(* CODESYS project Rack.project

Project tree, tasks and I/O mapping:
  Device : AM401-CPU1608TP/TN, Shenzhen Inovance Control Technology, version 3.5.11.11
      settings: PersistentStartAdddr = 120000; PersistentStartEndAddr = 491519; Mode = 1
    application Application
      libraries: Standard, * (System); CmpLog, 3.5.5.0 (System); SysMem, 3.5.5.0 (System); CmpEventMgr, 3.5.8.0 (System); CmpApp, 3.5.11.0 (System)
      task MainTask (cyclic, interval 20 ms, priority 1) calls PLC_PRG
      task ETHERCAT (cyclic, interval 4000 µs, priority 0) calls ETHERCAT.EtherCAT_Task, Axis_Ctrl
      02_功能块/
        气缸/
          function block FB_Cylinder [LD]
        初始化/
          function block FB_LineCylinderInit [LD]
          function block FB_MainlineInit [LD]
          function block FB_MaterialInit [LD]
          function block FB_CylinderInit [LD]
      01_变量/
        global variables PersistentVars
        global variables GVL_FB
        global variables GVL_X
        global variables GVL_G
        global variables GVL_H
        global variables GVL_T
        global variables GVL_Q
        global variables GVL_O
        global variables GVT_INT
        global variables GVL_Axis
      03_程序/
        自动/
          program Auto_A [LD]
          program Auto_C [LD]
        输出/
          program Other [LD]
          program Cylinder_AZone [ST]
          program Cylinder_CZone [ST]
        系统/
          program Mode [LD]
          program Rst [LD]
        异常/
          program Error [LD]
        伺服控制/
          program Axis_Teaching [LD]
          program Axis_Ctrl [LD]
        OB/
          program PLC_PRG [ST]
      DifferentialMonitor
    ConfigStorage
    Device Diagnosis
    Network Configuration
      LocalBus Config
      EtherCAT Config
    HardWare Configuration
    资源使用表
    SoftMotion General Axis Pool
    HIGH_SPEED_IO : High Speed IO Module, Inovance, version 00.00.00.20
        unmapped channels: %IW0 InputData, %QB0 OutputData
      HSIO
    HwConfiguratioinDevice : SystemConfig, Inovance, version 00.00.00.10
        settings: NetworkConfigArray.NetworkConfigArray.BusType = 10; NetworkConfigArray.NetworkConfigArray.RackSum = 1; NetworkConfigArray.NetworkConfigArray.HardwareConfigArray.HardwareConfigArray.RackNo = 1
    ETHERCAT : EtherCAT Master, 3S - Smart Software Solutions GmbH, version 3.5.11.10
        settings:  = 0; NetworkName = 'eth1'; SelectNetworkByName = TRUE; DisableTaskGeneration = True
      Z1 : SV660_1Axis_V0.08, Inovance, order no. InoSV660N, version Revision=16#00010000
          settings: WriteValueList = H03-03_8195_4_1_UINT_RW;H03-05_8195_6_1_UINT_RW;H03-06_8195_7_31_UINT_RW;H03-07_8195_8_0_UINT_RW;; Number of Outputs = 2; Number of Inputs = 4; Number of Infos about Outputs = 2; Number of Infos about Inputs = 4; Sync.Length = 6; Sync.Length = 12; FMMU.Length = 6; FMMU.Length = 12; AutoUpdate = False; DC sync0 cycletime = 4000; DC sync1 cycletime = 4000; Number of SDO = 9; Homing method.Index = 16#6098; Homing method.Subindex = 16#00; Homing method.Value = 29; Homing method.Size = 8; Homing method.AbortIfError = FALSE; Homing method.JumpToLine = FALSE; Homing method.Line = 0; Homing method.CompleteAccess = FALSE; Speed during search for switch.Index = 16#6099; Speed during search for switch.Subindex = 16#01; Speed during search for switch.Value = 8388608; Speed during search for switch.Size = 32; Speed during search for switch.AbortIfError = FALSE; Speed during search for switch.JumpToLine = FALSE; Speed during search for switch.Line = 0; Speed during search for switch.CompleteAccess = FALSE; Homing acceleration.Index = 16#609A; Homing acceleration.Subindex = 16#00; Homing acceleration.Value = 167772160; Homing acceleration.Size = 32; Homing acceleration.AbortIfError = FALSE; Homing acceleration.JumpToLine = FALSE; Homing acceleration.Line = 0; Homing acceleration.CompleteAccess = FALSE; Speed during search for zero.Index = 16#6099; Speed during search for zero.Subindex = 16#02; Speed during search for zero.Value = 3355443;
            Speed during search for zero.Size = 32; Speed during search for zero.AbortIfError = FALSE; Speed during search for zero.JumpToLine = FALSE; Speed during search for zero.Line = 0; Speed during search for zero.CompleteAccess = FALSE; Time of home searching.Index = 16#2005; Time of home searching.Subindex = 16#24; Time of home searching.Value = 50000; Time of home searching.Size = 16; Time of home searching.AbortIfError = FALSE; Time of home searching.JumpToLine = FALSE; Time of home searching.Line = 0; Time of home searching.CompleteAccess = FALSE; Positive torque limit value.Index = 16#60E0; Positive torque limit value.Subindex = 16#00; Positive torque limit value.Value = 5000; Positive torque limit value.Size = 16; Positive torque limit value.AbortIfError = FALSE; Positive torque limit value.JumpToLine = FALSE; Positive torque limit value.Line = 0; Positive torque limit value.CompleteAccess = FALSE; Negative torque limit value.Index = 16#60E1; Negative torque limit value.Subindex = 16#00; Negative torque limit value.Value = 5000; Negative torque limit value.Size = 16; Negative torque limit value.AbortIfError = FALSE; Negative torque limit value.JumpToLine = FALSE; Negative torque limit value.Line = 0; Negative torque limit value.CompleteAccess = FALSE; Max profile velocity.Index = 16#607F; Max profile velocity.Subindex = 16#00; Max profile velocity.Value = 167772160; Max profile velocity.Size = 32; Max profile velocity.AbortIfError = FALSE; Max profile velocity.JumpToLine = FALSE; Max profile velocity.Line = 0; Max profile velocity.CompleteAccess = FALSE; RxTxPdo.NumberofEntries = 2; RxTxPdo.Sm = 2; RxTxPdo.DependOnSlot = False;
            RxTxPdo.DependOnSlotGroup = False; RxTxPdo.OverwrittenByModule = False; Exclude = [16#1701,16#1702,16#1703,16#1704,16#1705]; Controlword.Index = 16#6040; Controlword.SubIndex = 0; Controlword.Size = 16; Controlword.Offset = 0; Controlword.DependOnSlot = False; Controlword.DependOnSlotGroup = False; Target position.Index = 16#607A; Target position.SubIndex = 0; Target position.Size = 32; Target position.Offset = 0; Target position.DependOnSlot = False; Target position.DependOnSlotGroup = False; RxTxPdo.Sm = -1; RxTxPdo.NumberofEntries = 4; RxTxPdo.Index = 16#1A00; RxTxPdo.Sm = 3; RxTxPdo.DependOnSlot = False; RxTxPdo.DependOnSlotGroup = False; RxTxPdo.OverwrittenByModule = False; Exclude = [16#1B01,16#1B02,16#1B03,16#1B04]; Error code.Index = 16#603F; Error code.SubIndex = 0; Error code.Size = 16; Error code.Offset = 0; Error code.DependOnSlot = False; Error code.DependOnSlotGroup = False; Statusword.Index = 16#6041; Statusword.SubIndex = 0; Statusword.Size = 16; Statusword.Offset = 0; Statusword.DependOnSlot = False; Statusword.DependOnSlotGroup = False; Position actual value.Index = 16#6064; Position actual value.SubIndex = 0; Position actual value.Size = 32; Position actual value.Offset = 0; Position actual value.DependOnSlot = False;
            Position actual value.DependOnSlotGroup = False; Digital inputs.Index = 16#60FD; Digital inputs.SubIndex = 0; Digital inputs.Size = 32; Digital inputs.Offset = 0; Digital inputs.DependOnSlot = False; Digital inputs.DependOnSlotGroup = False; RxTxPdo.Sm = -1; Controlword.Name = 'Controlword'; Controlword.DataType = 'UINT'; Controlword.Default = ''; Controlword.Comment = ''; Target position.Name = 'Target position'; Target position.DataType = 'DINT'; Target position.Default = ''; Target position.Comment = ''; Error code.Name = 'Error code'; Error code.DataType = 'UINT'; Error code.Default = ''; Error code.Comment = ''; Statusword.Name = 'Statusword'; Statusword.DataType = 'UINT'; Statusword.Default = ''; Statusword.Comment = ''; Position actual value.Name = 'Position actual value'; Position actual value.DataType = 'DINT'; Position actual value.Default = ''; Position actual value.Comment = ''; Digital inputs.Name = 'Digital inputs'; Digital inputs.DataType = 'UDINT'; Digital inputs.Default = ''; Digital inputs.Comment = ''
          unmapped channels: %QW100 Controlword, %QD102 Target position, %IW100 Error code, %IW102 Statusword, %ID104 Position actual value, %ID106 Digital inputs
        Axis_1 : Axis, 3S - Smart Software Solutions GmbH, order no. 0, version 4.0.0.0
            settings: wDriveID = 0; dwRatioTechUnitsDenom = 8388608; iRatioTechUnitsNum = 5; 4000 = 1; 4001 = 0; 4003 = true; 4004 = 26; 4005 = 0; 4006 = 5; 4007 = 100; 4008 = 2; 4009 = 50000; 4010 = 5000; 4011 = 5000; 4012 = 100; ScalingIncs = 16#800000; 6005 = 5; AdrOffset_8010 = 200; BitOffset_8010 = 0; BitLength_8010 = 16; Address_8010 = '%QW100'; Type_8010 = 'UINT'; AddressPointer_8010 = ADR(%QW100); AdrOffset_8020 = 408; BitOffset_8020 = 0; BitLength_8020 = 32; Address_8020 = '%QD102'; Type_8020 = 'DINT'; AddressPointer_8020 = ADR(%QD102); AdrOffset_8030 = 4294967295; BitOffset_8030 = 0; BitLength_8030 = 0; Address_8030 = ''; Type_8030 = ''; AddressPointer_8030 = 0; AdrOffset_8040 = 4294967295; BitOffset_8040 = 0; BitLength_8040 = 0; Address_8040 = ''; Type_8040 = '';
              AddressPointer_8040 = 0; AdrOffset_8050 = 4294967295; BitOffset_8050 = 0; BitLength_8050 = 0; Address_8050 = ''; Type_8050 = ''; AddressPointer_8050 = 0; AdrOffset_8060 = 4294967295; BitOffset_8060 = 0; BitLength_8060 = 0; Address_8060 = ''; Type_8060 = ''; AddressPointer_8060 = 0; AdrOffset_8070 = 4294967295; BitOffset_8070 = 0; BitLength_8070 = 0; Address_8070 = ''; Type_8070 = ''; AddressPointer_8070 = 0; AdrOffset_8080 = 4294967295; BitOffset_8080 = 0; BitLength_8080 = 0; Address_8080 = ''; Type_8080 = ''; AddressPointer_8080 = 0; AdrOffset_8090 = 4294967295; BitOffset_8090 = 0; BitLength_8090 = 0; Address_8090 = ''; Type_8090 = ''; AddressPointer_8090 = 0; AdrOffset_8510 = 204; BitOffset_8510 = 0; BitLength_8510 = 16; Address_8510 = '%IW102'; Type_8510 = 'UINT'; AddressPointer_8510 = ADR(%IW102); AdrOffset_8520 = 416; BitOffset_8520 = 0; BitLength_8520 = 32;
              Address_8520 = '%ID104'; Type_8520 = 'DINT'; AddressPointer_8520 = ADR(%ID104); AdrOffset_8530 = 4294967295; BitOffset_8530 = 0; BitLength_8530 = 0; Address_8530 = ''; Type_8530 = ''; AddressPointer_8530 = 0; AdrOffset_8540 = 4294967295; BitOffset_8540 = 0; BitLength_8540 = 0; Address_8540 = ''; Type_8540 = ''; AddressPointer_8540 = 0; AdrOffset_8550 = 4294967295; BitOffset_8550 = 0; BitLength_8550 = 0; Address_8550 = ''; Type_8550 = ''; AddressPointer_8550 = 0; AdrOffset_8560 = 424; BitOffset_8560 = 0; BitLength_8560 = 32; Address_8560 = '%ID106'; Type_8560 = 'UDINT'; AddressPointer_8560 = ADR(%ID106); AdrOffset_8570 = 4294967295; BitOffset_8570 = 0; BitLength_8570 = 0; Address_8570 = ''; Type_8570 = ''; AddressPointer_8570 = 0; AdrOffset_8580 = 4294967295; BitOffset_8580 = 0; BitLength_8580 = 0; Address_8580 = ''; Type_8580 = ''; AddressPointer_8580 = 0; AdrOffset_8590 = 4294967295;
              BitOffset_8590 = 0; BitLength_8590 = 0; Address_8590 = ''; Type_8590 = ''; AddressPointer_8590 = 0; AdrOffset_8600 = 4294967295; BitOffset_8600 = 0; BitLength_8600 = 0; Address_8600 = ''; Type_8600 = ''; AddressPointer_8600 = 0; AdrOffset_8600 = 4294967295; BitOffset_8600 = 0; BitLength_8600 = 0; Address_8610 = ''; Type_8610 = ''; AddressPointer_8610 = 0; AdrOffset_8620 = 4294967295; BitOffset_8620 = 0; BitLength_8620 = 0; Address_8620 = ''; Type_8620 = ''; AddressPointer_8620 = 0
      C2_EC_12_B12 : C2-EC-12-B12, Sico Robot Automatic Technology (Nanjing) Co., Ltd., order no. C2-EC-12-B12, version Revision=16#00000001
          settings: AutoUpdate = False; DC sync0 cycletime = 4000; DC sync1 cycletime = 4000
          unmapped channels: %QX14.0 a[0..7], %QX14.1 a[0..7], %QX14.2 a[0..7], %QX14.3 a[0..7], %QX14.4 a[0..7], %QX14.5 a[0..7], %QX14.6 a[0..7], %QX14.7 a[0..7], %QX15.0 a[8..15], %QX15.1 a[8..15], %QX15.2 a[8..15], %QX15.3 a[8..15], %QX15.4 a[8..15], %QX15.5 a[8..15], %QX15.6 a[8..15], %QX15.7 a[8..15], %QX16.0 b[0..7], %QX16.1 b[0..7], %QX16.2 b[0..7], %QX16.3 b[0..7], %QX16.4 b[0..7], %QX16.5 b[0..7], %QX16.6 b[0..7], %QX16.7 b[0..7], %QX17.0 b[8..15], %QX17.1 b[8..15], %QX17.2 b[8..15], %QX17.3 b[8..15], %QX17.4 b[8..15], %QX17.5 b[8..15], %QX17.6 b[8..15], %QX17.7 b[8..15]
      C2_EC_12_B12_1 : C2-EC-12-B12, Sico Robot Automatic Technology (Nanjing) Co., Ltd., order no. C2-EC-12-B12, version Revision=16#00000001
          settings: AutoUpdate = False; DC sync0 cycletime = 4000; DC sync1 cycletime = 4000
          unmapped channels: %QX10.0 a[0..7], %QX10.1 a[0..7], %QX10.2 a[0..7], %QX10.3 a[0..7], %QX10.4 a[0..7], %QX10.5 a[0..7], %QX10.6 a[0..7], %QX10.7 a[0..7], %QX11.0 a[8..15], %QX11.1 a[8..15], %QX11.2 a[8..15], %QX11.3 a[8..15], %QX11.4 a[8..15], %QX11.5 a[8..15], %QX11.6 a[8..15], %QX11.7 a[8..15], %QX12.0 b[0..7], %QX12.1 b[0..7], %QX12.2 b[0..7], %QX12.3 b[0..7], %QX12.4 b[0..7], %QX12.5 b[0..7], %QX12.6 b[0..7], %QX12.7 b[0..7], %QX13.0 b[8..15], %QX13.1 b[8..15], %QX13.2 b[8..15], %QX13.3 b[8..15], %QX13.4 b[8..15], %QX13.5 b[8..15], %QX13.6 b[8..15], %QX13.7 b[8..15]
      GL10_RTU_ECTA : GL10-RTU-ECTA_2.0.6.0, Inovance, order no. GL10-RTU-ECTA, version Revision=16#01006000
          settings: Number of Outputs = 2; Number of Inputs = 9; IOModuleSize = 3; IOModuleName = GL10_3200END_2,GL10_3200END_3,GL10_0016ETN_1; IOModuleGuid = f377121e-49ca-4d15-9928-081e798ca8d1,1747bdd4-14e3-4bcd-ac98-21177ad82d1b,2504b1f7-36b1-4a3c-950b-33998ed58a91; Number of Infos about Outputs = 2; Number of Infos about Inputs = 9; Sync.Length = 2; Sync.Length = 10; FMMU.Length = 2; FMMU.Length = 10; Number of RxPDOs of the Slave = 4; Number of TxPDOs of the Slave = 5; AutoUpdate = False; DC sync0 cycletime = 4000; DC sync1 cycletime = 4000; Number of SDO = 11; DO module output mode after EtherCAT lost link.Index = 16#8202; DO module output mode after EtherCAT lost link.Subindex = 16#01; DO module output mode after EtherCAT lost link.Value = 65535; DO module output mode after EtherCAT lost link.Size = 16; DO module output mode after EtherCAT lost link.AbortIfError = FALSE; DO module output mode after EtherCAT lost link.JumpToLine = FALSE; DO module output mode after EtherCAT lost link.Line = 0; DO module output mode after EtherCAT lost link.CompleteAccess = False; DO module output value after EtherCAT lost link.Index = 16#8202; DO module output value after EtherCAT lost link.Subindex = 16#02; DO module output value after EtherCAT lost link.Value = 0; DO module output value after EtherCAT lost link.Size = 16; DO module output value after EtherCAT lost link.AbortIfError = FALSE; DO module output value after EtherCAT lost link.JumpToLine = FALSE; DO module output value after EtherCAT lost link.Line = 0; DO module output value after EtherCAT lost link.CompleteAccess = False; clear slot cfg 0xf030 entries.Index = 16#F030; clear slot cfg 0xf030 entries.Subindex = 16#00; clear slot cfg 0xf030 entries.Value = 0; clear slot cfg 0xf030 entries.Size = 8; clear slot cfg 0xf030 entries.AbortIfError = FALSE; clear slot cfg 0xf030 entries.JumpToLine = FALSE; clear slot cfg 0xf030 entries.Line = 0;
            clear slot cfg 0xf030 entries.CompleteAccess = False; download slot cfg 0xf030 entry.Index = 16#F030; download slot cfg 0xf030 entry.Subindex = 16#01; download slot cfg 0xf030 entry.Value = 284426769; download slot cfg 0xf030 entry.Size = 32; download slot cfg 0xf030 entry.AbortIfError = FALSE; download slot cfg 0xf030 entry.JumpToLine = FALSE; download slot cfg 0xf030 entry.Line = 0; download slot cfg 0xf030 entry.CompleteAccess = False; download slot cfg 0xf030 entry.Index = 16#F030; download slot cfg 0xf030 entry.Subindex = 16#02; download slot cfg 0xf030 entry.Value = 284426769; download slot cfg 0xf030 entry.Size = 32; download slot cfg 0xf030 entry.AbortIfError = FALSE; download slot cfg 0xf030 entry.JumpToLine = FALSE; download slot cfg 0xf030 entry.Line = 0; download slot cfg 0xf030 entry.CompleteAccess = False; download slot cfg 0xf030 entry.Index = 16#F030; download slot cfg 0xf030 entry.Subindex = 16#03; download slot cfg 0xf030 entry.Value = 284426784; download slot cfg 0xf030 entry.Size = 32; download slot cfg 0xf030 entry.AbortIfError = FALSE; download slot cfg 0xf030 entry.JumpToLine = FALSE; download slot cfg 0xf030 entry.Line = 0; download slot cfg 0xf030 entry.CompleteAccess = False; download slot cfg 0xf030 entry count.Index = 16#F030; download slot cfg 0xf030 entry count.Subindex = 16#00; download slot cfg 0xf030 entry count.Value = 3; download slot cfg 0xf030 entry count.Size = 8; download slot cfg 0xf030 entry count.AbortIfError = FALSE; download slot cfg 0xf030 entry count.JumpToLine = FALSE; download slot cfg 0xf030 entry count.Line = 0; download slot cfg 0xf030 entry count.CompleteAccess = False; RxTxPdo.NumberofExcludes = 0; RxTxPdo.NumberofEntries = 1; RxTxPdo.Index = 16#17A0; RxTxPdo.Fixed = True; RxTxPdo.Mandatory = False; RxTxPdo.Virtual = False; RxTxPdo.Sm = -1;
            RxTxPdo.Su = -1; RxTxPdo.Name = 'Device RPDO Mapping parameter'; RxTxPdo.DependOnSlot = False; RxTxPdo.DependOnSlotGroup = False; RxTxPdo.OverwrittenByModule = False; Device control.Index = 16#FB00; Device control.SubIndex = 0; Device control.Size = 16; Device control.Offset = 0; Device control.DependOnSlot = False; Device control.DependOnSlotGroup = False; RxTxPdo.NumberofExcludes = 1; RxTxPdo.NumberofEntries = 2; RxTxPdo.Index = 16#1620; RxTxPdo.Fixed = True; RxTxPdo.Mandatory = False; RxTxPdo.Virtual = False; RxTxPdo.Sm = 2; RxTxPdo.Su = 0; RxTxPdo.Name = '0016XXX Output maping'; RxTxPdo.DependOnSlot = True; RxTxPdo.DependOnSlotGroup = False; RxTxPdo.OverwrittenByModule = True; Exclude = 16#1624; GL10_0016ETN_1 Digital output CH1-8bit.Index = 16#7202; GL10_0016ETN_1 Digital output CH1-8bit.SubIndex = 1; GL10_0016ETN_1 Digital output CH1-8bit.Size = 8; GL10_0016ETN_1 Digital output CH1-8bit.Offset = 0; GL10_0016ETN_1 Digital output CH1-8bit.DependOnSlot = True; GL10_0016ETN_1 Digital output CH1-8bit.DependOnSlotGroup = True; GL10_0016ETN_1 Digital output CH2-8bit.Index = 16#7202; GL10_0016ETN_1 Digital output CH2-8bit.SubIndex = 2; GL10_0016ETN_1 Digital output CH2-8bit.Size = 8; GL10_0016ETN_1 Digital output CH2-8bit.Offset = 0; GL10_0016ETN_1 Digital output CH2-8bit.DependOnSlot = True; GL10_0016ETN_1 Digital output CH2-8bit.DependOnSlotGroup = True; RxTxPdo.NumberofExcludes = 1; RxTxPdo.NumberofEntries = 16; RxTxPdo.Index = 16#1624; RxTxPdo.Fixed = True;
            RxTxPdo.Mandatory = False; RxTxPdo.Virtual = False; RxTxPdo.Sm = -1; RxTxPdo.Su = 0; RxTxPdo.Name = '0016XXX Output maping'; RxTxPdo.DependOnSlot = True; RxTxPdo.DependOnSlotGroup = False; RxTxPdo.OverwrittenByModule = True; Exclude = 16#1620; GL10_0016ETN_1 Digital output CH1-bit0.Index = 16#7203; GL10_0016ETN_1 Digital output CH1-bit0.SubIndex = 1; GL10_0016ETN_1 Digital output CH1-bit0.Size = 1; GL10_0016ETN_1 Digital output CH1-bit0.Offset = 0; GL10_0016ETN_1 Digital output CH1-bit0.DependOnSlot = True; GL10_0016ETN_1 Digital output CH1-bit0.DependOnSlotGroup = True; GL10_0016ETN_1 Digital output CH1-bit1.Index = 16#7203; GL10_0016ETN_1 Digital output CH1-bit1.SubIndex = 2; GL10_0016ETN_1 Digital output CH1-bit1.Size = 1; GL10_0016ETN_1 Digital output CH1-bit1.Offset = 0; GL10_0016ETN_1 Digital output CH1-bit1.DependOnSlot = True; GL10_0016ETN_1 Digital output CH1-bit1.DependOnSlotGroup = True; GL10_0016ETN_1 Digital output CH1-bit2.Index = 16#7203; GL10_0016ETN_1 Digital output CH1-bit2.SubIndex = 3; GL10_0016ETN_1 Digital output CH1-bit2.Size = 1; GL10_0016ETN_1 Digital output CH1-bit2.Offset = 0; GL10_0016ETN_1 Digital output CH1-bit2.DependOnSlot = True; GL10_0016ETN_1 Digital output CH1-bit2.DependOnSlotGroup = True; GL10_0016ETN_1 Digital output CH1-bit3.Index = 16#7203; GL10_0016ETN_1 Digital output CH1-bit3.SubIndex = 4; GL10_0016ETN_1 Digital output CH1-bit3.Size = 1; GL10_0016ETN_1 Digital output CH1-bit3.Offset = 0; GL10_0016ETN_1 Digital output CH1-bit3.DependOnSlot = True; GL10_0016ETN_1 Digital output CH1-bit3.DependOnSlotGroup = True; GL10_0016ETN_1 Digital output CH1-bit4.Index = 16#7203; GL10_0016ETN_1 Digital output CH1-bit4.SubIndex = 5; GL10_0016ETN_1 Digital output CH1-bit4.Size = 1; GL10_0016ETN_1 Digital output CH1-bit4.Offset = 0; GL10_0016ETN_1 Digital output CH1-bit4.DependOnSlot = True; GL10_0016ETN_1 Digital output CH1-bit4.DependOnSlotGroup = True; GL10_0016ETN_1 Digital output CH1-bit5.Index = 16#7203;
            GL10_0016ETN_1 Digital output CH1-bit5.SubIndex = 6; GL10_0016ETN_1 Digital output CH1-bit5.Size = 1; GL10_0016ETN_1 Digital output CH1-bit5.Offset = 0; GL10_0016ETN_1 Digital output CH1-bit5.DependOnSlot = True; GL10_0016ETN_1 Digital output CH1-bit5.DependOnSlotGroup = True; GL10_0016ETN_1 Digital output CH1-bit6.Index = 16#7203; GL10_0016ETN_1 Digital output CH1-bit6.SubIndex = 7; GL10_0016ETN_1 Digital output CH1-bit6.Size = 1; GL10_0016ETN_1 Digital output CH1-bit6.Offset = 0; GL10_0016ETN_1 Digital output CH1-bit6.DependOnSlot = True; GL10_0016ETN_1 Digital output CH1-bit6.DependOnSlotGroup = True; GL10_0016ETN_1 Digital output CH1-bit7.Index = 16#7203; GL10_0016ETN_1 Digital output CH1-bit7.SubIndex = 8; GL10_0016ETN_1 Digital output CH1-bit7.Size = 1; GL10_0016ETN_1 Digital output CH1-bit7.Offset = 0; GL10_0016ETN_1 Digital output CH1-bit7.DependOnSlot = True; GL10_0016ETN_1 Digital output CH1-bit7.DependOnSlotGroup = True; GL10_0016ETN_1 Digital output CH2-bit0.Index = 16#7203; GL10_0016ETN_1 Digital output CH2-bit0.SubIndex = 9; GL10_0016ETN_1 Digital output CH2-bit0.Size = 1; GL10_0016ETN_1 Digital output CH2-bit0.Offset = 0; GL10_0016ETN_1 Digital output CH2-bit0.DependOnSlot = True; GL10_0016ETN_1 Digital output CH2-bit0.DependOnSlotGroup = True; GL10_0016ETN_1 Digital output CH2-bit1.Index = 16#7203; GL10_0016ETN_1 Digital output CH2-bit1.SubIndex = 10; GL10_0016ETN_1 Digital output CH2-bit1.Size = 1; GL10_0016ETN_1 Digital output CH2-bit1.Offset = 0; GL10_0016ETN_1 Digital output CH2-bit1.DependOnSlot = True; GL10_0016ETN_1 Digital output CH2-bit1.DependOnSlotGroup = True; GL10_0016ETN_1 Digital output CH2-bit2.Index = 16#7203; GL10_0016ETN_1 Digital output CH2-bit2.SubIndex = 11; GL10_0016ETN_1 Digital output CH2-bit2.Size = 1; GL10_0016ETN_1 Digital output CH2-bit2.Offset = 0; GL10_0016ETN_1 Digital output CH2-bit2.DependOnSlot = True; GL10_0016ETN_1 Digital output CH2-bit2.DependOnSlotGroup = True; GL10_0016ETN_1 Digital output CH2-bit3.Index = 16#7203; GL10_0016ETN_1 Digital output CH2-bit3.SubIndex = 12; GL10_0016ETN_1 Digital output CH2-bit3.Size = 1; GL10_0016ETN_1 Digital output CH2-bit3.Offset = 0; GL10_0016ETN_1 Digital output CH2-bit3.DependOnSlot = True;
            GL10_0016ETN_1 Digital output CH2-bit3.DependOnSlotGroup = True; GL10_0016ETN_1 Digital output CH2-bit4.Index = 16#7203; GL10_0016ETN_1 Digital output CH2-bit4.SubIndex = 13; GL10_0016ETN_1 Digital output CH2-bit4.Size = 1; GL10_0016ETN_1 Digital output CH2-bit4.Offset = 0; GL10_0016ETN_1 Digital output CH2-bit4.DependOnSlot = True; GL10_0016ETN_1 Digital output CH2-bit4.DependOnSlotGroup = True; GL10_0016ETN_1 Digital output CH2-bit5.Index = 16#7203; GL10_0016ETN_1 Digital output CH2-bit5.SubIndex = 14; GL10_0016ETN_1 Digital output CH2-bit5.Size = 1; GL10_0016ETN_1 Digital output CH2-bit5.Offset = 0; GL10_0016ETN_1 Digital output CH2-bit5.DependOnSlot = True; GL10_0016ETN_1 Digital output CH2-bit5.DependOnSlotGroup = True; GL10_0016ETN_1 Digital output CH2-bit6.Index = 16#7203; GL10_0016ETN_1 Digital output CH2-bit6.SubIndex = 15; GL10_0016ETN_1 Digital output CH2-bit6.Size = 1; GL10_0016ETN_1 Digital output CH2-bit6.Offset = 0; GL10_0016ETN_1 Digital output CH2-bit6.DependOnSlot = True; GL10_0016ETN_1 Digital output CH2-bit6.DependOnSlotGroup = True; GL10_0016ETN_1 Digital output CH2-bit7.Index = 16#7203; GL10_0016ETN_1 Digital output CH2-bit7.SubIndex = 16; GL10_0016ETN_1 Digital output CH2-bit7.Size = 1; GL10_0016ETN_1 Digital output CH2-bit7.Offset = 0; GL10_0016ETN_1 Digital output CH2-bit7.DependOnSlot = True; GL10_0016ETN_1 Digital output CH2-bit7.DependOnSlotGroup = True; RxTxPdo.NumberofExcludes = 0; RxTxPdo.NumberofEntries = 2; RxTxPdo.Index = 16#1622; RxTxPdo.Fixed = True; RxTxPdo.Mandatory = False; RxTxPdo.Virtual = False; RxTxPdo.Sm = -1; RxTxPdo.Su = 0; RxTxPdo.Name = '0016XXX Control maping'; RxTxPdo.DependOnSlot = True; RxTxPdo.DependOnSlotGroup = False; RxTxPdo.OverwrittenByModule = True; GL10_0016ETN_1 DO module output mode after EtherCAT lost link.Index = 16#8202; GL10_0016ETN_1 DO module output mode after EtherCAT lost link.SubIndex = 1; GL10_0016ETN_1 DO module output mode after EtherCAT lost link.Size = 16;
            GL10_0016ETN_1 DO module output mode after EtherCAT lost link.Offset = 0; GL10_0016ETN_1 DO module output mode after EtherCAT lost link.DependOnSlot = True; GL10_0016ETN_1 DO module output mode after EtherCAT lost link.DependOnSlotGroup = True; GL10_0016ETN_1 DO module output value after EtherCAT lost link.Index = 16#8202; GL10_0016ETN_1 DO module output value after EtherCAT lost link.SubIndex = 2; GL10_0016ETN_1 DO module output value after EtherCAT lost link.Size = 16; GL10_0016ETN_1 DO module output value after EtherCAT lost link.Offset = 0; GL10_0016ETN_1 DO module output value after EtherCAT lost link.DependOnSlot = True; GL10_0016ETN_1 DO module output value after EtherCAT lost link.DependOnSlotGroup = True; RxTxPdo.NumberofExcludes = 0; RxTxPdo.NumberofEntries = 1; RxTxPdo.Index = 16#1BA0; RxTxPdo.Fixed = True; RxTxPdo.Mandatory = False; RxTxPdo.Virtual = False; RxTxPdo.Sm = 3; RxTxPdo.Su = 3; RxTxPdo.Name = 'Device TPDO Mapping parameter'; RxTxPdo.DependOnSlot = False; RxTxPdo.DependOnSlotGroup = False; RxTxPdo.OverwrittenByModule = False; Device status.Index = 16#F100; Device status.SubIndex = 0; Device status.Size = 16; Device status.Offset = 0; Device status.DependOnSlot = False; Device status.DependOnSlotGroup = False; RxTxPdo.NumberofExcludes = 1; RxTxPdo.NumberofEntries = 4; RxTxPdo.Index = 16#1A00; RxTxPdo.Fixed = True; RxTxPdo.Mandatory = False; RxTxPdo.Virtual = False; RxTxPdo.Sm = 3; RxTxPdo.Su = 0; RxTxPdo.Name = '3200END Input maping'; RxTxPdo.DependOnSlot = True; RxTxPdo.DependOnSlotGroup = False; RxTxPdo.OverwrittenByModule = True; Exclude = 16#1A04;
            GL10_3200END_2 Digital input CH1-8bit.Index = 16#6001; GL10_3200END_2 Digital input CH1-8bit.SubIndex = 1; GL10_3200END_2 Digital input CH1-8bit.Size = 8; GL10_3200END_2 Digital input CH1-8bit.Offset = 0; GL10_3200END_2 Digital input CH1-8bit.DependOnSlot = True; GL10_3200END_2 Digital input CH1-8bit.DependOnSlotGroup = True; GL10_3200END_2 Digital input CH2-8bit.Index = 16#6001; GL10_3200END_2 Digital input CH2-8bit.SubIndex = 2; GL10_3200END_2 Digital input CH2-8bit.Size = 8; GL10_3200END_2 Digital input CH2-8bit.Offset = 0; GL10_3200END_2 Digital input CH2-8bit.DependOnSlot = True; GL10_3200END_2 Digital input CH2-8bit.DependOnSlotGroup = True; GL10_3200END_2 Digital input CH3-8bit.Index = 16#6001; GL10_3200END_2 Digital input CH3-8bit.SubIndex = 3; GL10_3200END_2 Digital input CH3-8bit.Size = 8; GL10_3200END_2 Digital input CH3-8bit.Offset = 0; GL10_3200END_2 Digital input CH3-8bit.DependOnSlot = True; GL10_3200END_2 Digital input CH3-8bit.DependOnSlotGroup = True; GL10_3200END_2 Digital input CH4-8bit.Index = 16#6001; GL10_3200END_2 Digital input CH4-8bit.SubIndex = 4; GL10_3200END_2 Digital input CH4-8bit.Size = 8; GL10_3200END_2 Digital input CH4-8bit.Offset = 0; GL10_3200END_2 Digital input CH4-8bit.DependOnSlot = True; GL10_3200END_2 Digital input CH4-8bit.DependOnSlotGroup = True; RxTxPdo.NumberofExcludes = 1; RxTxPdo.NumberofEntries = 32; RxTxPdo.Index = 16#1A04; RxTxPdo.Fixed = True; RxTxPdo.Mandatory = False; RxTxPdo.Virtual = False; RxTxPdo.Sm = -1; RxTxPdo.Su = 0; RxTxPdo.Name = '3200END Input maping'; RxTxPdo.DependOnSlot = True; RxTxPdo.DependOnSlotGroup = False; RxTxPdo.OverwrittenByModule = True; Exclude = 16#1A00; GL10_3200END_2 Digital input CH1-bit0.Index = 16#6002; GL10_3200END_2 Digital input CH1-bit0.SubIndex = 1; GL10_3200END_2 Digital input CH1-bit0.Size = 1;
            GL10_3200END_2 Digital input CH1-bit0.Offset = 0; GL10_3200END_2 Digital input CH1-bit0.DependOnSlot = True; GL10_3200END_2 Digital input CH1-bit0.DependOnSlotGroup = True; GL10_3200END_2 Digital input CH1-bit1.Index = 16#6002; GL10_3200END_2 Digital input CH1-bit1.SubIndex = 2; GL10_3200END_2 Digital input CH1-bit1.Size = 1; GL10_3200END_2 Digital input CH1-bit1.Offset = 0; GL10_3200END_2 Digital input CH1-bit1.DependOnSlot = True; GL10_3200END_2 Digital input CH1-bit1.DependOnSlotGroup = True; GL10_3200END_2 Digital input CH1-bit2.Index = 16#6002; GL10_3200END_2 Digital input CH1-bit2.SubIndex = 3; GL10_3200END_2 Digital input CH1-bit2.Size = 1; GL10_3200END_2 Digital input CH1-bit2.Offset = 0; GL10_3200END_2 Digital input CH1-bit2.DependOnSlot = True; GL10_3200END_2 Digital input CH1-bit2.DependOnSlotGroup = True; GL10_3200END_2 Digital input CH1-bit3.Index = 16#6002; GL10_3200END_2 Digital input CH1-bit3.SubIndex = 4; GL10_3200END_2 Digital input CH1-bit3.Size = 1; GL10_3200END_2 Digital input CH1-bit3.Offset = 0; GL10_3200END_2 Digital input CH1-bit3.DependOnSlot = True; GL10_3200END_2 Digital input CH1-bit3.DependOnSlotGroup = True; GL10_3200END_2 Digital input CH1-bit4.Index = 16#6002; GL10_3200END_2 Digital input CH1-bit4.SubIndex = 5; GL10_3200END_2 Digital input CH1-bit4.Size = 1; GL10_3200END_2 Digital input CH1-bit4.Offset = 0; GL10_3200END_2 Digital input CH1-bit4.DependOnSlot = True; GL10_3200END_2 Digital input CH1-bit4.DependOnSlotGroup = True; GL10_3200END_2 Digital input CH1-bit5.Index = 16#6002; GL10_3200END_2 Digital input CH1-bit5.SubIndex = 6; GL10_3200END_2 Digital input CH1-bit5.Size = 1; GL10_3200END_2 Digital input CH1-bit5.Offset = 0; GL10_3200END_2 Digital input CH1-bit5.DependOnSlot = True; GL10_3200END_2 Digital input CH1-bit5.DependOnSlotGroup = True; GL10_3200END_2 Digital input CH1-bit6.Index = 16#6002; GL10_3200END_2 Digital input CH1-bit6.SubIndex = 7; GL10_3200END_2 Digital input CH1-bit6.Size = 1; GL10_3200END_2 Digital input CH1-bit6.Offset = 0; GL10_3200END_2 Digital input CH1-bit6.DependOnSlot = True; GL10_3200END_2 Digital input CH1-bit6.DependOnSlotGroup = True; GL10_3200END_2 Digital input CH1-bit7.Index = 16#6002;
            GL10_3200END_2 Digital input CH1-bit7.SubIndex = 8; GL10_3200END_2 Digital input CH1-bit7.Size = 1; GL10_3200END_2 Digital input CH1-bit7.Offset = 0; GL10_3200END_2 Digital input CH1-bit7.DependOnSlot = True; GL10_3200END_2 Digital input CH1-bit7.DependOnSlotGroup = True; GL10_3200END_2 Digital input CH2-bit0.Index = 16#6002; GL10_3200END_2 Digital input CH2-bit0.SubIndex = 9; GL10_3200END_2 Digital input CH2-bit0.Size = 1; GL10_3200END_2 Digital input CH2-bit0.Offset = 0; GL10_3200END_2 Digital input CH2-bit0.DependOnSlot = True; GL10_3200END_2 Digital input CH2-bit0.DependOnSlotGroup = True; GL10_3200END_2 Digital input CH2-bit1.Index = 16#6002; GL10_3200END_2 Digital input CH2-bit1.SubIndex = 10; GL10_3200END_2 Digital input CH2-bit1.Size = 1; GL10_3200END_2 Digital input CH2-bit1.Offset = 0; GL10_3200END_2 Digital input CH2-bit1.DependOnSlot = True; GL10_3200END_2 Digital input CH2-bit1.DependOnSlotGroup = True; GL10_3200END_2 Digital input CH2-bit2.Index = 16#6002; GL10_3200END_2 Digital input CH2-bit2.SubIndex = 11; GL10_3200END_2 Digital input CH2-bit2.Size = 1; GL10_3200END_2 Digital input CH2-bit2.Offset = 0; GL10_3200END_2 Digital input CH2-bit2.DependOnSlot = True; GL10_3200END_2 Digital input CH2-bit2.DependOnSlotGroup = True; GL10_3200END_2 Digital input CH2-bit3.Index = 16#6002; GL10_3200END_2 Digital input CH2-bit3.SubIndex = 12; GL10_3200END_2 Digital input CH2-bit3.Size = 1; GL10_3200END_2 Digital input CH2-bit3.Offset = 0; GL10_3200END_2 Digital input CH2-bit3.DependOnSlot = True; GL10_3200END_2 Digital input CH2-bit3.DependOnSlotGroup = True; GL10_3200END_2 Digital input CH2-bit4.Index = 16#6002; GL10_3200END_2 Digital input CH2-bit4.SubIndex = 13; GL10_3200END_2 Digital input CH2-bit4.Size = 1; GL10_3200END_2 Digital input CH2-bit4.Offset = 0; GL10_3200END_2 Digital input CH2-bit4.DependOnSlot = True; GL10_3200END_2 Digital input CH2-bit4.DependOnSlotGroup = True; GL10_3200END_2 Digital input CH2-bit5.Index = 16#6002; GL10_3200END_2 Digital input CH2-bit5.SubIndex = 14; GL10_3200END_2 Digital input CH2-bit5.Size = 1; GL10_3200END_2 Digital input CH2-bit5.Offset = 0; GL10_3200END_2 Digital input CH2-bit5.DependOnSlot = True;
            GL10_3200END_2 Digital input CH2-bit5.DependOnSlotGroup = True; GL10_3200END_2 Digital input CH2-bit6.Index = 16#6002; GL10_3200END_2 Digital input CH2-bit6.SubIndex = 15; GL10_3200END_2 Digital input CH2-bit6.Size = 1; GL10_3200END_2 Digital input CH2-bit6.Offset = 0; GL10_3200END_2 Digital input CH2-bit6.DependOnSlot = True; GL10_3200END_2 Digital input CH2-bit6.DependOnSlotGroup = True; GL10_3200END_2 Digital input CH2-bit7.Index = 16#6002; GL10_3200END_2 Digital input CH2-bit7.SubIndex = 16; GL10_3200END_2 Digital input CH2-bit7.Size = 1; GL10_3200END_2 Digital input CH2-bit7.Offset = 0; GL10_3200END_2 Digital input CH2-bit7.DependOnSlot = True; GL10_3200END_2 Digital input CH2-bit7.DependOnSlotGroup = True; GL10_3200END_2 Digital input CH3-bit0.Index = 16#6002; GL10_3200END_2 Digital input CH3-bit0.SubIndex = 17; GL10_3200END_2 Digital input CH3-bit0.Size = 1; GL10_3200END_2 Digital input CH3-bit0.Offset = 0; GL10_3200END_2 Digital input CH3-bit0.DependOnSlot = True; GL10_3200END_2 Digital input CH3-bit0.DependOnSlotGroup = True; GL10_3200END_2 Digital input CH3-bit1.Index = 16#6002; GL10_3200END_2 Digital input CH3-bit1.SubIndex = 18; GL10_3200END_2 Digital input CH3-bit1.Size = 1; GL10_3200END_2 Digital input CH3-bit1.Offset = 0; GL10_3200END_2 Digital input CH3-bit1.DependOnSlot = True; GL10_3200END_2 Digital input CH3-bit1.DependOnSlotGroup = True; GL10_3200END_2 Digital input CH3-bit2.Index = 16#6002; GL10_3200END_2 Digital input CH3-bit2.SubIndex = 19; GL10_3200END_2 Digital input CH3-bit2.Size = 1; GL10_3200END_2 Digital input CH3-bit2.Offset = 0; GL10_3200END_2 Digital input CH3-bit2.DependOnSlot = True; GL10_3200END_2 Digital input CH3-bit2.DependOnSlotGroup = True; GL10_3200END_2 Digital input CH3-bit3.Index = 16#6002; GL10_3200END_2 Digital input CH3-bit3.SubIndex = 20; GL10_3200END_2 Digital input CH3-bit3.Size = 1; GL10_3200END_2 Digital input CH3-bit3.Offset = 0; GL10_3200END_2 Digital input CH3-bit3.DependOnSlot = True; GL10_3200END_2 Digital input CH3-bit3.DependOnSlotGroup = True; GL10_3200END_2 Digital input CH3-bit4.Index = 16#6002; GL10_3200END_2 Digital input CH3-bit4.SubIndex = 21; GL10_3200END_2 Digital input CH3-bit4.Size = 1;
            GL10_3200END_2 Digital input CH3-bit4.Offset = 0; GL10_3200END_2 Digital input CH3-bit4.DependOnSlot = True; GL10_3200END_2 Digital input CH3-bit4.DependOnSlotGroup = True; GL10_3200END_2 Digital input CH3-bit5.Index = 16#6002; GL10_3200END_2 Digital input CH3-bit5.SubIndex = 22; GL10_3200END_2 Digital input CH3-bit5.Size = 1; GL10_3200END_2 Digital input CH3-bit5.Offset = 0; GL10_3200END_2 Digital input CH3-bit5.DependOnSlot = True; GL10_3200END_2 Digital input CH3-bit5.DependOnSlotGroup = True; GL10_3200END_2 Digital input CH3-bit6.Index = 16#6002; GL10_3200END_2 Digital input CH3-bit6.SubIndex = 23; GL10_3200END_2 Digital input CH3-bit6.Size = 1; GL10_3200END_2 Digital input CH3-bit6.Offset = 0; GL10_3200END_2 Digital input CH3-bit6.DependOnSlot = True; GL10_3200END_2 Digital input CH3-bit6.DependOnSlotGroup = True; GL10_3200END_2 Digital input CH3-bit7.Index = 16#6002; GL10_3200END_2 Digital input CH3-bit7.SubIndex = 24; GL10_3200END_2 Digital input CH3-bit7.Size = 1; GL10_3200END_2 Digital input CH3-bit7.Offset = 0; GL10_3200END_2 Digital input CH3-bit7.DependOnSlot = True; GL10_3200END_2 Digital input CH3-bit7.DependOnSlotGroup = True; GL10_3200END_2 Digital input CH4-bit0.Index = 16#6002; GL10_3200END_2 Digital input CH4-bit0.SubIndex = 25; GL10_3200END_2 Digital input CH4-bit0.Size = 1; GL10_3200END_2 Digital input CH4-bit0.Offset = 0; GL10_3200END_2 Digital input CH4-bit0.DependOnSlot = True; GL10_3200END_2 Digital input CH4-bit0.DependOnSlotGroup = True; GL10_3200END_2 Digital input CH4-bit1.Index = 16#6002; GL10_3200END_2 Digital input CH4-bit1.SubIndex = 26; GL10_3200END_2 Digital input CH4-bit1.Size = 1; GL10_3200END_2 Digital input CH4-bit1.Offset = 0; GL10_3200END_2 Digital input CH4-bit1.DependOnSlot = True; GL10_3200END_2 Digital input CH4-bit1.DependOnSlotGroup = True; GL10_3200END_2 Digital input CH4-bit2.Index = 16#6002; GL10_3200END_2 Digital input CH4-bit2.SubIndex = 27; GL10_3200END_2 Digital input CH4-bit2.Size = 1; GL10_3200END_2 Digital input CH4-bit2.Offset = 0; GL10_3200END_2 Digital input CH4-bit2.DependOnSlot = True; GL10_3200END_2 Digital input CH4-bit2.DependOnSlotGroup = True; GL10_3200END_2 Digital input CH4-bit3.Index = 16#6002;
            GL10_3200END_2 Digital input CH4-bit3.SubIndex = 28; GL10_3200END_2 Digital input CH4-bit3.Size = 1; GL10_3200END_2 Digital input CH4-bit3.Offset = 0; GL10_3200END_2 Digital input CH4-bit3.DependOnSlot = True; GL10_3200END_2 Digital input CH4-bit3.DependOnSlotGroup = True; GL10_3200END_2 Digital input CH4-bit4.Index = 16#6002; GL10_3200END_2 Digital input CH4-bit4.SubIndex = 29; GL10_3200END_2 Digital input CH4-bit4.Size = 1; GL10_3200END_2 Digital input CH4-bit4.Offset = 0; GL10_3200END_2 Digital input CH4-bit4.DependOnSlot = True; GL10_3200END_2 Digital input CH4-bit4.DependOnSlotGroup = True; GL10_3200END_2 Digital input CH4-bit5.Index = 16#6002; GL10_3200END_2 Digital input CH4-bit5.SubIndex = 30; GL10_3200END_2 Digital input CH4-bit5.Size = 1; GL10_3200END_2 Digital input CH4-bit5.Offset = 0; GL10_3200END_2 Digital input CH4-bit5.DependOnSlot = True; GL10_3200END_2 Digital input CH4-bit5.DependOnSlotGroup = True; GL10_3200END_2 Digital input CH4-bit6.Index = 16#6002; GL10_3200END_2 Digital input CH4-bit6.SubIndex = 31; GL10_3200END_2 Digital input CH4-bit6.Size = 1; GL10_3200END_2 Digital input CH4-bit6.Offset = 0; GL10_3200END_2 Digital input CH4-bit6.DependOnSlot = True; GL10_3200END_2 Digital input CH4-bit6.DependOnSlotGroup = True; GL10_3200END_2 Digital input CH4-bit7.Index = 16#6002; GL10_3200END_2 Digital input CH4-bit7.SubIndex = 32; GL10_3200END_2 Digital input CH4-bit7.Size = 1; GL10_3200END_2 Digital input CH4-bit7.Offset = 0; GL10_3200END_2 Digital input CH4-bit7.DependOnSlot = True; GL10_3200END_2 Digital input CH4-bit7.DependOnSlotGroup = True; RxTxPdo.NumberofExcludes = 1; RxTxPdo.NumberofEntries = 4; RxTxPdo.Index = 16#1A10; RxTxPdo.Fixed = True; RxTxPdo.Mandatory = False; RxTxPdo.Virtual = False; RxTxPdo.Sm = 3; RxTxPdo.Su = 0; RxTxPdo.Name = '3200END Input maping'; RxTxPdo.DependOnSlot = True; RxTxPdo.DependOnSlotGroup = False;
            RxTxPdo.OverwrittenByModule = True; Exclude = 16#1A14; GL10_3200END_3 Digital input CH1-8bit.Index = 16#6101; GL10_3200END_3 Digital input CH1-8bit.SubIndex = 1; GL10_3200END_3 Digital input CH1-8bit.Size = 8; GL10_3200END_3 Digital input CH1-8bit.Offset = 0; GL10_3200END_3 Digital input CH1-8bit.DependOnSlot = True; GL10_3200END_3 Digital input CH1-8bit.DependOnSlotGroup = True; GL10_3200END_3 Digital input CH2-8bit.Index = 16#6101; GL10_3200END_3 Digital input CH2-8bit.SubIndex = 2; GL10_3200END_3 Digital input CH2-8bit.Size = 8; GL10_3200END_3 Digital input CH2-8bit.Offset = 0; GL10_3200END_3 Digital input CH2-8bit.DependOnSlot = True; GL10_3200END_3 Digital input CH2-8bit.DependOnSlotGroup = True; GL10_3200END_3 Digital input CH3-8bit.Index = 16#6101; GL10_3200END_3 Digital input CH3-8bit.SubIndex = 3; GL10_3200END_3 Digital input CH3-8bit.Size = 8; GL10_3200END_3 Digital input CH3-8bit.Offset = 0; GL10_3200END_3 Digital input CH3-8bit.DependOnSlot = True; GL10_3200END_3 Digital input CH3-8bit.DependOnSlotGroup = True; GL10_3200END_3 Digital input CH4-8bit.Index = 16#6101; GL10_3200END_3 Digital input CH4-8bit.SubIndex = 4; GL10_3200END_3 Digital input CH4-8bit.Size = 8; GL10_3200END_3 Digital input CH4-8bit.Offset = 0; GL10_3200END_3 Digital input CH4-8bit.DependOnSlot = True; GL10_3200END_3 Digital input CH4-8bit.DependOnSlotGroup = True; RxTxPdo.NumberofExcludes = 1; RxTxPdo.NumberofEntries = 32; RxTxPdo.Index = 16#1A14; RxTxPdo.Fixed = True; RxTxPdo.Mandatory = False; RxTxPdo.Virtual = False; RxTxPdo.Sm = -1; RxTxPdo.Su = 0; RxTxPdo.Name = '3200END Input maping'; RxTxPdo.DependOnSlot = True; RxTxPdo.DependOnSlotGroup = False; RxTxPdo.OverwrittenByModule = True; Exclude = 16#1A10; GL10_3200END_3 Digital input CH1-bit0.Index = 16#6102;
            GL10_3200END_3 Digital input CH1-bit0.SubIndex = 1; GL10_3200END_3 Digital input CH1-bit0.Size = 1; GL10_3200END_3 Digital input CH1-bit0.Offset = 0; GL10_3200END_3 Digital input CH1-bit0.DependOnSlot = True; GL10_3200END_3 Digital input CH1-bit0.DependOnSlotGroup = True; GL10_3200END_3 Digital input CH1-bit1.Index = 16#6102; GL10_3200END_3 Digital input CH1-bit1.SubIndex = 2; GL10_3200END_3 Digital input CH1-bit1.Size = 1; GL10_3200END_3 Digital input CH1-bit1.Offset = 0; GL10_3200END_3 Digital input CH1-bit1.DependOnSlot = True; GL10_3200END_3 Digital input CH1-bit1.DependOnSlotGroup = True; GL10_3200END_3 Digital input CH1-bit2.Index = 16#6102; GL10_3200END_3 Digital input CH1-bit2.SubIndex = 3; GL10_3200END_3 Digital input CH1-bit2.Size = 1; GL10_3200END_3 Digital input CH1-bit2.Offset = 0; GL10_3200END_3 Digital input CH1-bit2.DependOnSlot = True; GL10_3200END_3 Digital input CH1-bit2.DependOnSlotGroup = True; GL10_3200END_3 Digital input CH1-bit3.Index = 16#6102; GL10_3200END_3 Digital input CH1-bit3.SubIndex = 4; GL10_3200END_3 Digital input CH1-bit3.Size = 1; GL10_3200END_3 Digital input CH1-bit3.Offset = 0; GL10_3200END_3 Digital input CH1-bit3.DependOnSlot = True; GL10_3200END_3 Digital input CH1-bit3.DependOnSlotGroup = True; GL10_3200END_3 Digital input CH1-bit4.Index = 16#6102; GL10_3200END_3 Digital input CH1-bit4.SubIndex = 5; GL10_3200END_3 Digital input CH1-bit4.Size = 1; GL10_3200END_3 Digital input CH1-bit4.Offset = 0; GL10_3200END_3 Digital input CH1-bit4.DependOnSlot = True; GL10_3200END_3 Digital input CH1-bit4.DependOnSlotGroup = True; GL10_3200END_3 Digital input CH1-bit5.Index = 16#6102; GL10_3200END_3 Digital input CH1-bit5.SubIndex = 6; GL10_3200END_3 Digital input CH1-bit5.Size = 1; GL10_3200END_3 Digital input CH1-bit5.Offset = 0; GL10_3200END_3 Digital input CH1-bit5.DependOnSlot = True; GL10_3200END_3 Digital input CH1-bit5.DependOnSlotGroup = True; GL10_3200END_3 Digital input CH1-bit6.Index = 16#6102; GL10_3200END_3 Digital input CH1-bit6.SubIndex = 7; GL10_3200END_3 Digital input CH1-bit6.Size = 1; GL10_3200END_3 Digital input CH1-bit6.Offset = 0; GL10_3200END_3 Digital input CH1-bit6.DependOnSlot = True;
            GL10_3200END_3 Digital input CH1-bit6.DependOnSlotGroup = True; GL10_3200END_3 Digital input CH1-bit7.Index = 16#6102; GL10_3200END_3 Digital input CH1-bit7.SubIndex = 8; GL10_3200END_3 Digital input CH1-bit7.Size = 1; GL10_3200END_3 Digital input CH1-bit7.Offset = 0; GL10_3200END_3 Digital input CH1-bit7.DependOnSlot = True; GL10_3200END_3 Digital input CH1-bit7.DependOnSlotGroup = True; GL10_3200END_3 Digital input CH2-bit0.Index = 16#6102; GL10_3200END_3 Digital input CH2-bit0.SubIndex = 9; GL10_3200END_3 Digital input CH2-bit0.Size = 1; GL10_3200END_3 Digital input CH2-bit0.Offset = 0; GL10_3200END_3 Digital input CH2-bit0.DependOnSlot = True; GL10_3200END_3 Digital input CH2-bit0.DependOnSlotGroup = True; GL10_3200END_3 Digital input CH2-bit1.Index = 16#6102; GL10_3200END_3 Digital input CH2-bit1.SubIndex = 10; GL10_3200END_3 Digital input CH2-bit1.Size = 1; GL10_3200END_3 Digital input CH2-bit1.Offset = 0; GL10_3200END_3 Digital input CH2-bit1.DependOnSlot = True; GL10_3200END_3 Digital input CH2-bit1.DependOnSlotGroup = True; GL10_3200END_3 Digital input CH2-bit2.Index = 16#6102; GL10_3200END_3 Digital input CH2-bit2.SubIndex = 11; GL10_3200END_3 Digital input CH2-bit2.Size = 1; GL10_3200END_3 Digital input CH2-bit2.Offset = 0; GL10_3200END_3 Digital input CH2-bit2.DependOnSlot = True; GL10_3200END_3 Digital input CH2-bit2.DependOnSlotGroup = True; GL10_3200END_3 Digital input CH2-bit3.Index = 16#6102; GL10_3200END_3 Digital input CH2-bit3.SubIndex = 12; GL10_3200END_3 Digital input CH2-bit3.Size = 1; GL10_3200END_3 Digital input CH2-bit3.Offset = 0; GL10_3200END_3 Digital input CH2-bit3.DependOnSlot = True; GL10_3200END_3 Digital input CH2-bit3.DependOnSlotGroup = True; GL10_3200END_3 Digital input CH2-bit4.Index = 16#6102; GL10_3200END_3 Digital input CH2-bit4.SubIndex = 13; GL10_3200END_3 Digital input CH2-bit4.Size = 1; GL10_3200END_3 Digital input CH2-bit4.Offset = 0; GL10_3200END_3 Digital input CH2-bit4.DependOnSlot = True; GL10_3200END_3 Digital input CH2-bit4.DependOnSlotGroup = True; GL10_3200END_3 Digital input CH2-bit5.Index = 16#6102; GL10_3200END_3 Digital input CH2-bit5.SubIndex = 14; GL10_3200END_3 Digital input CH2-bit5.Size = 1;
            GL10_3200END_3 Digital input CH2-bit5.Offset = 0; GL10_3200END_3 Digital input CH2-bit5.DependOnSlot = True; GL10_3200END_3 Digital input CH2-bit5.DependOnSlotGroup = True; GL10_3200END_3 Digital input CH2-bit6.Index = 16#6102; GL10_3200END_3 Digital input CH2-bit6.SubIndex = 15; GL10_3200END_3 Digital input CH2-bit6.Size = 1; GL10_3200END_3 Digital input CH2-bit6.Offset = 0; GL10_3200END_3 Digital input CH2-bit6.DependOnSlot = True; GL10_3200END_3 Digital input CH2-bit6.DependOnSlotGroup = True; GL10_3200END_3 Digital input CH2-bit7.Index = 16#6102; GL10_3200END_3 Digital input CH2-bit7.SubIndex = 16; GL10_3200END_3 Digital input CH2-bit7.Size = 1; GL10_3200END_3 Digital input CH2-bit7.Offset = 0; GL10_3200END_3 Digital input CH2-bit7.DependOnSlot = True; GL10_3200END_3 Digital input CH2-bit7.DependOnSlotGroup = True; GL10_3200END_3 Digital input CH3-bit0.Index = 16#6102; GL10_3200END_3 Digital input CH3-bit0.SubIndex = 17; GL10_3200END_3 Digital input CH3-bit0.Size = 1; GL10_3200END_3 Digital input CH3-bit0.Offset = 0; GL10_3200END_3 Digital input CH3-bit0.DependOnSlot = True; GL10_3200END_3 Digital input CH3-bit0.DependOnSlotGroup = True; GL10_3200END_3 Digital input CH3-bit1.Index = 16#6102; GL10_3200END_3 Digital input CH3-bit1.SubIndex = 18; GL10_3200END_3 Digital input CH3-bit1.Size = 1; GL10_3200END_3 Digital input CH3-bit1.Offset = 0; GL10_3200END_3 Digital input CH3-bit1.DependOnSlot = True; GL10_3200END_3 Digital input CH3-bit1.DependOnSlotGroup = True; GL10_3200END_3 Digital input CH3-bit2.Index = 16#6102; GL10_3200END_3 Digital input CH3-bit2.SubIndex = 19; GL10_3200END_3 Digital input CH3-bit2.Size = 1; GL10_3200END_3 Digital input CH3-bit2.Offset = 0; GL10_3200END_3 Digital input CH3-bit2.DependOnSlot = True; GL10_3200END_3 Digital input CH3-bit2.DependOnSlotGroup = True; GL10_3200END_3 Digital input CH3-bit3.Index = 16#6102; GL10_3200END_3 Digital input CH3-bit3.SubIndex = 20; GL10_3200END_3 Digital input CH3-bit3.Size = 1; GL10_3200END_3 Digital input CH3-bit3.Offset = 0; GL10_3200END_3 Digital input CH3-bit3.DependOnSlot = True; GL10_3200END_3 Digital input CH3-bit3.DependOnSlotGroup = True; GL10_3200END_3 Digital input CH3-bit4.Index = 16#6102;
            GL10_3200END_3 Digital input CH3-bit4.SubIndex = 21; GL10_3200END_3 Digital input CH3-bit4.Size = 1; GL10_3200END_3 Digital input CH3-bit4.Offset = 0; GL10_3200END_3 Digital input CH3-bit4.DependOnSlot = True; GL10_3200END_3 Digital input CH3-bit4.DependOnSlotGroup = True; GL10_3200END_3 Digital input CH3-bit5.Index = 16#6102; GL10_3200END_3 Digital input CH3-bit5.SubIndex = 22; GL10_3200END_3 Digital input CH3-bit5.Size = 1; GL10_3200END_3 Digital input CH3-bit5.Offset = 0; GL10_3200END_3 Digital input CH3-bit5.DependOnSlot = True; GL10_3200END_3 Digital input CH3-bit5.DependOnSlotGroup = True; GL10_3200END_3 Digital input CH3-bit6.Index = 16#6102; GL10_3200END_3 Digital input CH3-bit6.SubIndex = 23; GL10_3200END_3 Digital input CH3-bit6.Size = 1; GL10_3200END_3 Digital input CH3-bit6.Offset = 0; GL10_3200END_3 Digital input CH3-bit6.DependOnSlot = True; GL10_3200END_3 Digital input CH3-bit6.DependOnSlotGroup = True; GL10_3200END_3 Digital input CH3-bit7.Index = 16#6102; GL10_3200END_3 Digital input CH3-bit7.SubIndex = 24; GL10_3200END_3 Digital input CH3-bit7.Size = 1; GL10_3200END_3 Digital input CH3-bit7.Offset = 0; GL10_3200END_3 Digital input CH3-bit7.DependOnSlot = True; GL10_3200END_3 Digital input CH3-bit7.DependOnSlotGroup = True; GL10_3200END_3 Digital input CH4-bit0.Index = 16#6102; GL10_3200END_3 Digital input CH4-bit0.SubIndex = 25; GL10_3200END_3 Digital input CH4-bit0.Size = 1; GL10_3200END_3 Digital input CH4-bit0.Offset = 0; GL10_3200END_3 Digital input CH4-bit0.DependOnSlot = True; GL10_3200END_3 Digital input CH4-bit0.DependOnSlotGroup = True; GL10_3200END_3 Digital input CH4-bit1.Index = 16#6102; GL10_3200END_3 Digital input CH4-bit1.SubIndex = 26; GL10_3200END_3 Digital input CH4-bit1.Size = 1; GL10_3200END_3 Digital input CH4-bit1.Offset = 0; GL10_3200END_3 Digital input CH4-bit1.DependOnSlot = True; GL10_3200END_3 Digital input CH4-bit1.DependOnSlotGroup = True; GL10_3200END_3 Digital input CH4-bit2.Index = 16#6102; GL10_3200END_3 Digital input CH4-bit2.SubIndex = 27; GL10_3200END_3 Digital input CH4-bit2.Size = 1; GL10_3200END_3 Digital input CH4-bit2.Offset = 0; GL10_3200END_3 Digital input CH4-bit2.DependOnSlot = True;
            GL10_3200END_3 Digital input CH4-bit2.DependOnSlotGroup = True; GL10_3200END_3 Digital input CH4-bit3.Index = 16#6102; GL10_3200END_3 Digital input CH4-bit3.SubIndex = 28; GL10_3200END_3 Digital input CH4-bit3.Size = 1; GL10_3200END_3 Digital input CH4-bit3.Offset = 0; GL10_3200END_3 Digital input CH4-bit3.DependOnSlot = True; GL10_3200END_3 Digital input CH4-bit3.DependOnSlotGroup = True; GL10_3200END_3 Digital input CH4-bit4.Index = 16#6102; GL10_3200END_3 Digital input CH4-bit4.SubIndex = 29; GL10_3200END_3 Digital input CH4-bit4.Size = 1; GL10_3200END_3 Digital input CH4-bit4.Offset = 0; GL10_3200END_3 Digital input CH4-bit4.DependOnSlot = True; GL10_3200END_3 Digital input CH4-bit4.DependOnSlotGroup = True; GL10_3200END_3 Digital input CH4-bit5.Index = 16#6102; GL10_3200END_3 Digital input CH4-bit5.SubIndex = 30; GL10_3200END_3 Digital input CH4-bit5.Size = 1; GL10_3200END_3 Digital input CH4-bit5.Offset = 0; GL10_3200END_3 Digital input CH4-bit5.DependOnSlot = True; GL10_3200END_3 Digital input CH4-bit5.DependOnSlotGroup = True; GL10_3200END_3 Digital input CH4-bit6.Index = 16#6102; GL10_3200END_3 Digital input CH4-bit6.SubIndex = 31; GL10_3200END_3 Digital input CH4-bit6.Size = 1; GL10_3200END_3 Digital input CH4-bit6.Offset = 0; GL10_3200END_3 Digital input CH4-bit6.DependOnSlot = True; GL10_3200END_3 Digital input CH4-bit6.DependOnSlotGroup = True; GL10_3200END_3 Digital input CH4-bit7.Index = 16#6102; GL10_3200END_3 Digital input CH4-bit7.SubIndex = 32; GL10_3200END_3 Digital input CH4-bit7.Size = 1; GL10_3200END_3 Digital input CH4-bit7.Offset = 0; GL10_3200END_3 Digital input CH4-bit7.DependOnSlot = True; GL10_3200END_3 Digital input CH4-bit7.DependOnSlotGroup = True; Device control.Name = 'Device control'; Device control.DataType = 'UINT'; Device control.Default = ''; Device control.Comment = ''; GL10_0016ETN_1 Digital output CH1-8bit.Name = 'GL10_0016ETN_1 Digital output CH1-8bit'; GL10_0016ETN_1 Digital output CH1-8bit.DataType = 'USINT'; GL10_0016ETN_1 Digital output CH1-8bit.Default = ''; GL10_0016ETN_1 Digital output CH1-8bit.Comment = ''; GL10_0016ETN_1 Digital output CH2-8bit.Name = 'GL10_0016ETN_1 Digital output CH2-8bit';
            GL10_0016ETN_1 Digital output CH2-8bit.DataType = 'USINT'; GL10_0016ETN_1 Digital output CH2-8bit.Default = ''; GL10_0016ETN_1 Digital output CH2-8bit.Comment = ''; GL10_0016ETN_1 Digital output CH1-bit0.Name = 'GL10_0016ETN_1 Digital output CH1-bit0'; GL10_0016ETN_1 Digital output CH1-bit0.DataType = 'BOOL'; GL10_0016ETN_1 Digital output CH1-bit0.Default = ''; GL10_0016ETN_1 Digital output CH1-bit0.Comment = ''; GL10_0016ETN_1 Digital output CH1-bit1.Name = 'GL10_0016ETN_1 Digital output CH1-bit1'; GL10_0016ETN_1 Digital output CH1-bit1.DataType = 'BOOL'; GL10_0016ETN_1 Digital output CH1-bit1.Default = ''; GL10_0016ETN_1 Digital output CH1-bit1.Comment = ''; GL10_0016ETN_1 Digital output CH1-bit2.Name = 'GL10_0016ETN_1 Digital output CH1-bit2'; GL10_0016ETN_1 Digital output CH1-bit2.DataType = 'BOOL'; GL10_0016ETN_1 Digital output CH1-bit2.Default = ''; GL10_0016ETN_1 Digital output CH1-bit2.Comment = ''; GL10_0016ETN_1 Digital output CH1-bit3.Name = 'GL10_0016ETN_1 Digital output CH1-bit3'; GL10_0016ETN_1 Digital output CH1-bit3.DataType = 'BOOL'; GL10_0016ETN_1 Digital output CH1-bit3.Default = ''; GL10_0016ETN_1 Digital output CH1-bit3.Comment = ''; GL10_0016ETN_1 Digital output CH1-bit4.Name = 'GL10_0016ETN_1 Digital output CH1-bit4'; GL10_0016ETN_1 Digital output CH1-bit4.DataType = 'BOOL'; GL10_0016ETN_1 Digital output CH1-bit4.Default = ''; GL10_0016ETN_1 Digital output CH1-bit4.Comment = ''; GL10_0016ETN_1 Digital output CH1-bit5.Name = 'GL10_0016ETN_1 Digital output CH1-bit5'; GL10_0016ETN_1 Digital output CH1-bit5.DataType = 'BOOL'; GL10_0016ETN_1 Digital output CH1-bit5.Default = ''; GL10_0016ETN_1 Digital output CH1-bit5.Comment = ''; GL10_0016ETN_1 Digital output CH1-bit6.Name = 'GL10_0016ETN_1 Digital output CH1-bit6'; GL10_0016ETN_1 Digital output CH1-bit6.DataType = 'BOOL'; GL10_0016ETN_1 Digital output CH1-bit6.Default = ''; GL10_0016ETN_1 Digital output CH1-bit6.Comment = ''; GL10_0016ETN_1 Digital output CH1-bit7.Name = 'GL10_0016ETN_1 Digital output CH1-bit7'; GL10_0016ETN_1 Digital output CH1-bit7.DataType = 'BOOL'; GL10_0016ETN_1 Digital output CH1-bit7.Default = ''; GL10_0016ETN_1 Digital output CH1-bit7.Comment = ''; GL10_0016ETN_1 Digital output CH2-bit0.Name = 'GL10_0016ETN_1 Digital output CH2-bit0'; GL10_0016ETN_1 Digital output CH2-bit0.DataType = 'BOOL'; GL10_0016ETN_1 Digital output CH2-bit0.Default = ''; GL10_0016ETN_1 Digital output CH2-bit0.Comment = ''; GL10_0016ETN_1 Digital output CH2-bit1.Name = 'GL10_0016ETN_1 Digital output CH2-bit1';
            GL10_0016ETN_1 Digital output CH2-bit1.DataType = 'BOOL'; GL10_0016ETN_1 Digital output CH2-bit1.Default = ''; GL10_0016ETN_1 Digital output CH2-bit1.Comment = ''; GL10_0016ETN_1 Digital output CH2-bit2.Name = 'GL10_0016ETN_1 Digital output CH2-bit2'; GL10_0016ETN_1 Digital output CH2-bit2.DataType = 'BOOL'; GL10_0016ETN_1 Digital output CH2-bit2.Default = ''; GL10_0016ETN_1 Digital output CH2-bit2.Comment = ''; GL10_0016ETN_1 Digital output CH2-bit3.Name = 'GL10_0016ETN_1 Digital output CH2-bit3'; GL10_0016ETN_1 Digital output CH2-bit3.DataType = 'BOOL'; GL10_0016ETN_1 Digital output CH2-bit3.Default = ''; GL10_0016ETN_1 Digital output CH2-bit3.Comment = ''; GL10_0016ETN_1 Digital output CH2-bit4.Name = 'GL10_0016ETN_1 Digital output CH2-bit4'; GL10_0016ETN_1 Digital output CH2-bit4.DataType = 'BOOL'; GL10_0016ETN_1 Digital output CH2-bit4.Default = ''; GL10_0016ETN_1 Digital output CH2-bit4.Comment = ''; GL10_0016ETN_1 Digital output CH2-bit5.Name = 'GL10_0016ETN_1 Digital output CH2-bit5'; GL10_0016ETN_1 Digital output CH2-bit5.DataType = 'BOOL'; GL10_0016ETN_1 Digital output CH2-bit5.Default = ''; GL10_0016ETN_1 Digital output CH2-bit5.Comment = ''; GL10_0016ETN_1 Digital output CH2-bit6.Name = 'GL10_0016ETN_1 Digital output CH2-bit6'; GL10_0016ETN_1 Digital output CH2-bit6.DataType = 'BOOL'; GL10_0016ETN_1 Digital output CH2-bit6.Default = ''; GL10_0016ETN_1 Digital output CH2-bit6.Comment = ''; GL10_0016ETN_1 Digital output CH2-bit7.Name = 'GL10_0016ETN_1 Digital output CH2-bit7'; GL10_0016ETN_1 Digital output CH2-bit7.DataType = 'BOOL'; GL10_0016ETN_1 Digital output CH2-bit7.Default = ''; GL10_0016ETN_1 Digital output CH2-bit7.Comment = ''; GL10_0016ETN_1 DO module output mode after EtherCAT lost link.Name = 'GL10_0016ETN_1 DO module output mode after EtherCAT lost link'; GL10_0016ETN_1 DO module output mode after EtherCAT lost link.DataType = 'UINT'; GL10_0016ETN_1 DO module output mode after EtherCAT lost link.Default = ''; GL10_0016ETN_1 DO module output mode after EtherCAT lost link.Comment = ''; GL10_0016ETN_1 DO module output value after EtherCAT lost link.Name = 'GL10_0016ETN_1 DO module output value after EtherCAT lost link'; GL10_0016ETN_1 DO module output value after EtherCAT lost link.DataType = 'UINT'; GL10_0016ETN_1 DO module output value after EtherCAT lost link.Default = ''; GL10_0016ETN_1 DO module output value after EtherCAT lost link.Comment = ''; Device status.Name = 'Device status'; Device status.DataType = 'UINT'; Device status.Default = ''; Device status.Comment = ''; GL10_3200END_2 Digital input CH1-8bit.Name = 'GL10_3200END_2 Digital input CH1-8bit';
            GL10_3200END_2 Digital input CH1-8bit.DataType = 'USINT'; GL10_3200END_2 Digital input CH1-8bit.Default = ''; GL10_3200END_2 Digital input CH1-8bit.Comment = ''; GL10_3200END_2 Digital input CH2-8bit.Name = 'GL10_3200END_2 Digital input CH2-8bit'; GL10_3200END_2 Digital input CH2-8bit.DataType = 'USINT'; GL10_3200END_2 Digital input CH2-8bit.Default = ''; GL10_3200END_2 Digital input CH2-8bit.Comment = ''; GL10_3200END_2 Digital input CH3-8bit.Name = 'GL10_3200END_2 Digital input CH3-8bit'; GL10_3200END_2 Digital input CH3-8bit.DataType = 'USINT'; GL10_3200END_2 Digital input CH3-8bit.Default = ''; GL10_3200END_2 Digital input CH3-8bit.Comment = ''; GL10_3200END_2 Digital input CH4-8bit.Name = 'GL10_3200END_2 Digital input CH4-8bit'; GL10_3200END_2 Digital input CH4-8bit.DataType = 'USINT'; GL10_3200END_2 Digital input CH4-8bit.Default = ''; GL10_3200END_2 Digital input CH4-8bit.Comment = ''; GL10_3200END_2 Digital input CH1-bit0.Name = 'GL10_3200END_2 Digital input CH1-bit0'; GL10_3200END_2 Digital input CH1-bit0.DataType = 'BOOL'; GL10_3200END_2 Digital input CH1-bit0.Default = ''; GL10_3200END_2 Digital input CH1-bit0.Comment = ''; GL10_3200END_2 Digital input CH1-bit1.Name = 'GL10_3200END_2 Digital input CH1-bit1'; GL10_3200END_2 Digital input CH1-bit1.DataType = 'BOOL'; GL10_3200END_2 Digital input CH1-bit1.Default = ''; GL10_3200END_2 Digital input CH1-bit1.Comment = ''; GL10_3200END_2 Digital input CH1-bit2.Name = 'GL10_3200END_2 Digital input CH1-bit2'; GL10_3200END_2 Digital input CH1-bit2.DataType = 'BOOL'; GL10_3200END_2 Digital input CH1-bit2.Default = ''; GL10_3200END_2 Digital input CH1-bit2.Comment = ''; GL10_3200END_2 Digital input CH1-bit3.Name = 'GL10_3200END_2 Digital input CH1-bit3'; GL10_3200END_2 Digital input CH1-bit3.DataType = 'BOOL'; GL10_3200END_2 Digital input CH1-bit3.Default = ''; GL10_3200END_2 Digital input CH1-bit3.Comment = ''; GL10_3200END_2 Digital input CH1-bit4.Name = 'GL10_3200END_2 Digital input CH1-bit4'; GL10_3200END_2 Digital input CH1-bit4.DataType = 'BOOL'; GL10_3200END_2 Digital input CH1-bit4.Default = ''; GL10_3200END_2 Digital input CH1-bit4.Comment = ''; GL10_3200END_2 Digital input CH1-bit5.Name = 'GL10_3200END_2 Digital input CH1-bit5'; GL10_3200END_2 Digital input CH1-bit5.DataType = 'BOOL'; GL10_3200END_2 Digital input CH1-bit5.Default = ''; GL10_3200END_2 Digital input CH1-bit5.Comment = ''; GL10_3200END_2 Digital input CH1-bit6.Name = 'GL10_3200END_2 Digital input CH1-bit6';
            GL10_3200END_2 Digital input CH1-bit6.DataType = 'BOOL'; GL10_3200END_2 Digital input CH1-bit6.Default = ''; GL10_3200END_2 Digital input CH1-bit6.Comment = ''; GL10_3200END_2 Digital input CH1-bit7.Name = 'GL10_3200END_2 Digital input CH1-bit7'; GL10_3200END_2 Digital input CH1-bit7.DataType = 'BOOL'; GL10_3200END_2 Digital input CH1-bit7.Default = ''; GL10_3200END_2 Digital input CH1-bit7.Comment = ''; GL10_3200END_2 Digital input CH2-bit0.Name = 'GL10_3200END_2 Digital input CH2-bit0'; GL10_3200END_2 Digital input CH2-bit0.DataType = 'BOOL'; GL10_3200END_2 Digital input CH2-bit0.Default = ''; GL10_3200END_2 Digital input CH2-bit0.Comment = ''; GL10_3200END_2 Digital input CH2-bit1.Name = 'GL10_3200END_2 Digital input CH2-bit1'; GL10_3200END_2 Digital input CH2-bit1.DataType = 'BOOL'; GL10_3200END_2 Digital input CH2-bit1.Default = ''; GL10_3200END_2 Digital input CH2-bit1.Comment = ''; GL10_3200END_2 Digital input CH2-bit2.Name = 'GL10_3200END_2 Digital input CH2-bit2'; GL10_3200END_2 Digital input CH2-bit2.DataType = 'BOOL'; GL10_3200END_2 Digital input CH2-bit2.Default = ''; GL10_3200END_2 Digital input CH2-bit2.Comment = ''; GL10_3200END_2 Digital input CH2-bit3.Name = 'GL10_3200END_2 Digital input CH2-bit3'; GL10_3200END_2 Digital input CH2-bit3.DataType = 'BOOL'; GL10_3200END_2 Digital input CH2-bit3.Default = ''; GL10_3200END_2 Digital input CH2-bit3.Comment = ''; GL10_3200END_2 Digital input CH2-bit4.Name = 'GL10_3200END_2 Digital input CH2-bit4'; GL10_3200END_2 Digital input CH2-bit4.DataType = 'BOOL'; GL10_3200END_2 Digital input CH2-bit4.Default = ''; GL10_3200END_2 Digital input CH2-bit4.Comment = ''; GL10_3200END_2 Digital input CH2-bit5.Name = 'GL10_3200END_2 Digital input CH2-bit5'; GL10_3200END_2 Digital input CH2-bit5.DataType = 'BOOL'; GL10_3200END_2 Digital input CH2-bit5.Default = ''; GL10_3200END_2 Digital input CH2-bit5.Comment = ''; GL10_3200END_2 Digital input CH2-bit6.Name = 'GL10_3200END_2 Digital input CH2-bit6'; GL10_3200END_2 Digital input CH2-bit6.DataType = 'BOOL'; GL10_3200END_2 Digital input CH2-bit6.Default = ''; GL10_3200END_2 Digital input CH2-bit6.Comment = ''; GL10_3200END_2 Digital input CH2-bit7.Name = 'GL10_3200END_2 Digital input CH2-bit7'; GL10_3200END_2 Digital input CH2-bit7.DataType = 'BOOL'; GL10_3200END_2 Digital input CH2-bit7.Default = ''; GL10_3200END_2 Digital input CH2-bit7.Comment = ''; GL10_3200END_2 Digital input CH3-bit0.Name = 'GL10_3200END_2 Digital input CH3-bit0';
            GL10_3200END_2 Digital input CH3-bit0.DataType = 'BOOL'; GL10_3200END_2 Digital input CH3-bit0.Default = ''; GL10_3200END_2 Digital input CH3-bit0.Comment = ''; GL10_3200END_2 Digital input CH3-bit1.Name = 'GL10_3200END_2 Digital input CH3-bit1'; GL10_3200END_2 Digital input CH3-bit1.DataType = 'BOOL'; GL10_3200END_2 Digital input CH3-bit1.Default = ''; GL10_3200END_2 Digital input CH3-bit1.Comment = ''; GL10_3200END_2 Digital input CH3-bit2.Name = 'GL10_3200END_2 Digital input CH3-bit2'; GL10_3200END_2 Digital input CH3-bit2.DataType = 'BOOL'; GL10_3200END_2 Digital input CH3-bit2.Default = ''; GL10_3200END_2 Digital input CH3-bit2.Comment = ''; GL10_3200END_2 Digital input CH3-bit3.Name = 'GL10_3200END_2 Digital input CH3-bit3'; GL10_3200END_2 Digital input CH3-bit3.DataType = 'BOOL'; GL10_3200END_2 Digital input CH3-bit3.Default = ''; GL10_3200END_2 Digital input CH3-bit3.Comment = ''; GL10_3200END_2 Digital input CH3-bit4.Name = 'GL10_3200END_2 Digital input CH3-bit4'; GL10_3200END_2 Digital input CH3-bit4.DataType = 'BOOL'; GL10_3200END_2 Digital input CH3-bit4.Default = ''; GL10_3200END_2 Digital input CH3-bit4.Comment = ''; GL10_3200END_2 Digital input CH3-bit5.Name = 'GL10_3200END_2 Digital input CH3-bit5'; GL10_3200END_2 Digital input CH3-bit5.DataType = 'BOOL'; GL10_3200END_2 Digital input CH3-bit5.Default = ''; GL10_3200END_2 Digital input CH3-bit5.Comment = ''; GL10_3200END_2 Digital input CH3-bit6.Name = 'GL10_3200END_2 Digital input CH3-bit6'; GL10_3200END_2 Digital input CH3-bit6.DataType = 'BOOL'; GL10_3200END_2 Digital input CH3-bit6.Default = ''; GL10_3200END_2 Digital input CH3-bit6.Comment = ''; GL10_3200END_2 Digital input CH3-bit7.Name = 'GL10_3200END_2 Digital input CH3-bit7'; GL10_3200END_2 Digital input CH3-bit7.DataType = 'BOOL'; GL10_3200END_2 Digital input CH3-bit7.Default = ''; GL10_3200END_2 Digital input CH3-bit7.Comment = ''; GL10_3200END_2 Digital input CH4-bit0.Name = 'GL10_3200END_2 Digital input CH4-bit0'; GL10_3200END_2 Digital input CH4-bit0.DataType = 'BOOL'; GL10_3200END_2 Digital input CH4-bit0.Default = ''; GL10_3200END_2 Digital input CH4-bit0.Comment = ''; GL10_3200END_2 Digital input CH4-bit1.Name = 'GL10_3200END_2 Digital input CH4-bit1'; GL10_3200END_2 Digital input CH4-bit1.DataType = 'BOOL'; GL10_3200END_2 Digital input CH4-bit1.Default = ''; GL10_3200END_2 Digital input CH4-bit1.Comment = ''; GL10_3200END_2 Digital input CH4-bit2.Name = 'GL10_3200END_2 Digital input CH4-bit2';
            GL10_3200END_2 Digital input CH4-bit2.DataType = 'BOOL'; GL10_3200END_2 Digital input CH4-bit2.Default = ''; GL10_3200END_2 Digital input CH4-bit2.Comment = ''; GL10_3200END_2 Digital input CH4-bit3.Name = 'GL10_3200END_2 Digital input CH4-bit3'; GL10_3200END_2 Digital input CH4-bit3.DataType = 'BOOL'; GL10_3200END_2 Digital input CH4-bit3.Default = ''; GL10_3200END_2 Digital input CH4-bit3.Comment = ''; GL10_3200END_2 Digital input CH4-bit4.Name = 'GL10_3200END_2 Digital input CH4-bit4'; GL10_3200END_2 Digital input CH4-bit4.DataType = 'BOOL'; GL10_3200END_2 Digital input CH4-bit4.Default = ''; GL10_3200END_2 Digital input CH4-bit4.Comment = ''; GL10_3200END_2 Digital input CH4-bit5.Name = 'GL10_3200END_2 Digital input CH4-bit5'; GL10_3200END_2 Digital input CH4-bit5.DataType = 'BOOL'; GL10_3200END_2 Digital input CH4-bit5.Default = ''; GL10_3200END_2 Digital input CH4-bit5.Comment = ''; GL10_3200END_2 Digital input CH4-bit6.Name = 'GL10_3200END_2 Digital input CH4-bit6'; GL10_3200END_2 Digital input CH4-bit6.DataType = 'BOOL'; GL10_3200END_2 Digital input CH4-bit6.Default = ''; GL10_3200END_2 Digital input CH4-bit6.Comment = ''; GL10_3200END_2 Digital input CH4-bit7.Name = 'GL10_3200END_2 Digital input CH4-bit7'; GL10_3200END_2 Digital input CH4-bit7.DataType = 'BOOL'; GL10_3200END_2 Digital input CH4-bit7.Default = ''; GL10_3200END_2 Digital input CH4-bit7.Comment = ''; GL10_3200END_3 Digital input CH1-8bit.Name = 'GL10_3200END_3 Digital input CH1-8bit'; GL10_3200END_3 Digital input CH1-8bit.DataType = 'USINT'; GL10_3200END_3 Digital input CH1-8bit.Default = ''; GL10_3200END_3 Digital input CH1-8bit.Comment = ''; GL10_3200END_3 Digital input CH2-8bit.Name = 'GL10_3200END_3 Digital input CH2-8bit'; GL10_3200END_3 Digital input CH2-8bit.DataType = 'USINT'; GL10_3200END_3 Digital input CH2-8bit.Default = ''; GL10_3200END_3 Digital input CH2-8bit.Comment = ''; GL10_3200END_3 Digital input CH3-8bit.Name = 'GL10_3200END_3 Digital input CH3-8bit'; GL10_3200END_3 Digital input CH3-8bit.DataType = 'USINT'; GL10_3200END_3 Digital input CH3-8bit.Default = ''; GL10_3200END_3 Digital input CH3-8bit.Comment = ''; GL10_3200END_3 Digital input CH4-8bit.Name = 'GL10_3200END_3 Digital input CH4-8bit'; GL10_3200END_3 Digital input CH4-8bit.DataType = 'USINT'; GL10_3200END_3 Digital input CH4-8bit.Default = ''; GL10_3200END_3 Digital input CH4-8bit.Comment = ''; GL10_3200END_3 Digital input CH1-bit0.Name = 'GL10_3200END_3 Digital input CH1-bit0';
            GL10_3200END_3 Digital input CH1-bit0.DataType = 'BOOL'; GL10_3200END_3 Digital input CH1-bit0.Default = ''; GL10_3200END_3 Digital input CH1-bit0.Comment = ''; GL10_3200END_3 Digital input CH1-bit1.Name = 'GL10_3200END_3 Digital input CH1-bit1'; GL10_3200END_3 Digital input CH1-bit1.DataType = 'BOOL'; GL10_3200END_3 Digital input CH1-bit1.Default = ''; GL10_3200END_3 Digital input CH1-bit1.Comment = ''; GL10_3200END_3 Digital input CH1-bit2.Name = 'GL10_3200END_3 Digital input CH1-bit2'; GL10_3200END_3 Digital input CH1-bit2.DataType = 'BOOL'; GL10_3200END_3 Digital input CH1-bit2.Default = ''; GL10_3200END_3 Digital input CH1-bit2.Comment = ''; GL10_3200END_3 Digital input CH1-bit3.Name = 'GL10_3200END_3 Digital input CH1-bit3'; GL10_3200END_3 Digital input CH1-bit3.DataType = 'BOOL'; GL10_3200END_3 Digital input CH1-bit3.Default = ''; GL10_3200END_3 Digital input CH1-bit3.Comment = ''; GL10_3200END_3 Digital input CH1-bit4.Name = 'GL10_3200END_3 Digital input CH1-bit4'; GL10_3200END_3 Digital input CH1-bit4.DataType = 'BOOL'; GL10_3200END_3 Digital input CH1-bit4.Default = ''; GL10_3200END_3 Digital input CH1-bit4.Comment = ''; GL10_3200END_3 Digital input CH1-bit5.Name = 'GL10_3200END_3 Digital input CH1-bit5'; GL10_3200END_3 Digital input CH1-bit5.DataType = 'BOOL'; GL10_3200END_3 Digital input CH1-bit5.Default = ''; GL10_3200END_3 Digital input CH1-bit5.Comment = ''; GL10_3200END_3 Digital input CH1-bit6.Name = 'GL10_3200END_3 Digital input CH1-bit6'; GL10_3200END_3 Digital input CH1-bit6.DataType = 'BOOL'; GL10_3200END_3 Digital input CH1-bit6.Default = ''; GL10_3200END_3 Digital input CH1-bit6.Comment = ''; GL10_3200END_3 Digital input CH1-bit7.Name = 'GL10_3200END_3 Digital input CH1-bit7'; GL10_3200END_3 Digital input CH1-bit7.DataType = 'BOOL'; GL10_3200END_3 Digital input CH1-bit7.Default = ''; GL10_3200END_3 Digital input CH1-bit7.Comment = ''; GL10_3200END_3 Digital input CH2-bit0.Name = 'GL10_3200END_3 Digital input CH2-bit0'; GL10_3200END_3 Digital input CH2-bit0.DataType = 'BOOL'; GL10_3200END_3 Digital input CH2-bit0.Default = ''; GL10_3200END_3 Digital input CH2-bit0.Comment = ''; GL10_3200END_3 Digital input CH2-bit1.Name = 'GL10_3200END_3 Digital input CH2-bit1'; GL10_3200END_3 Digital input CH2-bit1.DataType = 'BOOL'; GL10_3200END_3 Digital input CH2-bit1.Default = ''; GL10_3200END_3 Digital input CH2-bit1.Comment = ''; GL10_3200END_3 Digital input CH2-bit2.Name = 'GL10_3200END_3 Digital input CH2-bit2';
            GL10_3200END_3 Digital input CH2-bit2.DataType = 'BOOL'; GL10_3200END_3 Digital input CH2-bit2.Default = ''; GL10_3200END_3 Digital input CH2-bit2.Comment = ''; GL10_3200END_3 Digital input CH2-bit3.Name = 'GL10_3200END_3 Digital input CH2-bit3'; GL10_3200END_3 Digital input CH2-bit3.DataType = 'BOOL'; GL10_3200END_3 Digital input CH2-bit3.Default = ''; GL10_3200END_3 Digital input CH2-bit3.Comment = ''; GL10_3200END_3 Digital input CH2-bit4.Name = 'GL10_3200END_3 Digital input CH2-bit4'; GL10_3200END_3 Digital input CH2-bit4.DataType = 'BOOL'; GL10_3200END_3 Digital input CH2-bit4.Default = ''; GL10_3200END_3 Digital input CH2-bit4.Comment = ''; GL10_3200END_3 Digital input CH2-bit5.Name = 'GL10_3200END_3 Digital input CH2-bit5'; GL10_3200END_3 Digital input CH2-bit5.DataType = 'BOOL'; GL10_3200END_3 Digital input CH2-bit5.Default = ''; GL10_3200END_3 Digital input CH2-bit5.Comment = ''; GL10_3200END_3 Digital input CH2-bit6.Name = 'GL10_3200END_3 Digital input CH2-bit6'; GL10_3200END_3 Digital input CH2-bit6.DataType = 'BOOL'; GL10_3200END_3 Digital input CH2-bit6.Default = ''; GL10_3200END_3 Digital input CH2-bit6.Comment = ''; GL10_3200END_3 Digital input CH2-bit7.Name = 'GL10_3200END_3 Digital input CH2-bit7'; GL10_3200END_3 Digital input CH2-bit7.DataType = 'BOOL'; GL10_3200END_3 Digital input CH2-bit7.Default = ''; GL10_3200END_3 Digital input CH2-bit7.Comment = ''; GL10_3200END_3 Digital input CH3-bit0.Name = 'GL10_3200END_3 Digital input CH3-bit0'; GL10_3200END_3 Digital input CH3-bit0.DataType = 'BOOL'; GL10_3200END_3 Digital input CH3-bit0.Default = ''; GL10_3200END_3 Digital input CH3-bit0.Comment = ''; GL10_3200END_3 Digital input CH3-bit1.Name = 'GL10_3200END_3 Digital input CH3-bit1'; GL10_3200END_3 Digital input CH3-bit1.DataType = 'BOOL'; GL10_3200END_3 Digital input CH3-bit1.Default = ''; GL10_3200END_3 Digital input CH3-bit1.Comment = ''; GL10_3200END_3 Digital input CH3-bit2.Name = 'GL10_3200END_3 Digital input CH3-bit2'; GL10_3200END_3 Digital input CH3-bit2.DataType = 'BOOL'; GL10_3200END_3 Digital input CH3-bit2.Default = ''; GL10_3200END_3 Digital input CH3-bit2.Comment = ''; GL10_3200END_3 Digital input CH3-bit3.Name = 'GL10_3200END_3 Digital input CH3-bit3'; GL10_3200END_3 Digital input CH3-bit3.DataType = 'BOOL'; GL10_3200END_3 Digital input CH3-bit3.Default = ''; GL10_3200END_3 Digital input CH3-bit3.Comment = ''; GL10_3200END_3 Digital input CH3-bit4.Name = 'GL10_3200END_3 Digital input CH3-bit4';
            GL10_3200END_3 Digital input CH3-bit4.DataType = 'BOOL'; GL10_3200END_3 Digital input CH3-bit4.Default = ''; GL10_3200END_3 Digital input CH3-bit4.Comment = ''; GL10_3200END_3 Digital input CH3-bit5.Name = 'GL10_3200END_3 Digital input CH3-bit5'; GL10_3200END_3 Digital input CH3-bit5.DataType = 'BOOL'; GL10_3200END_3 Digital input CH3-bit5.Default = ''; GL10_3200END_3 Digital input CH3-bit5.Comment = ''; GL10_3200END_3 Digital input CH3-bit6.Name = 'GL10_3200END_3 Digital input CH3-bit6'; GL10_3200END_3 Digital input CH3-bit6.DataType = 'BOOL'; GL10_3200END_3 Digital input CH3-bit6.Default = ''; GL10_3200END_3 Digital input CH3-bit6.Comment = ''; GL10_3200END_3 Digital input CH3-bit7.Name = 'GL10_3200END_3 Digital input CH3-bit7'; GL10_3200END_3 Digital input CH3-bit7.DataType = 'BOOL'; GL10_3200END_3 Digital input CH3-bit7.Default = ''; GL10_3200END_3 Digital input CH3-bit7.Comment = ''; GL10_3200END_3 Digital input CH4-bit0.Name = 'GL10_3200END_3 Digital input CH4-bit0'; GL10_3200END_3 Digital input CH4-bit0.DataType = 'BOOL'; GL10_3200END_3 Digital input CH4-bit0.Default = ''; GL10_3200END_3 Digital input CH4-bit0.Comment = ''; GL10_3200END_3 Digital input CH4-bit1.Name = 'GL10_3200END_3 Digital input CH4-bit1'; GL10_3200END_3 Digital input CH4-bit1.DataType = 'BOOL'; GL10_3200END_3 Digital input CH4-bit1.Default = ''; GL10_3200END_3 Digital input CH4-bit1.Comment = ''; GL10_3200END_3 Digital input CH4-bit2.Name = 'GL10_3200END_3 Digital input CH4-bit2'; GL10_3200END_3 Digital input CH4-bit2.DataType = 'BOOL'; GL10_3200END_3 Digital input CH4-bit2.Default = ''; GL10_3200END_3 Digital input CH4-bit2.Comment = ''; GL10_3200END_3 Digital input CH4-bit3.Name = 'GL10_3200END_3 Digital input CH4-bit3'; GL10_3200END_3 Digital input CH4-bit3.DataType = 'BOOL'; GL10_3200END_3 Digital input CH4-bit3.Default = ''; GL10_3200END_3 Digital input CH4-bit3.Comment = ''; GL10_3200END_3 Digital input CH4-bit4.Name = 'GL10_3200END_3 Digital input CH4-bit4'; GL10_3200END_3 Digital input CH4-bit4.DataType = 'BOOL'; GL10_3200END_3 Digital input CH4-bit4.Default = ''; GL10_3200END_3 Digital input CH4-bit4.Comment = ''; GL10_3200END_3 Digital input CH4-bit5.Name = 'GL10_3200END_3 Digital input CH4-bit5'; GL10_3200END_3 Digital input CH4-bit5.DataType = 'BOOL'; GL10_3200END_3 Digital input CH4-bit5.Default = ''; GL10_3200END_3 Digital input CH4-bit5.Comment = ''; GL10_3200END_3 Digital input CH4-bit6.Name = 'GL10_3200END_3 Digital input CH4-bit6';
            GL10_3200END_3 Digital input CH4-bit6.DataType = 'BOOL'; GL10_3200END_3 Digital input CH4-bit6.Default = ''; GL10_3200END_3 Digital input CH4-bit6.Comment = ''; GL10_3200END_3 Digital input CH4-bit7.Name = 'GL10_3200END_3 Digital input CH4-bit7'; GL10_3200END_3 Digital input CH4-bit7.DataType = 'BOOL'; GL10_3200END_3 Digital input CH4-bit7.Default = ''; GL10_3200END_3 Digital input CH4-bit7.Comment = ''
          unmapped channels: %QB2 GL10_0016ETN_1 Digital output CH1-8bit, %QB3 GL10_0016ETN_1 Digital output CH2-8bit, %IW214 Device status, %IB2 GL10_3200END_2 Digital input CH1-8bit, %IB3 GL10_3200END_2 Digital input CH2-8bit, %IB4 GL10_3200END_2 Digital input CH3-8bit, %IB5 GL10_3200END_2 Digital input CH4-8bit, %IB6 GL10_3200END_3 Digital input CH1-8bit, %IB7 GL10_3200END_3 Digital input CH2-8bit, %IB8 GL10_3200END_3 Digital input CH3-8bit, %IB9 GL10_3200END_3 Digital input CH4-8bit
        GL10_3200END_2 : AM600-3200END(32 channels DI Module), Inovance, order no. GL10-3200END, version 0
        GL10_3200END_3 : AM600-3200END(32 channels DI Module), Inovance, order no. GL10-3200END, version 0
        GL10_0016ETN_1 : AM600-0016XXX(16 channels DO module), Inovance, order no. GL10-0016XXX, version 0
    MODBUS_TCP : ModbusTCP Device, Inovance, version 00.00.00.10
        settings:  = 0
  SMElement/
    SM0_SM511
    SM512_SM1023
    SM1024_SM1535
    SM1536_SM2047
    SM2048_SM2559
    SM2560_SM3071
    SM3072_SM3583
    SM3584_SM4095
    SM4096_SM4607
    SM4608_SM5119
    SM5120_SM5631
    SM5632_SM6143
    SM6144_SM6655
    SM6656_SM7167
    SM7168_SM7679
    SM7680_SM8191
    SM8192_SM8703
    SM8704_SM9215
    SM9216_SM9727
    SM9728_SM9999
  SDElement/
    SD0_SD511
    SD512_SD1023
    SD1024_SD1535
    SD1536_SD2047
    SD2048_SD2559
    SD2560_SD3071
    SD3072_SD3583
    SD3584_SD4095
    SD4096_SD4607
    SD4608_SD5119
    SD5120_SD5631
    SD5632_SD6143
    SD6144_SD6655
    SD6656_SD7167
    SD7168_SD7679
    SD7680_SD8191
    SD8192_SD8703
    SD8704_SD9215
    SD9216_SD9727
    SD9728_SD9999
*)

// Device/Application/01_变量/PersistentVars
{attribute 'qualified_only'}
VAR_GLOBAL PERSISTENT RETAIN
END_VAR

// Device/Application/01_变量/GVL_FB
VAR_GLOBAL
	LnCylInit_A: FB_LineCylinderInit;
	LnCylInit_B: FB_LineCylinderInit;
	DockCylInitC: FB_CylinderInit;
	PickModInitA: FB_MaterialInit;
	PickModInitB: FB_MaterialInit;
	MainModInitC: FB_MainlineInit;
END_VAR

// Device/Application/01_变量/GVL_X
VAR_GLOBAL
X_MainEStopPB AT %IX9.7 :BOOL;
X_MatReqSig AT %IX9.2 :BOOL;
X_StartPB AT %IX9.4 :BOOL;
X_StopPB AT %IX9.5 :BOOL;
X_ResetPB AT %IX9.6 :BOOL;

X_ManAutoSw AT %IX9.3 :BOOL;	
X_MFrSafeDr AT %IX8.5 :BOOL;
X_MRrSafeDr AT %IX8.6 :BOOL;
X_MLftSafeDr AT %IX8.7 :BOOL;
X_MRgtSafeDr AT %IX9.0 :BOOL;

X_StpCyl_R_A1 AT %IX4.5 :BOOL;
X_StpCyl_W_A1 AT %IX4.4 :BOOL;
X_StpCyl_R_A2 AT %IX4.6 :BOOL;
X_StpCyl_W_A2 AT %IX4.7:BOOL;
X_StpCyl_R_A3 AT %IX5.3 :BOOL;
X_StpCyl_W_A3 AT %IX5.2 :BOOL;
X_StpCyl_R_A4 AT %IX6.2 :BOOL;
X_StpCyl_W_A4 AT %IX6.3 :BOOL;
X_StpCyl_R_A5 AT %IX6.5 :BOOL;
X_StpCyl_W_A5 AT %IX6.4 :BOOL;
X_LftCyl_R_A1 AT %IX5.0 :BOOL;
X_LftCyl_W_A1 AT %IX5.1 :BOOL;
X_LftCyl_R_A2 AT %IX5.6 :BOOL;
X_LftCyl_W_A2 AT %IX5.7 :BOOL;
X_LftCyl_R_A3 AT %IX6.1 :BOOL;
X_LftCyl_W_A3 AT %IX6.0 :BOOL;
X_LftCyl_R_A4 AT %IX6.6 :BOOL;
X_LftCyl_W_A4 AT %IX6.7 :BOOL;
X_TrnCyl_R_A1 AT %IX5.5 :BOOL;
X_TrnCyl_W_A1 AT %IX5.4 :BOOL;
X_ModASftC_R AT %IX2.0 :BOOL;
X_ModASftC_W AT %IX2.1 :BOOL;
X_ModAGrpC_R AT %IX2.5 :BOOL;
X_ModAGrpC_W AT %IX2.4 :BOOL;
X_ModARotC_R AT %IX2.3 :BOOL;
X_ModARotC_W AT %IX2.2 :BOOL;



X_StpCyl_R_C1 AT %IX7.3 :BOOL;
X_StpCyl_W_C1 AT %IX7.2 :BOOL;
X_LftCyl_R_C1 AT %IX7.1 :BOOL;
X_LftCyl_W_C1 AT %IX7.0 :BOOL;
X_ModCSftC_R AT %IX2.6 :BOOL;
X_ModCSftC_W AT %IX2.7 :BOOL;
X_MdCLftLC_R AT %IX3.0 :BOOL;
X_MdCLftLC_W AT %IX3.1 :BOOL;
X_MdCGrpLC_R AT %IX3.4 :BOOL;
X_MdCGrpLC_W AT %IX3.5 :BOOL;
X_MdCRotLC_R AT %IX3.2 :BOOL;
X_MdCRotLC_W AT %IX3.3 :BOOL;

X_FwdDet_A AT %IX7.4 :BOOL;
X_RevDet_A AT %IX7.5 :BOOL;
X_LftRotPosA AT %IX7.6 :BOOL;
X_PickPosDetA AT %IX7.7 :BOOL;
X_PlacePos_A AT %IX8.0 :BOOL;
X_PlaceFull_A AT %IX8.1 :BOOL;
X_BufPos_A AT %IX8.2 :BOOL;
X_BufFull_A AT %IX8.3 :BOOL;
X_WaitPos_A AT %IX8.4 :BOOL;



X_DockPosDetC  :BOOL;
X_NextStnRdyC  :BOOL;
END_VAR

// Device/Application/01_变量/GVL_G
VAR_GLOBAL
Clock_05HZ      AT %MX0.2: BOOL;
Clock_10HZ      AT %MX0.3: BOOL;
Clock_20HZ      AT %MX0.4: BOOL;
Clock_50HZ      AT %MX0.5: BOOL;
Clock_100HZ     AT %MX0.6: BOOL;
	
G_SysRunOk AT %MX2.0:BOOL;
G_SysFault AT %MX2.1:BOOL;
G_SysRstSt AT %MX2.2:BOOL;
G_SysRstAct AT %MX2.3:BOOL;
G_SysRstOk AT %MX2.4:BOOL;

G_SafeDrOk AT %MX2.7 :BOOL;

G_ManMode AT %MX3.0:BOOL;
G_AutoMode AT %MX3.1:BOOL;
G_DryRun AT %MX3.2:BOOL;
G_StepMode AT %MX3.3:BOOL;
G_ProdMode AT %MX3.4:BOOL;

G_PickAPart AT %MX4.0:BOOL;
G_MainLPart AT %MX4.2:BOOL;
G_MainRPart AT %MX4.3:BOOL;
PickAPart: BOOL;
MainLPart:BOOL;
ModAStep AT	%MW10 :INT;
ModCStep AT	%MW12 :INT;	
SysState AT	%MW13 :INT;			
END_VAR
VAR_GLOBAL PERSISTENT RETAIN
TotalProd AT %MB130772 : INT;
CT AT %MB130768 : DINT;
END_VAR

// Device/Application/01_变量/GVL_H
VAR_GLOBAL
H_BuzMaskSw AT %MX99.0 :BOOL;
H_MainLtSw AT %MX99.1 :BOOL;
H_SafeDrMask AT %MX99.3 :BOOL;
H_StnAMask AT %MX99.6 :BOOL;
H_DryRunPB AT %MX100.1 :BOOL;
H_StepPB AT %MX100.2 :BOOL;
H_ProdPB AT %MX100.3 :BOOL;
H_ModAStepPB AT %MX100.4 :BOOL;
H_ModCStepPB AT %MX100.6 :BOOL;
//气缸-主侧A
H_StpC_R_A1 AT %MX110.0 :BOOL;
H_StpC_W_A1 AT %MX110.1 :BOOL;
H_StpC_R_A2 AT %MX110.2 :BOOL;
H_StpC_W_A2 AT %MX110.3 :BOOL;
H_StpC_R_A3 AT %MX110.4 :BOOL;
H_StpC_W_A3 AT %MX110.5 :BOOL;
H_StpC_R_A4 AT %MX110.6 :BOOL;
H_StpC_W_A4 AT %MX110.7 :BOOL;
H_StpC_R_A5 AT %MX111.0 :BOOL;
H_StpC_W_A5 AT %MX111.1 :BOOL;
H_LftC_R_A1 AT %MX111.2 :BOOL;
H_LftC_W_A1 AT %MX111.3 :BOOL;
H_LftC_R_A2 AT %MX111.4 :BOOL;
H_LftC_W_A2 AT %MX111.5 :BOOL;
H_LftC_R_A3 AT %MX111.6 :BOOL;
H_LftC_W_A3 AT %MX111.7 :BOOL;
H_LftC_R_A4 AT %MX112.0 :BOOL;
H_LftC_W_A4 AT %MX112.1 :BOOL;
H_TrnC_R_A1 AT %MX112.2 :BOOL;
H_TrnC_W_A1 AT %MX112.3 :BOOL;
H_ModASftC_R AT %MX112.4 :BOOL;
H_ModASftC_W AT %MX112.5 :BOOL;
H_ModAGrpC_R AT %MX112.6 :BOOL;
H_ModAGrpC_W AT %MX112.7 :BOOL;
H_ModARotC_R AT %MX113.0 :BOOL;
H_ModARotC_W AT %MX113.1 :BOOL;

//气缸-C
H_StpC_R_C1 AT %MX130.0 :BOOL;
H_StpC_W_C1 AT %MX130.1:BOOL;
H_LftC_R_C1 AT %MX130.2 :BOOL;
H_LftC_W_C1 AT %MX130.3 :BOOL;
H_ModCSftC_R AT %MX130.4 :BOOL;
H_ModCSftC_W AT %MX130.5 :BOOL;
H_MdCLftLC_R AT %MX130.6 :BOOL;
H_MdCLftLC_W AT %MX130.7 :BOOL;
H_MdCLftRC_R AT %MX131.0 :BOOL;
H_MdCLftRC_W AT %MX131.1 :BOOL;
H_MdCGrpLC_R AT %MX131.2 :BOOL;
H_MdCGrpLC_W AT %MX131.3 :BOOL;
H_MdCGrpRC_R AT %MX131.4 :BOOL;
H_MdCGrpRC_W AT %MX131.5 :BOOL;
H_MdCRotLC_R AT %MX131.6 :BOOL;
H_MdCRotLC_W AT %MX131.7 :BOOL;
H_MdCRotRC_R AT %MX132.0 :BOOL;
H_MdCRotRC_W AT %MX132.1 :BOOL;
//流水线
H_ConvRunA1 AT %MX114.0 :BOOL;
H_ConvStopA1 AT %MX114.1 :BOOL;
H_ConvRunA2 AT %MX114.2 :BOOL;
H_ConvStopA2 AT %MX114.3 :BOOL;

//伺服-主侧A
H_Ax1ErrRst AT %MX115.0 :BOOL;
H_Ax1HomePB AT %MX115.1 :BOOL;
H_Ax1JogF_PB AT %MX115.2 :BOOL;
H_Ax1JogR_PB AT %MX115.3 :BOOL;
H_Ax1EnSw AT %MX115.4 :BOOL;

H_Ax1TchP1PB AT %MX116.0 :BOOL;
H_Ax1TchP2PB AT %MX116.1 :BOOL;
H_Ax1TchP3PB AT %MX116.2 :BOOL;

H_Ax1MovP1PB AT %MX117.0 :BOOL;
H_Ax1MovP2PB AT %MX117.1 :BOOL;
H_Ax1MovP3PB AT %MX117.2 :BOOL;

END_VAR
VAR_GLOBAL
//气缸-主侧A屏蔽
H_StpCR_A1_M AT %MX200.0 : BOOL;
H_ClrAccT_PB AT %MX204.6: BOOL;
H_StpCW_A1_M AT %MX200.1 : BOOL;
H_StpCR_A2_M AT %MX200.2 : BOOL;
H_StpCW_A2_M AT %MX200.3 : BOOL;
H_StpCR_A3_M AT %MX200.4 : BOOL;
H_StpCW_A3_M AT %MX200.5 : BOOL;
H_StpCR_A4_M AT %MX200.6 : BOOL;
H_StpCW_A4_M AT %MX200.7 : BOOL;
H_StpCR_A5_M AT %MX201.0 : BOOL;
H_StpCW_A5_M AT %MX201.1 : BOOL;
H_LftCR_A1_M AT %MX201.2 : BOOL;
H_LftCW_A1_M AT %MX201.3 : BOOL;
H_LftCR_A2_M AT %MX201.4 : BOOL;
H_LftCW_A2_M AT %MX201.5 : BOOL;
H_LftCR_A3_M AT %MX201.6 : BOOL;
H_LftCW_A3_M AT %MX201.7 : BOOL;
H_LftCR_A4_M AT %MX202.0 : BOOL;
H_LftCW_A4_M AT %MX202.1 : BOOL;
H_TrnCR_A1_M AT %MX202.2 : BOOL;
H_TrnCW_A1_M AT %MX202.3 : BOOL;
H_MdASftCR_M AT %MX202.4 : BOOL;
H_MdASftCW_M AT %MX202.5 : BOOL;
H_MdAGrpCR_M AT %MX202.6 : BOOL;
H_MdAGrpCW_M AT %MX202.7 : BOOL;
H_MdARotCR_M AT %MX203.0 : BOOL;
H_MdARotCW_M AT %MX203.1 : BOOL;
//气缸-C屏蔽
H_StpCR_C1_M AT %MX203.2 : BOOL;
H_StpCW_C1_M AT %MX203.3 : BOOL;
H_LftCR_C1_M AT %MX203.4 : BOOL;
H_LftCW_C1_M AT %MX203.5 : BOOL;
H_MdCSftCR_M AT %MX203.6 : BOOL;
H_MdCSftCW_M AT %MX203.7 : BOOL;
H_MdCLftLR_M AT %MX204.0 : BOOL;
H_MdCLftLW_M AT %MX204.1 : BOOL;
H_MdCRotLR_M AT %MX204.2 : BOOL;
H_MdCRotLW_M AT %MX204.3 : BOOL;
H_MdCGrpLR_M AT %MX204.4 : BOOL;
H_MdCGrpLW_M AT %MX204.5 : BOOL;
END_VAR

// Device/Application/01_变量/GVL_T
VAR_GLOBAL PERSISTENT RETAIN
StpCylPosT AT %MD32700 :TIME;
StpCylTO_T AT %MD32701 :TIME;
LftCylPosT AT %MD32702 :TIME;
LftCylTO_T AT %MD32703 :TIME;
SftCylPosT AT %MD32704 :TIME;
SftCylTO_T AT %MD32705 :TIME;
RotCylPosT AT %MD32706 :TIME;
RotCylTO_T AT %MD32707 :TIME;
GrpCylPosT AT %MD32708 :TIME;
GrpCylTO_T AT %MD32709 :TIME;
TotalTime AT %MB131360 : DINT;
Ax1ErrorID AT %MD32751 :UDINT;

//气缸-主侧A定位延时
H_StpCRPosDyA1 AT %MD32710 :TIME;
H_StpCWPosDyA1 AT %MD32711:TIME;
H_StpCRPosDyA2 AT %MD32712 :TIME;
H_StpCWPosDyA2 AT %MD32713 :TIME;
H_StpCRPosDyA3 AT %MD32714 :TIME;
H_StpCWPosDyA3 AT %MD32715 :TIME;
H_StpCRPosDyA4 AT %MD32716 :TIME;
H_StpCWPosDyA4 AT %MD32717 :TIME;
H_StpCRPosDyA5 AT %MD32718 :TIME;
H_StpCWPosDyA5 AT %MD32719 :TIME;
H_LftCRPosDyA1 AT %MD32720 :TIME;
H_LftCWPosDyA1 AT %MD32721 :TIME;
H_LftCRPosDyA2 AT %MD32722 :TIME;
H_LftCWPosDyA2 AT %MD32723 :TIME;
H_LftCRPosDyA3 AT %MD32724 :TIME;
H_LftCWPosDyA3 AT %MD32725 :TIME;
H_LftCRPosDyA4 AT %MD32726 :TIME;
H_LftCWPosDyA4 AT %MD32727 :TIME;
H_TrnCRPosDyA1 AT %MD32728 :TIME;
H_TrnCWPosDyA1 AT %MD32729 :TIME;
H_MASftCRPosDy AT %MD32730 :TIME;
H_MASftCWPosDy AT %MD32731 :TIME;
H_MAGrpCRPosDy AT %MD32732 :TIME;
H_MAGrpCWPosDy AT %MD32733 :TIME;
H_MARotCRPosDy AT %MD32734 :TIME;
H_MARotCWPosDy AT %MD32735 :TIME;
//气缸-C定位延时
H_StpCRPosDyC1 AT %MD32736 :TIME;
H_StpCWPosDyC1 AT %MD32737 :TIME;
H_LftCRPosDyC1 AT %MD32738 :TIME;
H_LftCWPosDyC1 AT %MD32739 :TIME;
H_MCSftCRPosDy AT %MD32740 :TIME;
H_MCSftCWPosDy AT %MD32741 :TIME;
H_MCLftLRPosDy AT %MD32742 :TIME;
H_MCLftLWPosDy AT %MD32743 :TIME;
H_MCRotLRPosDy AT %MD32744 :TIME;
H_MCRotLWPosDy AT %MD32745 :TIME;
H_MCGrpLRPosDy AT %MD32746 :TIME;
H_MCGrpLWPosDy AT %MD32747 :TIME;
//气缸-主侧A超时延时
H_StpCTO_DlyA1 AT %MD32600 :TIME;
H_StpCTO_DlyA2 AT %MD32601 :TIME;
H_StpCTO_DlyA3 AT %MD32602 :TIME;
H_StpCTO_DlyA4 AT %MD32603 :TIME;
H_StpCTO_DlyA5 AT %MD32604 :TIME;
H_LftCTO_DlyA1 AT %MD32605 :TIME;
H_LftCTO_DlyA2 AT %MD32606 :TIME;
H_LftCTO_DlyA3 AT %MD32607 :TIME;
H_LftCTO_DlyA4 AT %MD32608 :TIME;
H_TrnCTO_DlyA1 AT %MD32609 :TIME;
H_MASftCTO_Dly AT %MD32610 :TIME;
H_MAGrpCTO_Dly AT %MD32611 :TIME;
H_MARotCTO_Dly AT %MD32612 :TIME;
//气缸-C超时延时
H_StpCTO_DlyC1 AT %MD32613 :TIME;
H_LftCTO_DlyC1 AT %MD32614 :TIME;
H_MCSftCTO_Dly AT %MD32615 :TIME;
H_MCLftLTO_Dly AT %MD32616 :TIME;
H_MCRotLTO_Dly AT %MD32617 :TIME;
H_MCGrpLTO_Dly AT %MD32618 :TIME;
//气缸-主侧A屏蔽延时
H_StpCRMaskDyA1 AT %MD32630 :TIME;
H_StpCWMaskDyA1 AT %MD32631 :TIME;
H_StpCRMaskDyA2 AT %MD32632 :TIME;
H_StpCWMaskDyA2 AT %MD32633 :TIME;
H_StpCRMaskDyA3 AT %MD32634 :TIME;
H_StpCWMaskDyA3 AT %MD32635 :TIME;
H_StpCRMaskDyA4 AT %MD32636 :TIME;
H_StpCWMaskDyA4 AT %MD32637 :TIME;
H_StpCRMaskDyA5 AT %MD32638 :TIME;
H_StpCWMaskDyA5 AT %MD32639 :TIME;
H_LftCRMaskDyA1 AT %MD32640 :TIME;
H_LftCWMaskDyA1 AT %MD32641 :TIME;
H_LftCRMaskDyA2 AT %MD32642 :TIME;
H_LftCWMaskDyA2 AT %MD32643 :TIME;
H_LftCRMaskDyA3 AT %MD32644 :TIME;
H_LftCWMaskDyA3 AT %MD32645 :TIME;
H_LftCRMaskDyA4 AT %MD32646 :TIME;
H_LftCWMaskDyA4 AT %MD32647 :TIME;
H_TrnCRMaskDyA1 AT %MD32648 :TIME;
H_TrnCWMaskDyA1 AT %MD32649 :TIME;
H_MASftCRMaskDy AT %MD32650 :TIME;
H_MASftCWMaskDy AT %MD32651 :TIME;
H_MAGrpCRMaskDy AT %MD32652 :TIME;
H_MAGrpCWMaskDy AT %MD32653 :TIME;
H_MARotCRMaskDy AT %MD32654 :TIME;
H_MARotCWMaskDy AT %MD32655 :TIME;
//气缸-C屏蔽延时
H_StpCRMaskDyC1 AT %MD32656 :TIME;
H_StpCWMaskDyC1 AT %MD32657 :TIME;
H_LftCRMaskDyC1 AT %MD32658 :TIME;
H_LftCWMaskDyC1 AT %MD32659 :TIME;
H_MCSftCRMaskDy AT %MD32660 :TIME;
H_MCSftCWMaskDy AT %MD32661 :TIME;
H_MCLftLRMaskDy AT %MD32662 :TIME;
H_MCLftLWMaskDy AT %MD32663 :TIME;
H_MCRotLRMaskDy AT %MD32664 :TIME;
H_MCRotLWMaskDy AT %MD32665 :TIME;
H_MCGrpLRMaskDy AT %MD32666 :TIME;
H_MCGrpLWMaskDy AT %MD32667 :TIME;
END_VAR

// Device/Application/01_变量/GVL_Q
VAR_GLOBAL
//指示灯
Q_TowerLtRed AT %QX3.3 :BOOL;
Q_TowerLtYlw AT %QX3.1 :BOOL;
Q_TowerLtGrn AT %QX3.6 :BOOL;
Q_TowerLtBuz AT %QX3.5 :BOOL;

Q_MainLight AT %QX2.3 :BOOL;

Q_StartLt AT %QX3.0 :BOOL;
Q_StopLt AT %QX3.2 :BOOL;
Q_ResetLt AT %QX3.4 :BOOL;
//流水线
Q_ConvRunA1 AT %QX2.1 :BOOL;
Q_ConvRunA2 AT %QX2.0 :BOOL;
//气缸-A
Q_StpCyl_R_A1 AT %QX13.2 :BOOL;
Q_StpCyl_W_A1 AT %QX11.2:BOOL;
Q_StpCyl_R_A2 AT %QX13.3 :BOOL;
Q_StpCyl_W_A2 AT %QX11.3 :BOOL;
Q_StpCyl_R_A3 AT %QX14.1 :BOOL;
Q_StpCyl_W_A3 AT %QX16.1 :BOOL;
Q_StpCyl_R_A4 AT %QX14.5 :BOOL;
Q_StpCyl_W_A4 AT %QX16.5 :BOOL;
Q_StpCyl_R_A5 AT %QX14.6 :BOOL;
Q_StpCyl_W_A5 AT %QX16.6 :BOOL;
Q_LftCyl_R_A1 AT %QX14.0 :BOOL;
Q_LftCyl_W_A1 AT %QX16.0 :BOOL;
Q_LftCyl_R_A2 AT %QX14.3 :BOOL;
Q_LftCyl_W_A2 AT %QX16.3 :BOOL;
Q_LftCyl_R_A3 AT %QX14.4 :BOOL;
Q_LftCyl_W_A3 AT %QX16.4 :BOOL;
Q_LftCyl_R_A4 AT %QX14.7 :BOOL;
Q_LftCyl_W_A4 AT %QX16.7 :BOOL;
Q_TrnCyl_R_A1 AT %QX14.2 :BOOL;
Q_TrnCyl_W_A1 AT %QX16.2 :BOOL;
Q_ModASftC_R AT %QX12.0 :BOOL;
Q_ModASftC_W AT %QX10.0 :BOOL;
Q_ModAGrpC_R AT %QX12.2 :BOOL;
Q_ModAGrpC_W AT %QX10.2 :BOOL;
Q_ModARotC_R AT %QX12.1 :BOOL;
Q_ModARotC_W AT %QX10.1 :BOOL;
//气缸-C
Q_StpCyl_R_C1 AT %QX15.1 :BOOL;
Q_StpCyl_W_C1 AT %QX17.1 :BOOL;
Q_LftCyl_R_C1 AT %QX15.0 :BOOL;
Q_LftCyl_W_C1 AT %QX17.0 :BOOL;
Q_ModCSftC_R AT %QX12.3 :BOOL;
Q_ModCSftC_W AT %QX10.3 :BOOL;
Q_MdCLftLC_R AT %QX12.4 :BOOL;
Q_MdCLftLC_W AT %QX10.4 :BOOL;
Q_MdCGrpLC_R AT %QX12.6 :BOOL;
Q_MdCGrpLC_W AT %QX10.6 :BOOL;
Q_MdCRotLC_R AT %QX12.5 :BOOL;
Q_MdCRotLC_W AT %QX10.5 :BOOL;

END_VAR

// Device/Application/01_变量/GVL_O
VAR_GLOBAL
//气缸定位到达-A
O_StpC_R_A1 AT %MX140.0 :BOOL;
O_StpC_W_A1 AT %MX140.1 :BOOL;
O_StpC_R_A2 AT %MX140.2 :BOOL;
O_StpC_W_A2 AT %MX140.3 :BOOL;
O_StpC_R_A3 AT %MX140.4 :BOOL;
O_StpC_W_A3 AT %MX140.5 :BOOL;
O_StpC_R_A4 AT %MX140.6 :BOOL;
O_StpC_W_A4 AT %MX140.7 :BOOL;
O_StpC_R_A5 AT %MX141.0 :BOOL;
O_StpC_W_A5 AT %MX141.1 :BOOL;
O_LftC_R_A1 AT %MX141.2 :BOOL;
O_LftC_W_A1 AT %MX141.3 :BOOL;
O_LftC_R_A2 AT %MX141.4 :BOOL;
O_LftC_W_A2 AT %MX141.5 :BOOL;
O_LftC_R_A3 AT %MX141.6 :BOOL;
O_LftC_W_A3 AT %MX141.7 :BOOL;
O_LftC_R_A4 AT %MX142.0 :BOOL;
O_LftC_W_A4 AT %MX142.1 :BOOL;
O_TrnC_R_A1 AT %MX142.2 :BOOL;
O_TrnC_W_A1 AT %MX142.3 :BOOL;
O_ModASftC_R AT %MX142.4 :BOOL;
O_ModASftC_W AT %MX142.5 :BOOL;
O_ModAGrpC_R AT %MX142.6 :BOOL;
O_ModAGrpC_W AT %MX142.7 :BOOL;
O_ModARotC_R AT %MX143.0 :BOOL;
O_ModARotC_W AT %MX143.1 :BOOL;
//气缸定位到达-C
O_StpC_R_C1 AT %MX160.0 :BOOL;
O_StpC_W_C1 AT %MX160.1:BOOL;
O_LftC_R_C1 AT %MX160.2 :BOOL;
O_LftC_W_C1 AT %MX160.3 :BOOL;
O_ModCSftC_R AT %MX160.4 :BOOL;
O_ModCSftC_W AT %MX160.5 :BOOL;
O_MdCLftLC_R AT %MX160.6 :BOOL;
O_MdCLftLC_W AT %MX160.7 :BOOL;
O_MdCGrpLC_R AT %MX161.2 :BOOL;
O_MdCGrpLC_W AT %MX161.3 :BOOL;
O_MdCRotLC_R AT %MX161.6 :BOOL;
O_MdCRotLC_W AT %MX161.7 :BOOL;
//气缸定位异常-A
O_StpCRFltA1 AT %MX170.0 :BOOL;
O_StpCWFltA1 AT %MX170.1 :BOOL;
O_StpCRFltA2 AT %MX170.2 :BOOL;
O_StpCWFltA2 AT %MX170.3 :BOOL;
O_StpCRFltA3 AT %MX170.4 :BOOL;
O_StpCWFltA3 AT %MX170.5 :BOOL;
O_StpCRFltA4 AT %MX170.6 :BOOL;
O_StpCWFltA4 AT %MX170.7 :BOOL;
O_StpCRFltA5 AT %MX171.0 :BOOL;
O_StpCWFltA5 AT %MX171.1 :BOOL;
O_LftCRFltA1 AT %MX171.2 :BOOL;
O_LftCWFltA1 AT %MX171.3 :BOOL;
O_LftCRFltA2 AT %MX171.4 :BOOL;
O_LftCWFltA2 AT %MX171.5 :BOOL;
O_LftCRFltA3 AT %MX171.6 :BOOL;
O_LftCWFltA3 AT %MX171.7 :BOOL;
O_LftCRFltA4 AT %MX172.0 :BOOL;
O_LftCWFltA4 AT %MX172.1 :BOOL;
O_TrnCRFltA1 AT %MX172.2 :BOOL;
O_TrnCWFltA1 AT %MX172.3 :BOOL;
O_MASftCRFlt AT %MX172.4 :BOOL;
O_MASftCWFlt AT %MX172.5 :BOOL;
O_MAGrpCRFlt AT %MX172.6 :BOOL;
O_MAGrpCWFlt AT %MX172.7 :BOOL;
O_MARotCRFlt AT %MX173.0 :BOOL;
O_MARotCWFlt AT %MX173.1 :BOOL;
//气缸定位异常-C
O_StpCRFltC1 AT %MX190.0 :BOOL;
O_StpCWFltC1 AT %MX190.1:BOOL;
O_LftCRFltC1 AT %MX190.2 :BOOL;
O_LftCWFltC1 AT %MX190.3 :BOOL;
O_MCSftCRFlt AT %MX190.4 :BOOL;
O_MCSftCWFlt AT %MX190.5 :BOOL;
O_MCLftLRFlt AT %MX190.6 :BOOL;
O_MCLftLWFlt AT %MX190.7 :BOOL;
O_MCLftRRFlt AT %MX191.0 :BOOL;
O_MCLftRWFlt AT %MX191.1 :BOOL;
O_MCGrpLRFlt AT %MX191.2 :BOOL;
O_MCGrpLWFlt AT %MX191.3 :BOOL;
O_MCGrpRRFlt AT %MX191.4 :BOOL;
O_MCGrpRWFlt AT %MX191.5 :BOOL;
O_MCRotLRFlt AT %MX191.6 :BOOL;
O_MCRotLWFlt AT %MX191.7 :BOOL;
O_MCRotRRFlt AT %MX192.0 :BOOL;
O_MCRotRWFlt AT %MX192.1 :BOOL;
O_EmgStopFlt AT %MX193.0 :BOOL;
O_SafeDrFlt AT %MX193.1 :BOOL;
  
ModAFault:BOOL;
O_Stp2DirErr   AT %MX193.2 :BOOL;
O_Stp3CarrTO AT %MX193.3 :BOOL;
O_PickCarrTO  AT %MX193.4 :BOOL;
O_Stp5CarrTO AT %MX193.5 :BOOL;
O_WaitCarrTO  AT %MX193.6 :BOOL;
END_VAR

// Device/Application/01_变量/GVT_INT
VAR_GLOBAL
	//自动控制区域A
	St1Org_A: BOOL;
	St1Work_A: BOOL;
	DirDetDly_A: TON;
	WpDirDet_A: BOOL;
	DirChkStp_A: INT;
	DirChkRdy_A: BOOL;
	St2Org_A: BOOL;
	St2Work_A: BOOL;
	DetResSt2_A: INT;
	DetResSt3_A: INT;
	LftRotStOrgA: BOOL;
	LftRotNoRevA: BOOL;
	RevStep_A: INT;
	UD1Work_A: BOOL;
	RevWork_A: BOOL;
	St3Work_A: BOOL;
	UD1Org_A: BOOL;
	UD1Work1_A: BOOL;
	RevOrg_A: BOOL;
	UD1OrgPos1_A: BOOL;
	St3Work1_A: BOOL;
	St3Org_A: BOOL;
	R_TRIG_A: R_TRIG;
	UD2Work_A: BOOL;
	PickStnDly_A: TON;
	ReqAuxPick_A: BOOL;
	PickStnStp_A: INT;
	UD2Org_A: BOOL;
	PickModStp_A: INT;
	AlwAuxPlaceA: BOOL;
	ModReadyActA: BOOL;
	ModAllOrg_A: BOOL;
	ZAxMovPick_A: BOOL;
	GripCylWorkA: BOOL;
	ZAxMovInit_A: BOOL;
	SftCylWork_A: BOOL;
	ZAxMovPlaceA: BOOL;
	GripCylOrg_A: BOOL;
	ZAxMovInit1A: BOOL;
	SftCylOrg_A: BOOL;
	PlaceStp_A: INT;
	PlacePosDlyA: TON;
	ModRlsBusy_A: BOOL;
	ModPickBusyA: BOOL;
	St4Work_A: BOOL;
	UD3Work_A: BOOL;
	St4Org_A: BOOL;
	UD3Org_A: BOOL;
	BufStnStep_A: INT;
	WaitStnStpA: INT;
	St5Work_A: BOOL;
	St5Org_A: BOOL;
	WaitStnDly_A: TON;
	UD4Work_A: BOOL;
	ReqMainPickA: BOOL;
	UD4Org_A: BOOL;
	RotCylWork_A: BOOL;
	RotCylOrg_A: BOOL;
	PlaceStnMemA: BOOL;

//自动控区域C
	R_TRIG_C1: R_TRIG;
	R_TRIG_C: R_TRIG;
	MainModStepC: INT;
	DockStnStp_C: INT;
	AlwMainRls_C: BOOL;
	DockStnDly_C: TON;
	MainRlsBusyC: BOOL;
	StpCylWork_C: BOOL;
	LftCylWork_C: BOOL;
	LftCylOrg_C: BOOL;
	StpCylOrg_C: BOOL;
	MainModRdy_C: BOOL;
	MainAllOrg_C: BOOL;
	MainSftOrg_C: BOOL;
	MainLLftWrkC: BOOL;
	MainLGrpWrkC: BOOL;
	MainLLftOrgC: BOOL;
	MainSftWrk_C: BOOL;
	MainLLftWrk1C: BOOL;
	MainLRotWrk_C: BOOL;
	MainLGrpOrg_C: BOOL;
	MainLLftOrg1C: BOOL;
	MainLRotOrgC: BOOL;
	MainSftWrk1_C: BOOL;
	MainSftOrg1C: BOOL;
	MainPickAct_A: BOOL;
END_VAR

// Device/Application/01_变量/GVL_Axis
VAR_GLOBAL
//轴写入
Ax1Enable AT %MX7000.0:BOOL;
Ax1EmgStop AT %MX7010.0:BOOL;
Ax1Home AT %MX7020.0:BOOL;
Ax1JogFwd AT %MX7030.0:BOOL;
Ax1JogRev AT %MX7040.0:BOOL;
Ax1AbsMove AT %MX7050.0:BOOL;
Ax1ErrRst AT %MX7060.0:BOOL;
END_VAR

VAR_GLOBAL PERSISTENT RETAIN
Ax1Accel AT %MD30000:REAL;
Ax1Decel AT %MD30100:REAL;
Ax1JogSpd AT %MD30200:REAL;
Ax1AbsSpd AT %MD30300:REAL;
Ax1AbsPos AT %MD30400:REAL;
END_VAR
VAR_GLOBAL
//轴读取
Ax1PosLim AT %MX7100.0:BOOL;
Ax1NegLim AT %MX7110.0:BOOL;
Ax1Origin AT %MX7120.0:BOOL;
Ax1Error AT %MX7130.0:BOOL;
Ax1Busy AT %MX7140.0:BOOL;
Ax1InPos AT %MX7150.0:BOOL;
Ax1HomeOK AT %MX7160.0:BOOL;
Ax1CurPos AT %MD20000:REAL;
END_VAR
VAR_GLOBAL RETAIN PERSISTENT
//校点数据存储
Ax1PosP1 AT %MD31000:REAL;
Ax1PosP2 AT %MD31002:REAL;
Ax1PosP3 AT %MD31004:REAL;
END_VAR
VAR_GLOBAL
//伺服定位
Ax1GoP1 AT %MX7200.0:BOOL;
Ax1GoP2 AT %MX7200.1:BOOL;
Ax1GoP3 AT %MX7200.2:BOOL;
END_VAR

// Device/Application/03_程序/OB/PLC_PRG
PROGRAM PLC_PRG
VAR
END_VAR

Mode();
Rst();
Error();
Auto_A();
Auto_C();
Cylinder_AZone();
Cylinder_CZone();
Other();
Axis_Teaching();

END_PROGRAM

// Device/Application/03_程序/系统/Mode
PROGRAM Mode
VAR
	PLS_0: R_TRIG;
	PLS_1: R_TRIG;
	PLS_2: R_TRIG;
	TON1      :TON;
	TON2      :TON;
	TON3      :TON;
	TON4      :TON;
	TON5      :TON;
	TON6      :TON;
	TON7      :TON;
	TON8      :TON;
	TON9      :TON;
	TON10      :TON;
	TON11      :TON;
	NOT1: BOOL;
	TON_0: TON;
	PLS_3: R_TRIG;
END_VAR
VAR // added by the converter: edge detectors and wires of the graphical bodies
    _w1, _w2, _w3, _w4, _w5, _w6, _w7, _w8, _w9, _w10, _w11, _w12, _w13, _w14, _w15, _w16, _w17, _w18, _w19, _w20, _w21 : BOOL;
END_VAR

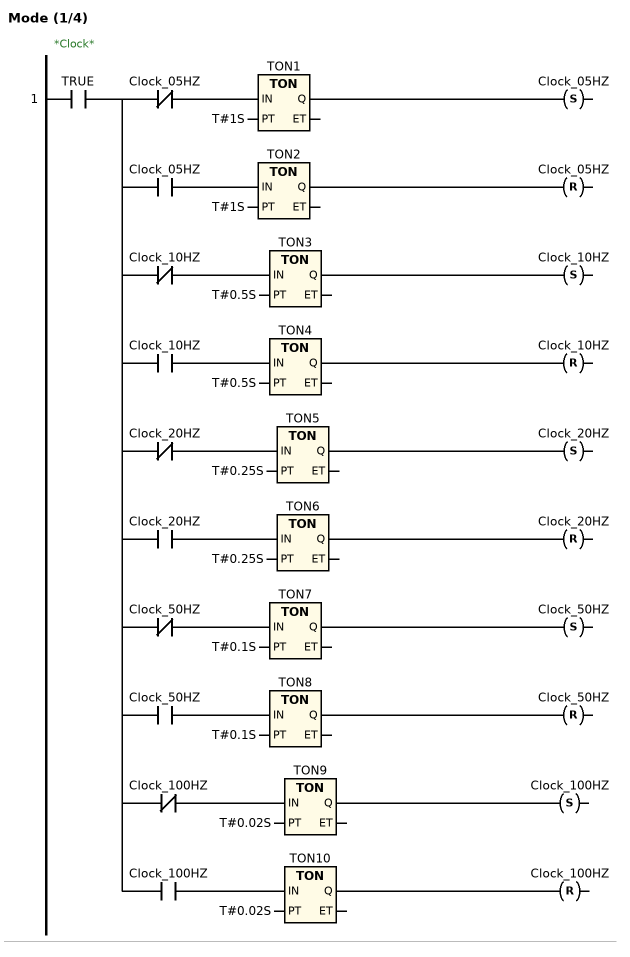
// NETWORK 1
// *Clock*
TON1(IN := TRUE AND NOT Clock_05HZ, PT := T#1S); // TON
Clock_05HZ S= TON1.Q;
TON2(IN := TRUE AND Clock_05HZ, PT := T#1S); // TON
Clock_05HZ R= TON2.Q;
TON3(IN := TRUE AND NOT Clock_10HZ, PT := T#0.5S); // TON
Clock_10HZ S= TON3.Q;
TON4(IN := TRUE AND Clock_10HZ, PT := T#0.5S); // TON
Clock_10HZ R= TON4.Q;
TON5(IN := TRUE AND NOT Clock_20HZ, PT := T#0.25S); // TON
Clock_20HZ S= TON5.Q;
TON6(IN := TRUE AND Clock_20HZ, PT := T#0.25S); // TON
Clock_20HZ R= TON6.Q;
TON7(IN := TRUE AND NOT Clock_50HZ, PT := T#0.1S); // TON
Clock_50HZ S= TON7.Q;
TON8(IN := TRUE AND Clock_50HZ, PT := T#0.1S); // TON
Clock_50HZ R= TON8.Q;
TON9(IN := TRUE AND NOT Clock_100HZ, PT := T#0.02S); // TON
Clock_100HZ S= TON9.Q;
TON10(IN := TRUE AND Clock_100HZ, PT := T#0.02S); // TON
Clock_100HZ R= TON10.Q;

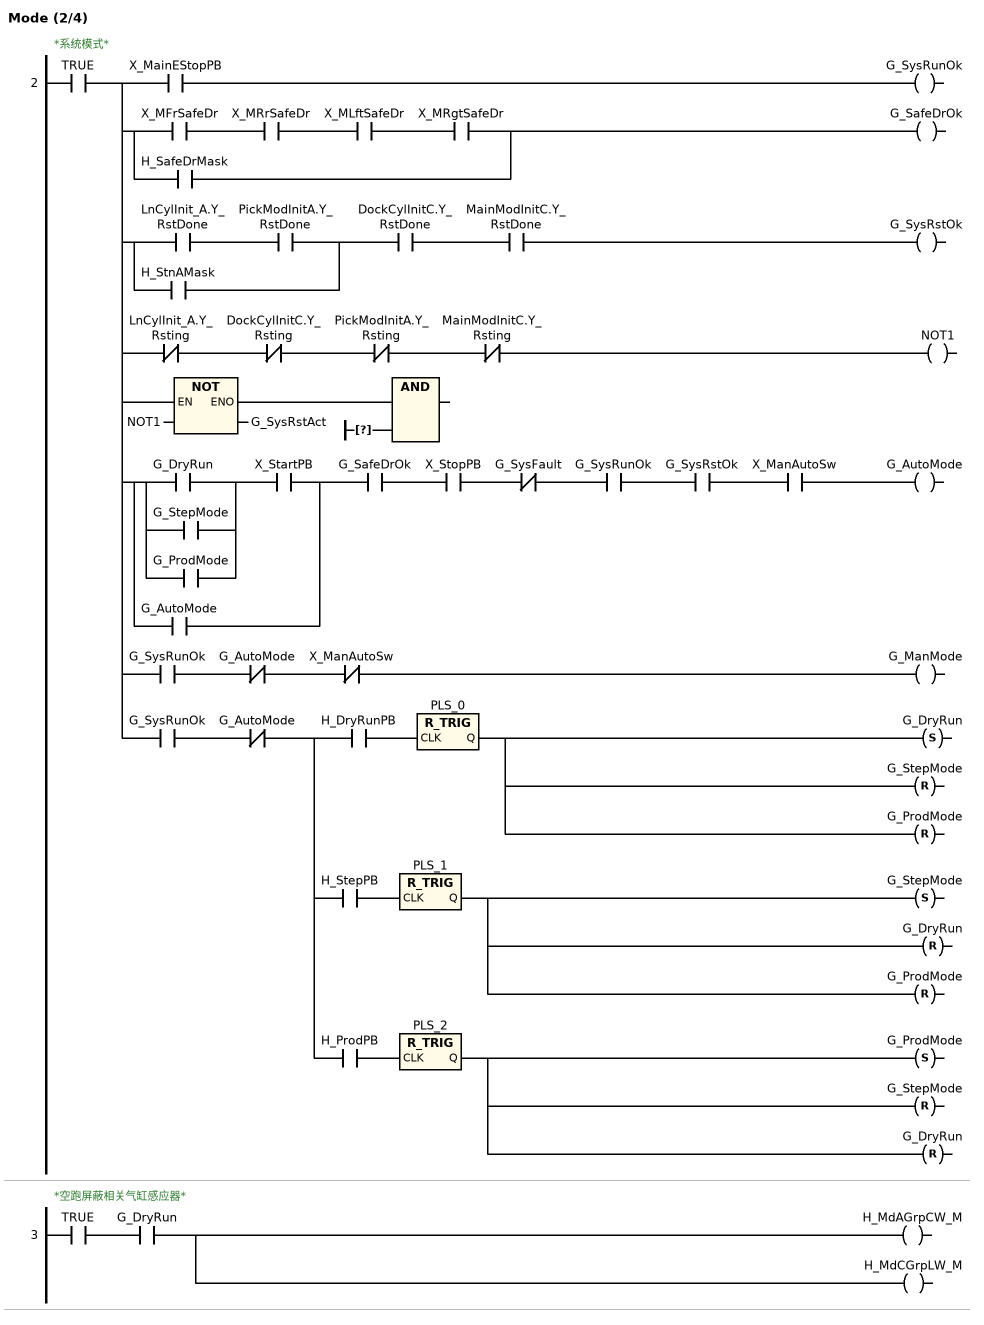
// NETWORK 2
// *系统模式*
_w1 := TRUE AND X_MainEStopPB;
G_SysRunOk := _w1;
_w2 := (TRUE AND X_MFrSafeDr) AND X_MRrSafeDr AND X_MLftSafeDr AND X_MRgtSafeDr OR TRUE AND H_SafeDrMask;
G_SafeDrOk := _w2;
_w3 := ((TRUE AND LnCylInit_A.Y_RstDone) AND PickModInitA.Y_RstDone OR TRUE AND H_StnAMask) AND DockCylInitC.Y_RstDone AND MainModInitC.Y_RstDone;
G_SysRstOk := _w3;
_w4 := (TRUE AND NOT LnCylInit_A.Y_Rsting) AND NOT DockCylInitC.Y_Rsting AND NOT PickModInitA.Y_Rsting AND NOT MainModInitC.Y_Rsting;
NOT1 := _w4;
G_SysRstAct := NOT NOT1;
_w5 := ((TRUE AND G_DryRun OR TRUE AND G_StepMode OR TRUE AND G_ProdMode) AND X_StartPB OR TRUE AND G_AutoMode) AND G_SafeDrOk AND X_StopPB AND NOT G_SysFault AND G_SysRunOk AND G_SysRstOk AND X_ManAutoSw;
G_AutoMode := _w5;
_w6 := (TRUE AND G_SysRunOk) AND NOT G_AutoMode AND NOT X_ManAutoSw;
G_ManMode := _w6;
_w7 := (TRUE AND G_SysRunOk) AND NOT G_AutoMode;
PLS_0(CLK := _w7 AND H_DryRunPB); // R_TRIG
G_DryRun S= PLS_0.Q;
G_StepMode R= PLS_0.Q;
G_ProdMode R= PLS_0.Q;
PLS_1(CLK := _w7 AND H_StepPB); // R_TRIG
G_StepMode S= PLS_1.Q;
G_DryRun R= PLS_1.Q;
G_ProdMode R= PLS_1.Q;
PLS_2(CLK := _w7 AND H_ProdPB); // R_TRIG
G_ProdMode S= PLS_2.Q;
G_StepMode R= PLS_2.Q;
G_DryRun R= PLS_2.Q;

// NETWORK 3
// *空跑屏蔽相关气缸感应器*
_w8 := TRUE AND G_DryRun;
H_MdAGrpCW_M := _w8;
H_MdCGrpLW_M := _w8;

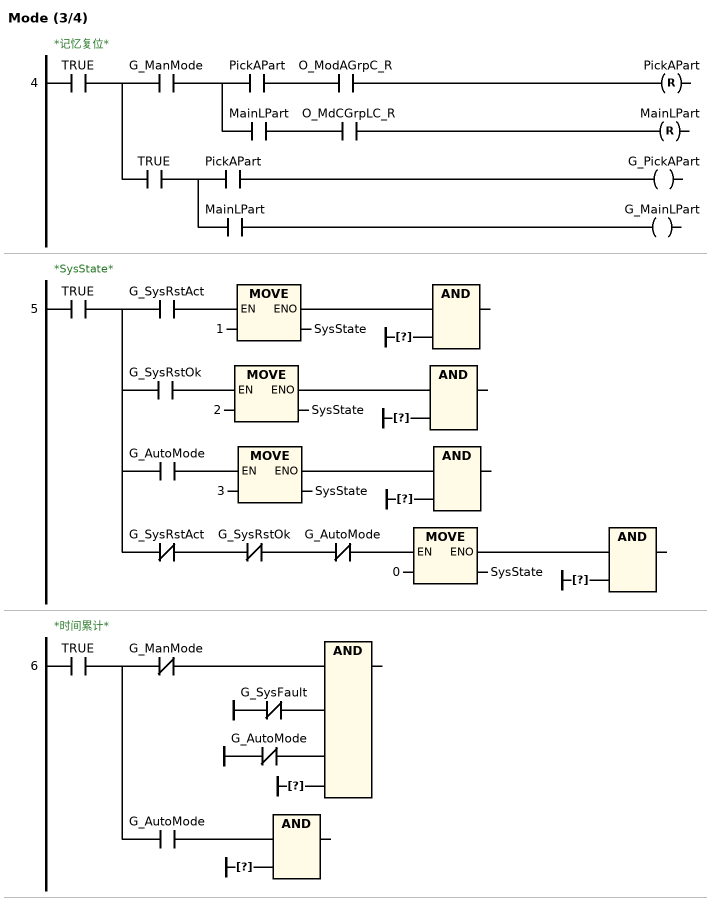
// NETWORK 4
// *记忆复位*
_w9 := TRUE AND G_ManMode;
_w10 := (_w9 AND PickAPart) AND O_ModAGrpC_R;
PickAPart R= _w10;
_w11 := (_w9 AND MainLPart) AND O_MdCGrpLC_R;
MainLPart R= _w11;
_w12 := TRUE AND TRUE;
_w13 := _w12 AND PickAPart;
G_PickAPart := _w13;
_w14 := _w12 AND MainLPart;
G_MainLPart := _w14;

// NETWORK 5
// *SysState*
_w15 := TRUE AND G_SysRstAct;
IF _w15 THEN SysState := 1; END_IF
_w16 := TRUE AND G_SysRstOk;
IF _w16 THEN SysState := 2; END_IF
_w17 := TRUE AND G_AutoMode;
IF _w17 THEN SysState := 3; END_IF
_w18 := (TRUE AND NOT G_SysRstAct) AND NOT G_SysRstOk AND NOT G_AutoMode;
IF _w18 THEN SysState := 0; END_IF

// NETWORK 6
// *时间累计*

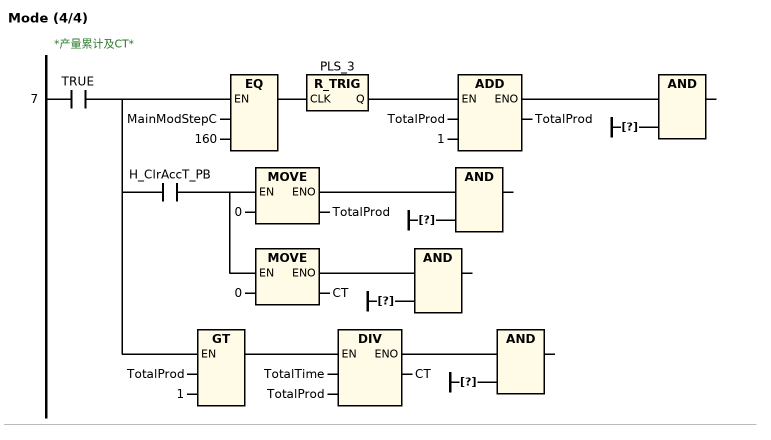
// NETWORK 7
// *产量累计及CT*
PLS_3(CLK := MainModStepC = 160); // R_TRIG
_w19 := PLS_3.Q;
IF _w19 THEN TotalProd := TotalProd + 1; END_IF
_w20 := TRUE AND H_ClrAccT_PB;
IF _w20 THEN TotalProd := 0; END_IF
IF _w20 THEN CT := 0; END_IF
_w21 := TotalProd > 1;
IF _w21 THEN CT := TotalTime / TotalProd; END_IF

END_PROGRAM

// Device/Application/03_程序/系统/Rst
PROGRAM Rst
VAR
	
	LnInitEnA: BOOL;
	LnInitStA: BOOL;
	DckInitEnC: BOOL;
	DckInitStC: BOOL;
	
	PModInitEnA: BOOL;
	PModInitStA: BOOL;
	MModInitEnC: BOOL;
	MModInitStC: BOOL;
	
	T1: TON;
	T2: TON;
	T3: TON;
	T4: TON;
	T5: TON;
	T6: TON;
END_VAR
VAR // added by the converter: edge detectors and wires of the graphical bodies
    _w1, _w2, _w3, _w4 : BOOL;
END_VAR

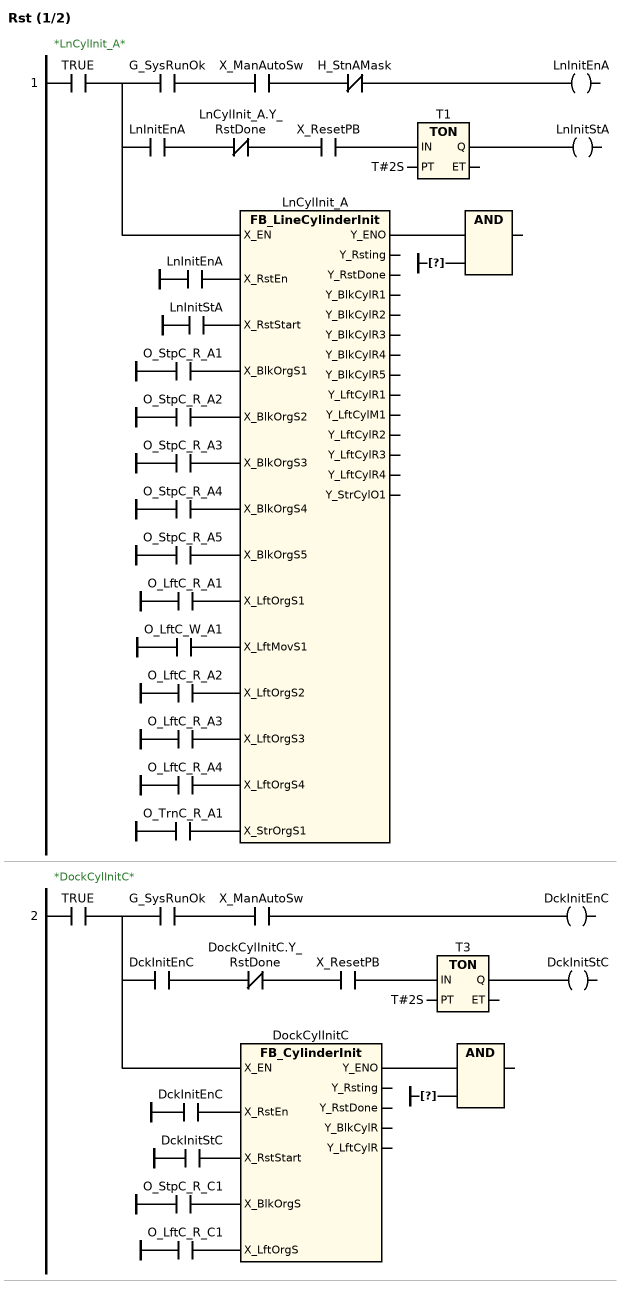
// NETWORK 1
// *LnCylInit_A*
_w1 := (TRUE AND G_SysRunOk) AND X_ManAutoSw AND NOT H_StnAMask;
LnInitEnA := _w1;
T1(IN := (TRUE AND LnInitEnA) AND NOT LnCylInit_A.Y_RstDone AND X_ResetPB, PT := T#2S); // TON
LnInitStA := T1.Q;
LnCylInit_A(
    X_EN := TRUE,
    X_RstEn := LnInitEnA,
    X_RstStart := LnInitStA,
    X_BlkOrgS1 := O_StpC_R_A1,
    X_BlkOrgS2 := O_StpC_R_A2,
    X_BlkOrgS3 := O_StpC_R_A3,
    X_BlkOrgS4 := O_StpC_R_A4,
    X_BlkOrgS5 := O_StpC_R_A5,
    X_LftOrgS1 := O_LftC_R_A1,
    X_LftMovS1 := O_LftC_W_A1,
    X_LftOrgS2 := O_LftC_R_A2,
    X_LftOrgS3 := O_LftC_R_A3,
    X_LftOrgS4 := O_LftC_R_A4,
    X_StrOrgS1 := O_TrnC_R_A1); // FB_LineCylinderInit

// NETWORK 2
// *DockCylInitC*
_w2 := (TRUE AND G_SysRunOk) AND X_ManAutoSw;
DckInitEnC := _w2;
T3(IN := (TRUE AND DckInitEnC) AND NOT DockCylInitC.Y_RstDone AND X_ResetPB, PT := T#2S); // TON
DckInitStC := T3.Q;
DockCylInitC(
    X_EN := TRUE,
    X_RstEn := DckInitEnC,
    X_RstStart := DckInitStC,
    X_BlkOrgS := O_StpC_R_C1,
    X_LftOrgS := O_LftC_R_C1); // FB_CylinderInit

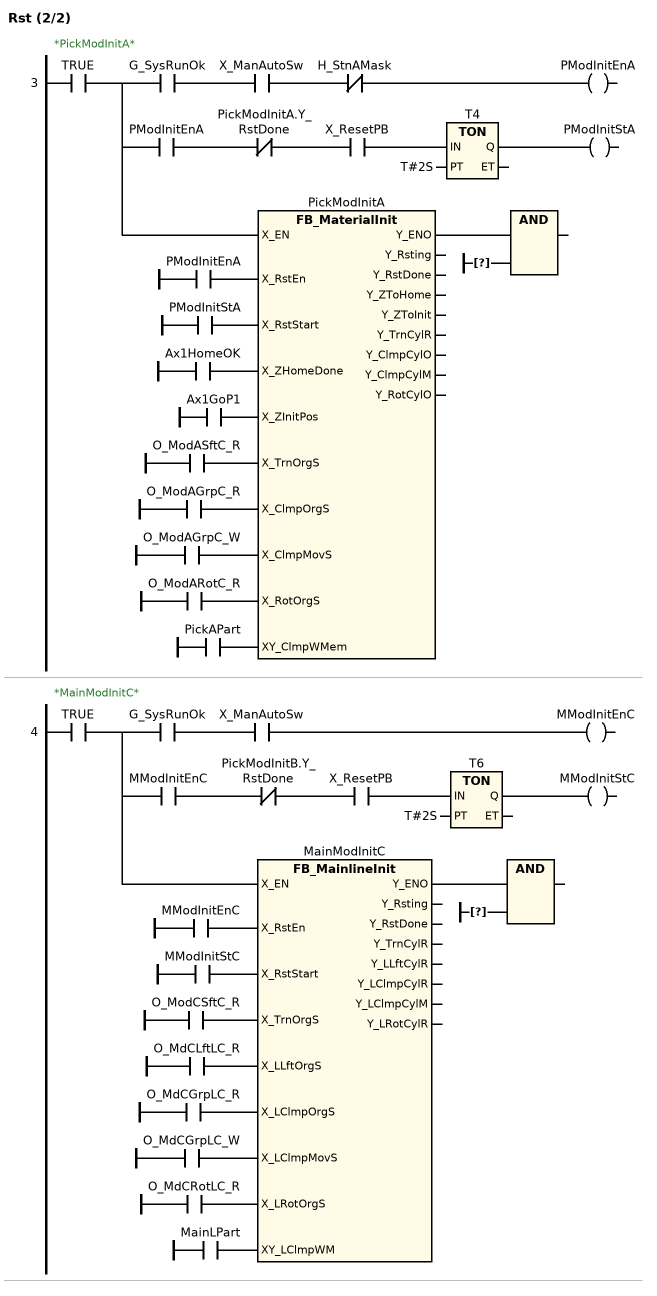
// NETWORK 3
// *PickModInitA*
_w3 := (TRUE AND G_SysRunOk) AND X_ManAutoSw AND NOT H_StnAMask;
PModInitEnA := _w3;
T4(IN := (TRUE AND PModInitEnA) AND NOT PickModInitA.Y_RstDone AND X_ResetPB, PT := T#2S); // TON
PModInitStA := T4.Q;
PickModInitA(
    X_EN := TRUE,
    X_RstEn := PModInitEnA,
    X_RstStart := PModInitStA,
    X_ZHomeDone := Ax1HomeOK,
    X_ZInitPos := Ax1GoP1,
    X_TrnOrgS := O_ModASftC_R,
    X_ClmpOrgS := O_ModAGrpC_R,
    X_ClmpMovS := O_ModAGrpC_W,
    X_RotOrgS := O_ModARotC_R,
    XY_ClmpWMem := PickAPart); // FB_MaterialInit

// NETWORK 4
// *MainModInitC*
_w4 := (TRUE AND G_SysRunOk) AND X_ManAutoSw;
MModInitEnC := _w4;
T6(IN := (TRUE AND MModInitEnC) AND NOT PickModInitB.Y_RstDone AND X_ResetPB, PT := T#2S); // TON
MModInitStC := T6.Q;
MainModInitC(
    X_EN := TRUE,
    X_RstEn := MModInitEnC,
    X_RstStart := MModInitStC,
    X_TrnOrgS := O_ModCSftC_R,
    X_LLftOrgS := O_MdCLftLC_R,
    X_LClmpOrgS := O_MdCGrpLC_R,
    X_LClmpMovS := O_MdCGrpLC_W,
    X_LRotOrgS := O_MdCRotLC_R,
    XY_LClmpWM := MainLPart); // FB_MainlineInit

END_PROGRAM

// Device/Application/02_功能块/初始化/FB_LineCylinderInit
FUNCTION_BLOCK FB_LineCylinderInit
VAR_INPUT
X_EN: BOOL;
X_RstEn : BOOL;
X_RstStart : BOOL;
X_BlkOrgS1: BOOL;
X_BlkOrgS2: BOOL;
X_BlkOrgS3: BOOL;
X_BlkOrgS4: BOOL;
X_BlkOrgS5: BOOL;	
X_LftOrgS1: BOOL;
X_LftMovS1: BOOL;
X_LftOrgS2: BOOL;
X_LftOrgS3: BOOL;
X_LftOrgS4: BOOL;
X_StrOrgS1: BOOL;
END_VAR
VAR_OUTPUT
Y_ENO: BOOL;
Y_Rsting : BOOL;
Y_RstDone : BOOL;
Y_BlkCylR1: BOOL;
Y_BlkCylR2: BOOL;
Y_BlkCylR3: BOOL;
Y_BlkCylR4: BOOL;
Y_BlkCylR5: BOOL; 
Y_LftCylR1: BOOL;
Y_LftCylM1: BOOL;
Y_LftCylR2: BOOL;
Y_LftCylR3: BOOL;
Y_LftCylR4: BOOL;
Y_StrCylO1: BOOL;
END_VAR

VAR

	PLS_0: R_TRIG;
	RstStep: INT;
	TON_0: TON;
	TON_1: TON;
	OrgPos1: BOOL;
	OrgPos2: BOOL;
	Delay1: BOOL;
	Delay2: BOOL;
END_VAR
VAR // added by the converter: edge detectors and wires of the graphical bodies
    _w1, _w2, _w3, _w4, _w5, _w6, _w7, _w8, _w9, _w10 : BOOL;
END_VAR

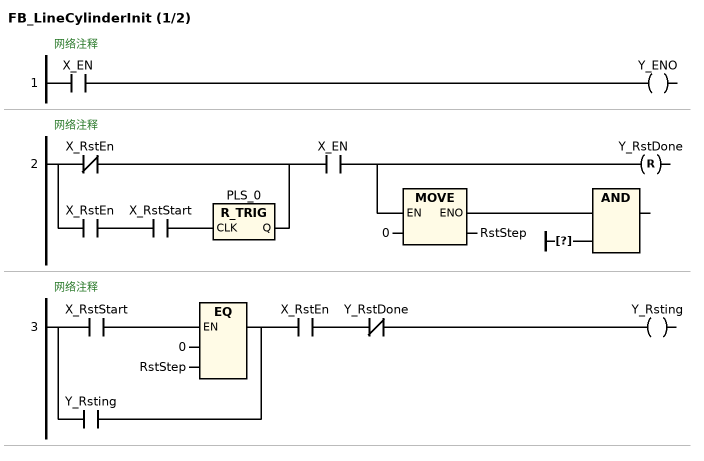
// NETWORK 1
// 网络注释
Y_ENO := X_EN;

// NETWORK 2
// 网络注释
PLS_0(CLK := X_RstEn AND X_RstStart); // R_TRIG
_w1 := (NOT X_RstEn OR PLS_0.Q) AND X_EN;
Y_RstDone R= _w1;
IF _w1 THEN RstStep := 0; END_IF

// NETWORK 3
// 网络注释
Y_Rsting := (X_RstStart AND 0 = RstStep OR Y_Rsting) AND X_RstEn AND NOT Y_RstDone;

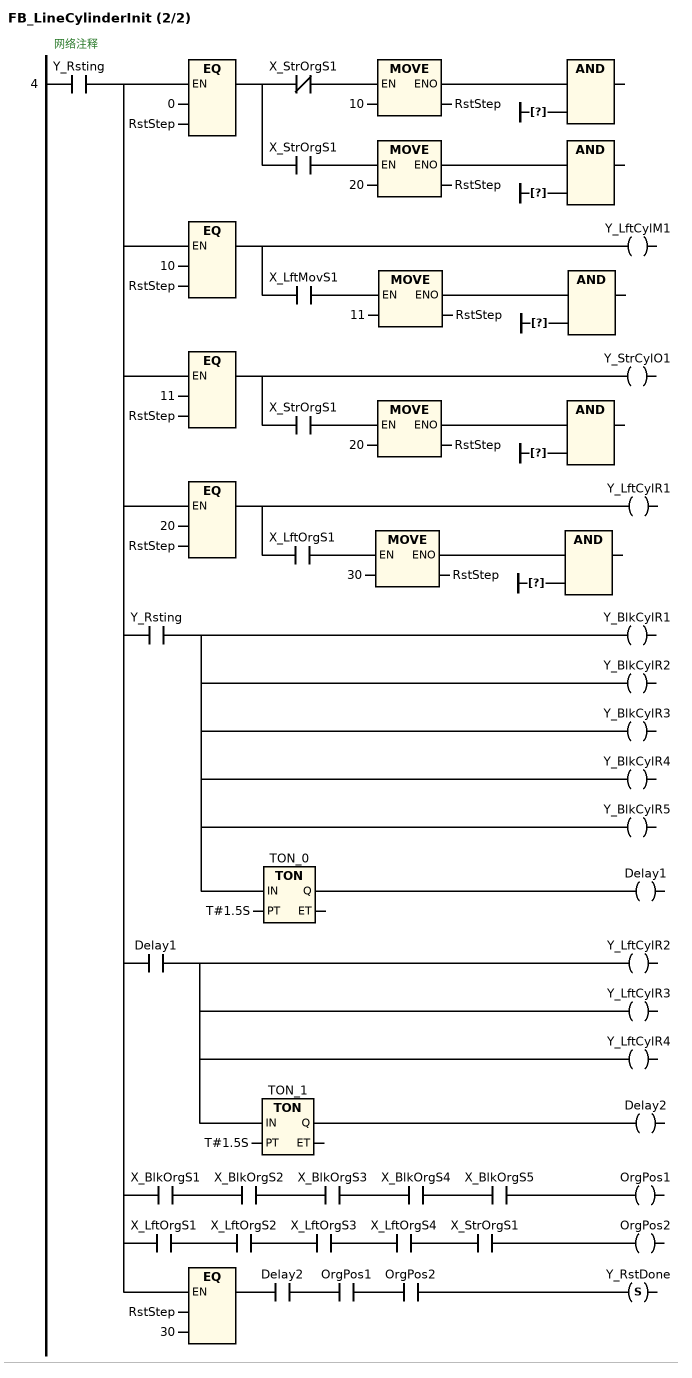
// NETWORK 4
// 网络注释
_w2 := Y_Rsting AND 0 = RstStep;
IF _w2 AND NOT X_StrOrgS1 THEN RstStep := 10; END_IF
IF _w2 AND X_StrOrgS1 THEN RstStep := 20; END_IF
_w3 := Y_Rsting AND 10 = RstStep;
Y_LftCylM1 := _w3;
IF _w3 AND X_LftMovS1 THEN RstStep := 11; END_IF
_w4 := Y_Rsting AND 11 = RstStep;
Y_StrCylO1 := _w4;
IF _w4 AND X_StrOrgS1 THEN RstStep := 20; END_IF
_w5 := Y_Rsting AND 20 = RstStep;
Y_LftCylR1 := _w5;
IF _w5 AND X_LftOrgS1 THEN RstStep := 30; END_IF
_w6 := Y_Rsting AND Y_Rsting;
Y_BlkCylR1 := _w6;
Y_BlkCylR2 := _w6;
Y_BlkCylR3 := _w6;
Y_BlkCylR4 := _w6;
Y_BlkCylR5 := _w6;
TON_0(IN := _w6, PT := T#1.5S); // TON
Delay1 := TON_0.Q;
_w7 := Y_Rsting AND Delay1;
Y_LftCylR2 := _w7;
Y_LftCylR3 := _w7;
Y_LftCylR4 := _w7;
TON_1(IN := _w7, PT := T#1.5S); // TON
Delay2 := TON_1.Q;
_w8 := (Y_Rsting AND X_BlkOrgS1) AND X_BlkOrgS2 AND X_BlkOrgS3 AND X_BlkOrgS4 AND X_BlkOrgS5;
OrgPos1 := _w8;
_w9 := (Y_Rsting AND X_LftOrgS1) AND X_LftOrgS2 AND X_LftOrgS3 AND X_LftOrgS4 AND X_StrOrgS1;
OrgPos2 := _w9;
_w10 := (Y_Rsting AND RstStep = 30) AND Delay2 AND OrgPos1 AND OrgPos2;
Y_RstDone S= _w10;

END_FUNCTION_BLOCK

// Device/Application/02_功能块/初始化/FB_CylinderInit
FUNCTION_BLOCK FB_CylinderInit
VAR_INPUT
X_EN: BOOL;
X_RstEn : BOOL;
X_RstStart : BOOL;
X_BlkOrgS: BOOL;	
X_LftOrgS: BOOL;
END_VAR
VAR_OUTPUT
Y_ENO: BOOL;
Y_Rsting : BOOL;
Y_RstDone : BOOL;
Y_BlkCylR: BOOL;
Y_LftCylR: BOOL;
END_VAR

VAR

	PLS_0: R_TRIG;
	
END_VAR
VAR // added by the converter: edge detectors and wires of the graphical bodies
    _w1 : BOOL;
END_VAR

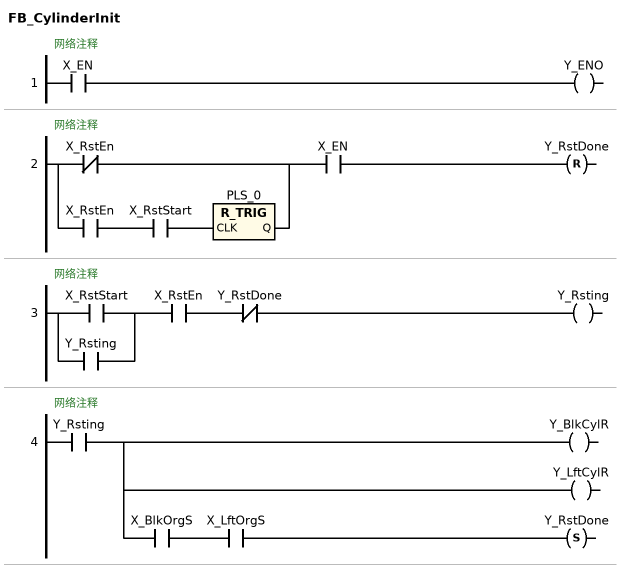
// NETWORK 1
// 网络注释
Y_ENO := X_EN;

// NETWORK 2
// 网络注释
PLS_0(CLK := X_RstEn AND X_RstStart); // R_TRIG
Y_RstDone R= (NOT X_RstEn OR PLS_0.Q) AND X_EN;

// NETWORK 3
// 网络注释
Y_Rsting := (X_RstStart OR Y_Rsting) AND X_RstEn AND NOT Y_RstDone;

// NETWORK 4
// 网络注释
Y_BlkCylR := Y_Rsting;
Y_LftCylR := Y_Rsting;
_w1 := (Y_Rsting AND X_BlkOrgS) AND X_LftOrgS;
Y_RstDone S= _w1;

END_FUNCTION_BLOCK

// Device/Application/02_功能块/初始化/FB_MaterialInit
FUNCTION_BLOCK FB_MaterialInit
VAR_INPUT
X_EN: BOOL;
X_RstEn : BOOL;
X_RstStart : BOOL;
X_ZHomeDone : BOOL;
X_ZInitPos : BOOL;
X_TrnOrgS: BOOL;
X_ClmpOrgS: BOOL;
X_ClmpMovS: BOOL;
X_RotOrgS: BOOL;

END_VAR

VAR_OUTPUT
Y_ENO: BOOL;
Y_Rsting : BOOL;
Y_RstDone : BOOL;
Y_ZToHome : BOOL;
Y_ZToInit : BOOL;
Y_TrnCylR: BOOL;
Y_ClmpCylO: BOOL;
Y_ClmpCylM: BOOL;
Y_RotCylO: BOOL;

END_VAR
VAR_IN_OUT
	XY_ClmpWMem  : BOOL;
END_VAR
VAR
	PLS_0: R_TRIG;
	RstStep: INT;
	TON_0: TON;
END_VAR
VAR // added by the converter: edge detectors and wires of the graphical bodies
    _w1, _w2, _w3, _w4, _w5, _w6, _w7, _w8, _w9, _w10, _w11, _w12, _w13 : BOOL;
END_VAR

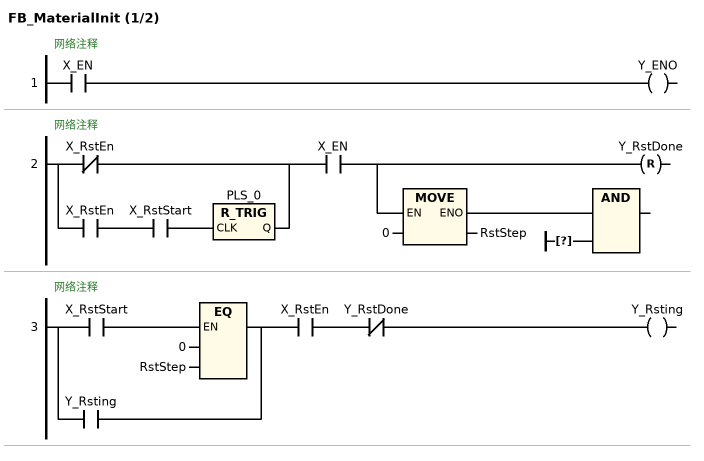
// NETWORK 1
// 网络注释
Y_ENO := X_EN;

// NETWORK 2
// 网络注释
PLS_0(CLK := X_RstEn AND X_RstStart); // R_TRIG
_w1 := (NOT X_RstEn OR PLS_0.Q) AND X_EN;
Y_RstDone R= _w1;
IF _w1 THEN RstStep := 0; END_IF

// NETWORK 3
// 网络注释
Y_Rsting := (X_RstStart AND 0 = RstStep OR Y_Rsting) AND X_RstEn AND NOT Y_RstDone;

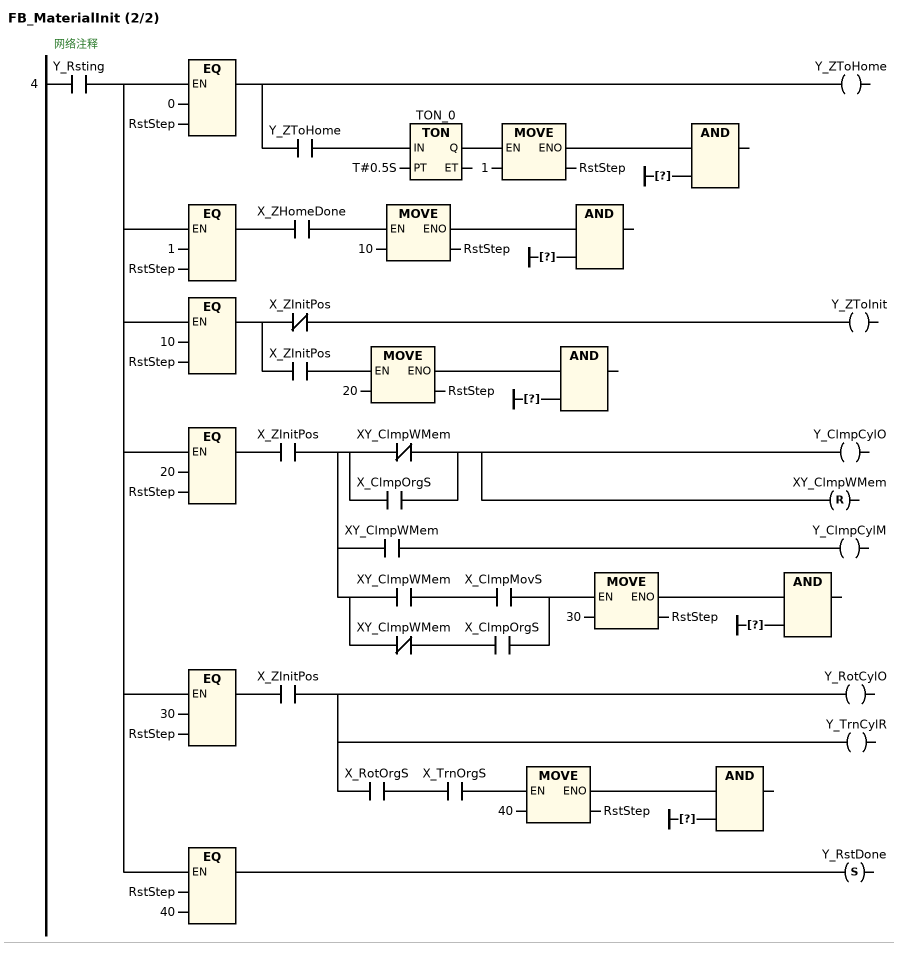
// NETWORK 4
// 网络注释
_w2 := Y_Rsting AND 0 = RstStep;
Y_ZToHome := _w2;
TON_0(IN := _w2 AND Y_ZToHome, PT := T#0.5S); // TON
_w3 := TON_0.Q;
IF _w3 THEN RstStep := 1; END_IF
_w4 := (Y_Rsting AND 1 = RstStep) AND X_ZHomeDone;
IF _w4 THEN RstStep := 10; END_IF
_w5 := Y_Rsting AND 10 = RstStep;
_w6 := _w5 AND NOT X_ZInitPos;
Y_ZToInit := _w6;
IF _w5 AND X_ZInitPos THEN RstStep := 20; END_IF
_w7 := (Y_Rsting AND 20 = RstStep) AND X_ZInitPos;
_w8 := _w7 AND NOT XY_ClmpWMem OR _w7 AND X_ClmpOrgS;
Y_ClmpCylO := _w8;
XY_ClmpWMem R= _w8;
_w9 := _w7 AND XY_ClmpWMem;
Y_ClmpCylM := _w9;
_w10 := (_w7 AND XY_ClmpWMem) AND X_ClmpMovS OR (_w7 AND NOT XY_ClmpWMem) AND X_ClmpOrgS;
IF _w10 THEN RstStep := 30; END_IF
_w11 := (Y_Rsting AND 30 = RstStep) AND X_ZInitPos;
Y_RotCylO := _w11;
Y_TrnCylR := _w11;
_w12 := (_w11 AND X_RotOrgS) AND X_TrnOrgS;
IF _w12 THEN RstStep := 40; END_IF
_w13 := Y_Rsting AND RstStep = 40;
Y_RstDone S= _w13;

END_FUNCTION_BLOCK

// Device/Application/02_功能块/初始化/FB_MainlineInit
FUNCTION_BLOCK FB_MainlineInit
VAR_INPUT
X_EN: BOOL;
X_RstEn : BOOL;
X_RstStart : BOOL;
X_TrnOrgS: BOOL;
X_LLftOrgS: BOOL;
X_LClmpOrgS: BOOL;
X_LClmpMovS: BOOL;
X_LRotOrgS: BOOL;
END_VAR

VAR_OUTPUT
Y_ENO: BOOL;
Y_Rsting : BOOL;
Y_RstDone : BOOL;
Y_TrnCylR: BOOL;
Y_LLftCylR: BOOL;
Y_LClmpCylR: BOOL;
Y_LClmpCylM: BOOL;
Y_LRotCylR: BOOL;
END_VAR

VAR_IN_OUT
	XY_LClmpWM : BOOL;
END_VAR

VAR
	PLS_0: R_TRIG;
	RstStep: INT;
END_VAR
VAR // added by the converter: edge detectors and wires of the graphical bodies
    _w1, _w2, _w3, _w4, _w5, _w6, _w7, _w8, _w9, _w10 : BOOL;
END_VAR

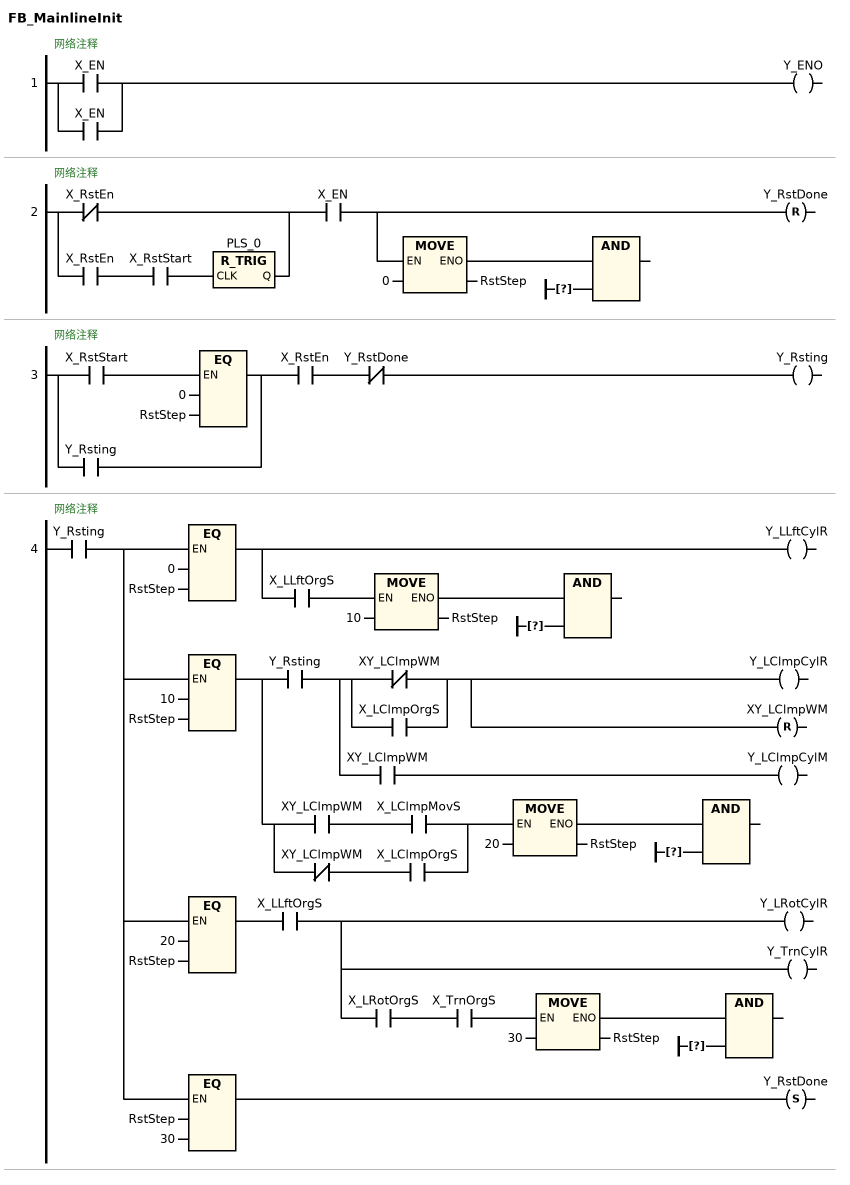
// NETWORK 1
// 网络注释
Y_ENO := X_EN OR X_EN;

// NETWORK 2
// 网络注释
PLS_0(CLK := X_RstEn AND X_RstStart); // R_TRIG
_w1 := (NOT X_RstEn OR PLS_0.Q) AND X_EN;
Y_RstDone R= _w1;
IF _w1 THEN RstStep := 0; END_IF

// NETWORK 3
// 网络注释
Y_Rsting := (X_RstStart AND 0 = RstStep OR Y_Rsting) AND X_RstEn AND NOT Y_RstDone;

// NETWORK 4
// 网络注释
_w2 := Y_Rsting AND 0 = RstStep;
Y_LLftCylR := _w2;
IF _w2 AND X_LLftOrgS THEN RstStep := 10; END_IF
_w3 := Y_Rsting AND 10 = RstStep;
_w4 := _w3 AND Y_Rsting;
_w5 := _w4 AND NOT XY_LClmpWM OR _w4 AND X_LClmpOrgS;
Y_LClmpCylR := _w5;
XY_LClmpWM R= _w5;
_w6 := _w4 AND XY_LClmpWM;
Y_LClmpCylM := _w6;
_w7 := (_w3 AND XY_LClmpWM) AND X_LClmpMovS OR (_w3 AND NOT XY_LClmpWM) AND X_LClmpOrgS;
IF _w7 THEN RstStep := 20; END_IF
_w8 := (Y_Rsting AND 20 = RstStep) AND X_LLftOrgS;
Y_LRotCylR := _w8;
Y_TrnCylR := _w8;
_w9 := (_w8 AND X_LRotOrgS) AND X_TrnOrgS;
IF _w9 THEN RstStep := 30; END_IF
_w10 := Y_Rsting AND RstStep = 30;
Y_RstDone S= _w10;

END_FUNCTION_BLOCK

// Device/Application/03_程序/异常/Error
PROGRAM Error
VAR
	E_A:  BOOL;
	E_A1: BOOL;
	E_A2: BOOL;
	E_A3: BOOL;
	Z_A_Anom: BOOL;
	
E_B:  BOOL;

E_C:  BOOL;
E_C1: BOOL;
E_C2: BOOL;
E_C3: BOOL;

Z_C_Anom: BOOL;
END_VAR
VAR // added by the converter: edge detectors and wires of the graphical bodies
    _w1, _w2, _w3, _w4, _w5, _w6, _w7, _w8, _w9, _w10 : BOOL;
END_VAR

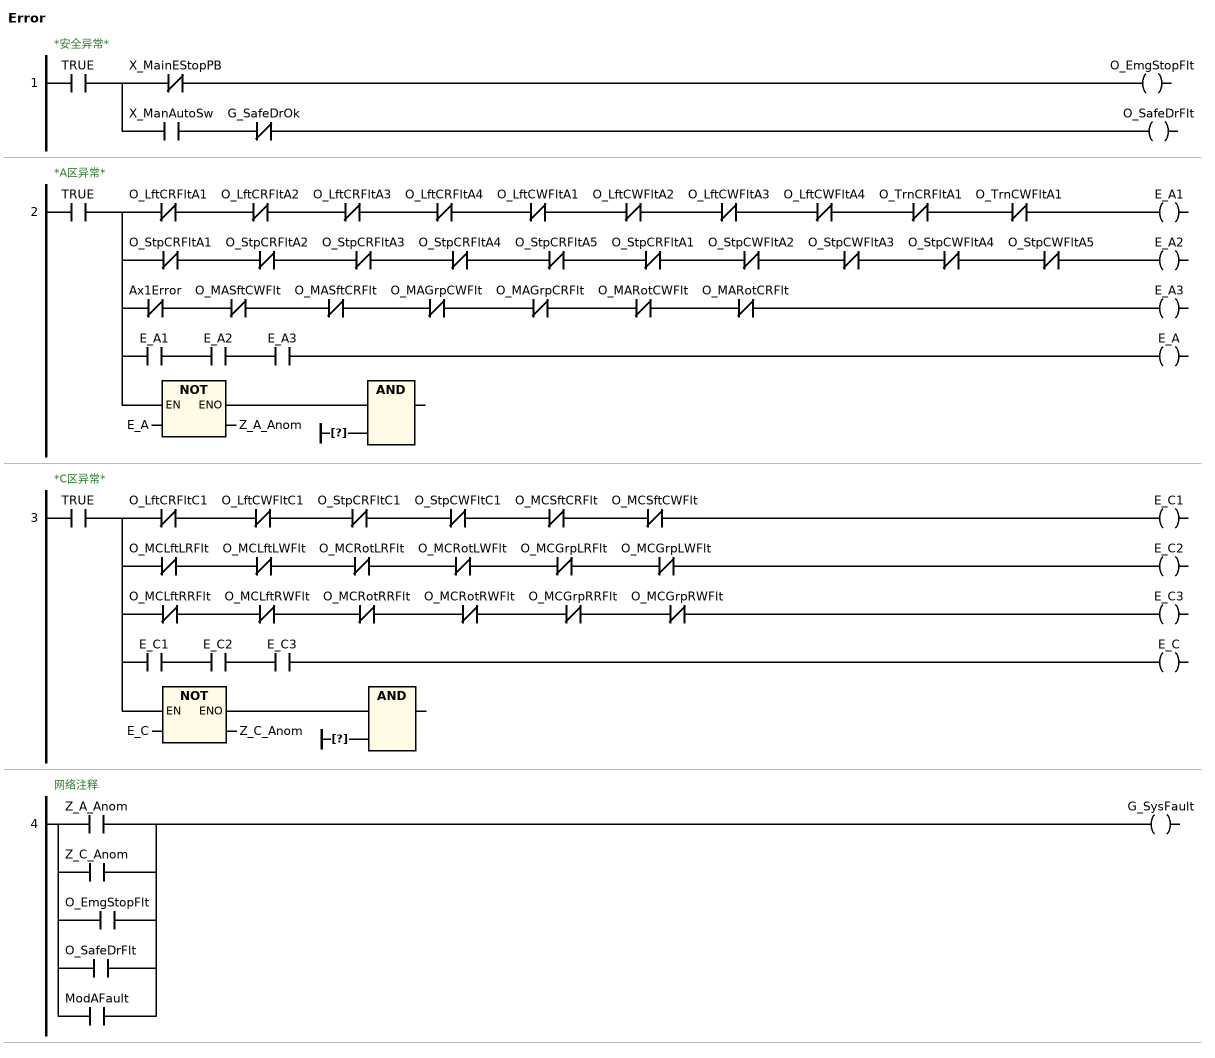
// NETWORK 1
// *安全异常*
_w1 := TRUE AND NOT X_MainEStopPB;
O_EmgStopFlt := _w1;
_w2 := (TRUE AND X_ManAutoSw) AND NOT G_SafeDrOk;
O_SafeDrFlt := _w2;

// NETWORK 2
// *A区异常*
_w3 := (TRUE AND NOT O_LftCRFltA1) AND NOT O_LftCRFltA2 AND NOT O_LftCRFltA3 AND NOT O_LftCRFltA4 AND NOT O_LftCWFltA1 AND NOT O_LftCWFltA2 AND NOT O_LftCWFltA3 AND NOT O_LftCWFltA4 AND NOT O_TrnCRFltA1 AND NOT O_TrnCWFltA1;
E_A1 := _w3;
_w4 := (TRUE AND NOT O_StpCRFltA1) AND NOT O_StpCRFltA2 AND NOT O_StpCRFltA3 AND NOT O_StpCRFltA4 AND NOT O_StpCRFltA5 AND NOT O_StpCRFltA1 AND NOT O_StpCWFltA2 AND NOT O_StpCWFltA3 AND NOT O_StpCWFltA4 AND NOT O_StpCWFltA5;
E_A2 := _w4;
_w5 := (TRUE AND NOT Ax1Error) AND NOT O_MASftCWFlt AND NOT O_MASftCRFlt AND NOT O_MAGrpCWFlt AND NOT O_MAGrpCRFlt AND NOT O_MARotCWFlt AND NOT O_MARotCRFlt;
E_A3 := _w5;
_w6 := (TRUE AND E_A1) AND E_A2 AND E_A3;
E_A := _w6;
Z_A_Anom := NOT E_A;

// NETWORK 3
// *C区异常*
_w7 := (TRUE AND NOT O_LftCRFltC1) AND NOT O_LftCWFltC1 AND NOT O_StpCRFltC1 AND NOT O_StpCWFltC1 AND NOT O_MCSftCRFlt AND NOT O_MCSftCWFlt;
E_C1 := _w7;
_w8 := (TRUE AND NOT O_MCLftLRFlt) AND NOT O_MCLftLWFlt AND NOT O_MCRotLRFlt AND NOT O_MCRotLWFlt AND NOT O_MCGrpLRFlt AND NOT O_MCGrpLWFlt;
E_C2 := _w8;
_w9 := (TRUE AND NOT O_MCLftRRFlt) AND NOT O_MCLftRWFlt AND NOT O_MCRotRRFlt AND NOT O_MCRotRWFlt AND NOT O_MCGrpRRFlt AND NOT O_MCGrpRWFlt;
E_C3 := _w9;
_w10 := (TRUE AND E_C1) AND E_C2 AND E_C3;
E_C := _w10;
Z_C_Anom := NOT E_C;

// NETWORK 4
// 网络注释
G_SysFault := Z_A_Anom OR Z_C_Anom OR O_EmgStopFlt OR O_SafeDrFlt OR ModAFault;

END_PROGRAM

// Device/Application/03_程序/自动/Auto_A
PROGRAM Auto_A
VAR

	R_TRIG_A1: R_TRIG;
	
	TON_0: TON;
	ModA_Pro: BOOL;
	PLSA: R_TRIG;
	ModA_Tst: BOOL;
	TON_1: TON;
	TON_2: TON;
	PLS_0: R_TRIG;
	TON_3: TON;
	TON_4: TON;
	TON_5: TON;
	TON_6: TON;
	TON_7: TON;
	TON_8: TON;
	TON_9: TON;
	R_TRIG_0: R_TRIG;
	TON_10: TON;
END_VAR
VAR // added by the converter: edge detectors and wires of the graphical bodies
    _w1, _w2, _w3, _w4, _w5, _w6, _w7, _w8, _w9, _w10, _w11, _w12, _w13, _w14, _w15, _w16, _w17, _w18, _w19, _w20, _w21, _w22, _w23, _w24, _w25, _w26, _w27, _w28, _w29, _w30, _w31, _w32, _w33, _w34, _w35, _w36, _w37, _w38, _w39, _w40, _w41, _w42, _w43, _w44, _w45, _w46, _w47, _w48, _w49, _w50, _w51, _w52, _w53, _w54, _w55, _w56, _w57, _w58, _w59, _w60, _w61, _w62, _w63, _w64, _w65, _w66, _w67, _w68, _w69, _w70, _w71, _w72, _w73, _w74, _w75, _w76, _w77, _w78, _w79, _w80, _w81, _w82, _w83, _w84, _w85 : BOOL;
END_VAR

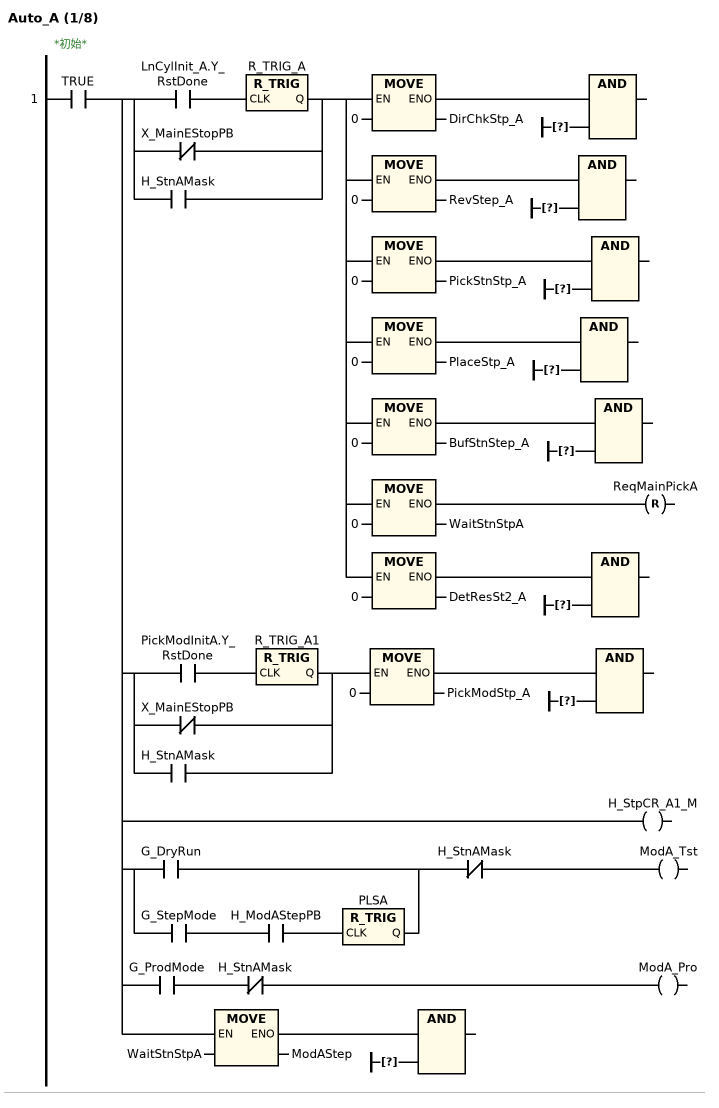
// NETWORK 1
// *初始*
R_TRIG_A(CLK := TRUE AND LnCylInit_A.Y_RstDone); // R_TRIG
_w1 := R_TRIG_A.Q OR TRUE AND NOT X_MainEStopPB OR TRUE AND H_StnAMask;
IF _w1 THEN DirChkStp_A := 0; END_IF
IF _w1 THEN RevStep_A := 0; END_IF
IF _w1 THEN PickStnStp_A := 0; END_IF
IF _w1 THEN PlaceStp_A := 0; END_IF
IF _w1 THEN BufStnStep_A := 0; END_IF
IF _w1 THEN WaitStnStpA := 0; END_IF
ReqMainPickA R= _w1;
IF _w1 THEN DetResSt2_A := 0; END_IF
R_TRIG_A1(CLK := TRUE AND PickModInitA.Y_RstDone); // R_TRIG
_w2 := R_TRIG_A1.Q OR TRUE AND NOT X_MainEStopPB OR TRUE AND H_StnAMask;
IF _w2 THEN PickModStp_A := 0; END_IF
H_StpCR_A1_M := TRUE;
PLSA(CLK := (TRUE AND G_StepMode) AND H_ModAStepPB); // R_TRIG
_w3 := (TRUE AND G_DryRun OR PLSA.Q) AND NOT H_StnAMask;
ModA_Tst := _w3;
_w4 := (TRUE AND G_ProdMode) AND NOT H_StnAMask;
ModA_Pro := _w4;
ModAStep := WaitStnStpA;

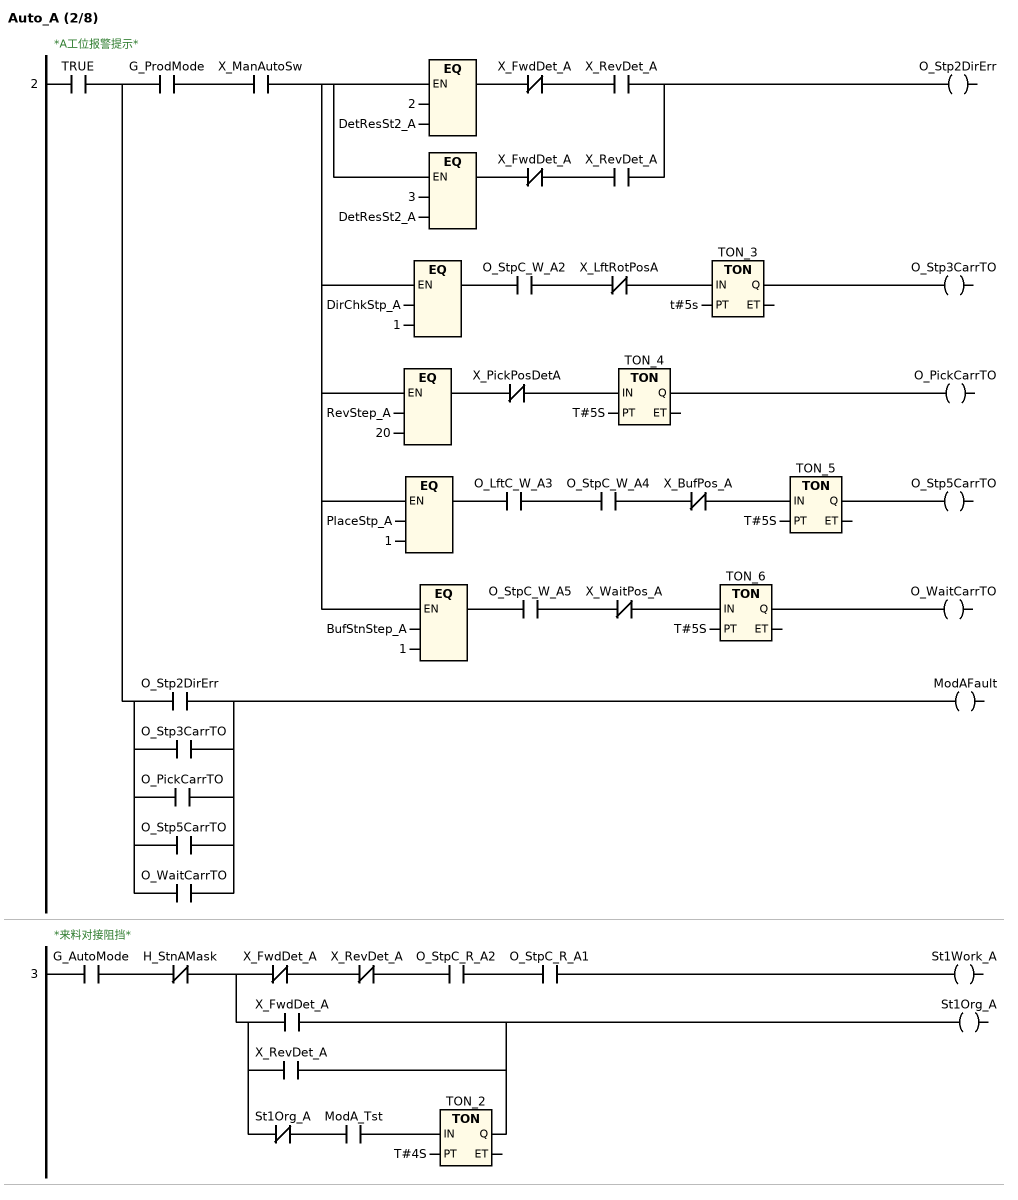
// NETWORK 2
// *A工位报警提示*
_w5 := (TRUE AND G_ProdMode) AND X_ManAutoSw;
_w6 := (_w5 AND 2 = DetResSt2_A) AND NOT X_FwdDet_A AND X_RevDet_A OR (_w5 AND 3 = DetResSt2_A) AND NOT X_FwdDet_A AND X_RevDet_A;
O_Stp2DirErr := _w6;
TON_3(IN := (_w5 AND DirChkStp_A = 1) AND O_StpC_W_A2 AND NOT X_LftRotPosA, PT := t#5s); // TON
O_Stp3CarrTO := TON_3.Q;
TON_4(IN := (_w5 AND RevStep_A = 20) AND NOT X_PickPosDetA, PT := T#5S); // TON
O_PickCarrTO := TON_4.Q;
TON_5(IN := (_w5 AND PlaceStp_A = 1) AND O_LftC_W_A3 AND O_StpC_W_A4 AND NOT X_BufPos_A, PT := T#5S); // TON
O_Stp5CarrTO := TON_5.Q;
TON_6(IN := (_w5 AND BufStnStep_A = 1) AND O_StpC_W_A5 AND NOT X_WaitPos_A, PT := T#5S); // TON
O_WaitCarrTO := TON_6.Q;
_w7 := TRUE AND O_Stp2DirErr OR TRUE AND O_Stp3CarrTO OR TRUE AND O_PickCarrTO OR TRUE AND O_Stp5CarrTO OR TRUE AND O_WaitCarrTO;
ModAFault := _w7;

// NETWORK 3
// *来料对接阻挡*
_w8 := G_AutoMode AND NOT H_StnAMask;
_w9 := (_w8 AND NOT X_FwdDet_A) AND NOT X_RevDet_A AND O_StpC_R_A2 AND O_StpC_R_A1;
St1Work_A := _w9;
TON_2(IN := (_w8 AND NOT St1Org_A) AND ModA_Tst, PT := T#4S); // TON
_w10 := _w8 AND X_FwdDet_A OR _w8 AND X_RevDet_A OR TON_2.Q;
St1Org_A := _w10;

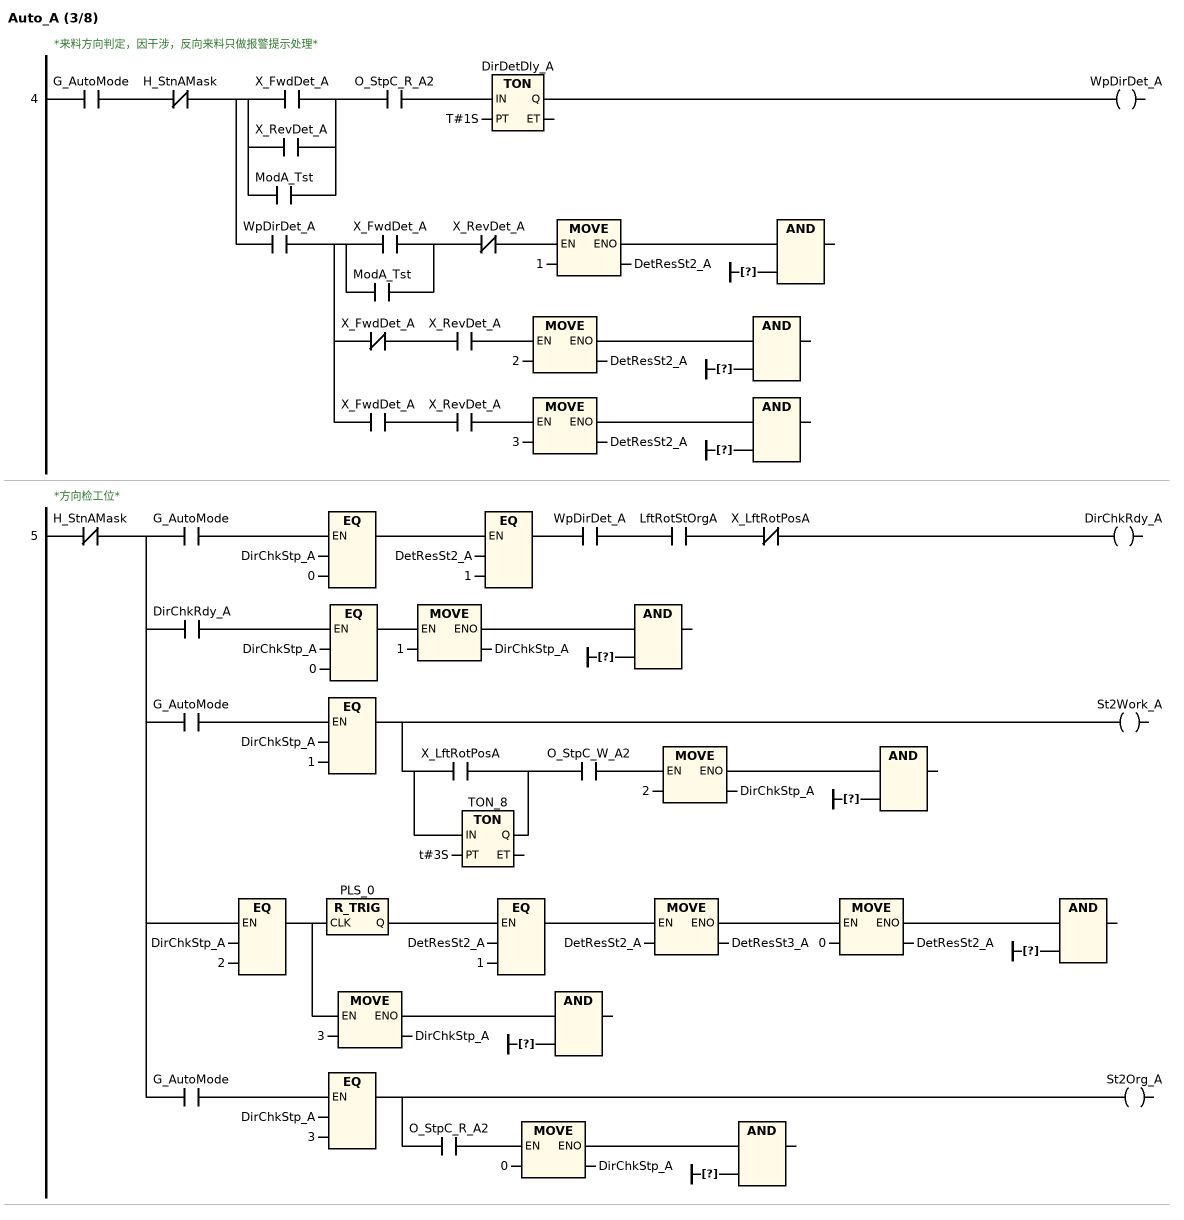
// NETWORK 4
// *来料方向判定，因干涉，反向来料只做报警提示处理*
_w11 := G_AutoMode AND NOT H_StnAMask;
DirDetDly_A(IN := (_w11 AND X_FwdDet_A OR _w11 AND X_RevDet_A OR _w11 AND ModA_Tst) AND O_StpC_R_A2, PT := T#1S); // TON
WpDirDet_A := DirDetDly_A.Q;
_w12 := _w11 AND WpDirDet_A;
_w13 := (_w12 AND X_FwdDet_A OR _w12 AND ModA_Tst) AND NOT X_RevDet_A;
IF _w13 THEN DetResSt2_A := 1; END_IF
_w14 := (_w12 AND NOT X_FwdDet_A) AND X_RevDet_A;
IF _w14 THEN DetResSt2_A := 2; END_IF
_w15 := (_w12 AND X_FwdDet_A) AND X_RevDet_A;
IF _w15 THEN DetResSt2_A := 3; END_IF

// NETWORK 5
// *方向检工位*
_w16 := NOT H_StnAMask;
_w17 := (_w16 AND G_AutoMode AND DirChkStp_A = 0 AND DetResSt2_A = 1) AND WpDirDet_A AND LftRotStOrgA AND NOT X_LftRotPosA;
DirChkRdy_A := _w17;
IF _w16 AND DirChkRdy_A AND DirChkStp_A = 0 THEN DirChkStp_A := 1; END_IF
_w18 := _w16 AND G_AutoMode AND DirChkStp_A = 1;
St2Work_A := _w18;
TON_8(IN := _w18, PT := t#3S); // TON
_w19 := (_w18 AND X_LftRotPosA OR TON_8.Q) AND O_StpC_W_A2;
IF _w19 THEN DirChkStp_A := 2; END_IF
_w20 := _w16 AND DirChkStp_A = 2;
PLS_0(CLK := _w20); // R_TRIG
_w21 := PLS_0.Q AND DetResSt2_A = 1;
IF _w21 THEN DetResSt3_A := DetResSt2_A; END_IF
IF _w21 THEN DetResSt2_A := 0; END_IF
IF _w20 THEN DirChkStp_A := 3; END_IF
_w22 := _w16 AND G_AutoMode AND DirChkStp_A = 3;
St2Org_A := _w22;
IF _w22 AND O_StpC_R_A2 THEN DirChkStp_A := 0; END_IF

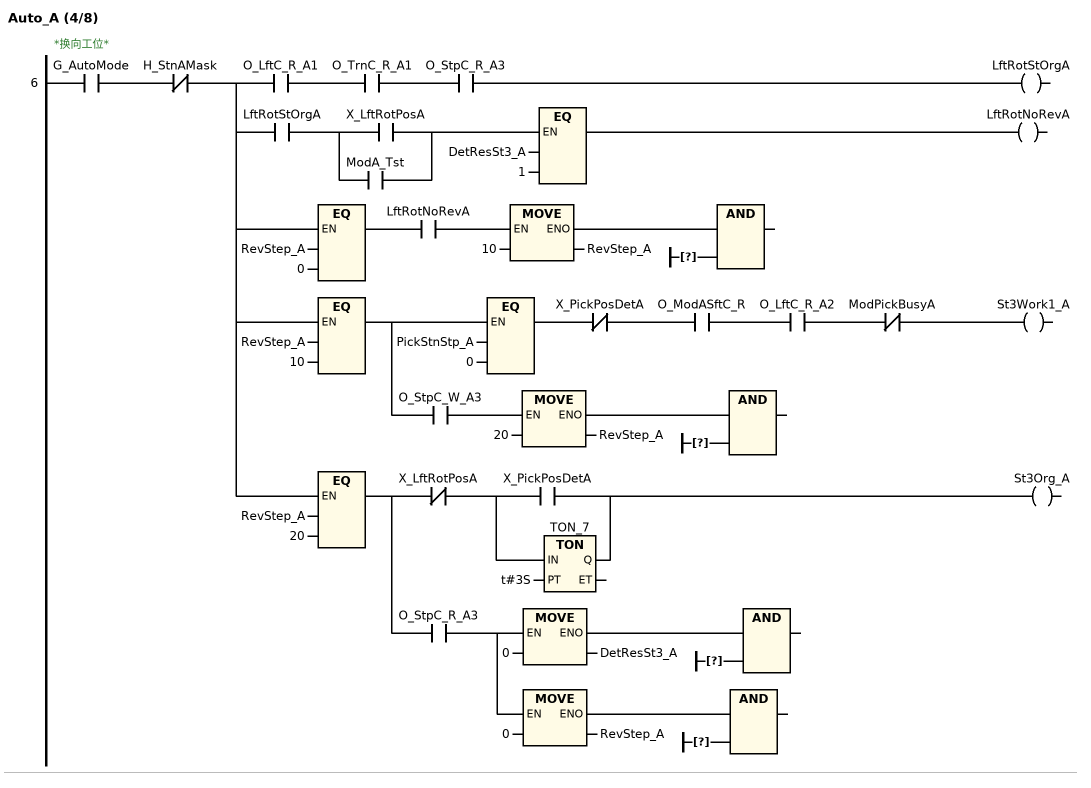
// NETWORK 6
// *换向工位*
_w23 := G_AutoMode AND NOT H_StnAMask;
_w24 := (_w23 AND O_LftC_R_A1) AND O_TrnC_R_A1 AND O_StpC_R_A3;
LftRotStOrgA := _w24;
_w25 := _w23 AND LftRotStOrgA;
_w26 := (_w25 AND X_LftRotPosA OR _w25 AND ModA_Tst) AND DetResSt3_A = 1;
LftRotNoRevA := _w26;
_w27 := (_w23 AND RevStep_A = 0) AND LftRotNoRevA;
IF _w27 THEN RevStep_A := 10; END_IF
_w28 := _w23 AND RevStep_A = 10;
_w29 := (_w28 AND PickStnStp_A = 0) AND NOT X_PickPosDetA AND O_ModASftC_R AND O_LftC_R_A2 AND NOT ModPickBusyA;
St3Work1_A := _w29;
IF _w28 AND O_StpC_W_A3 THEN RevStep_A := 20; END_IF
_w30 := _w23 AND RevStep_A = 20;
_w31 := _w30 AND NOT X_LftRotPosA;
TON_7(IN := _w31, PT := t#3S); // TON
_w32 := _w31 AND X_PickPosDetA OR TON_7.Q;
St3Org_A := _w32;
_w33 := _w30 AND O_StpC_R_A3;
IF _w33 THEN DetResSt3_A := 0; END_IF
IF _w33 THEN RevStep_A := 0; END_IF

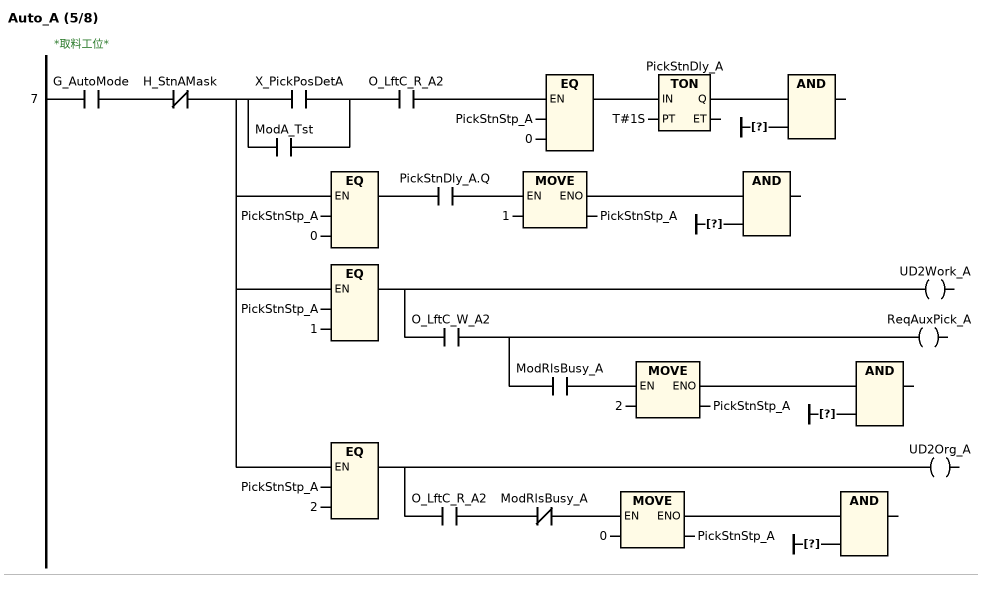
// NETWORK 7
// *取料工位*
_w34 := G_AutoMode AND NOT H_StnAMask;
PickStnDly_A(IN := (_w34 AND X_PickPosDetA OR _w34 AND ModA_Tst) AND O_LftC_R_A2 AND PickStnStp_A = 0, PT := T#1S); // TON
_w35 := (_w34 AND PickStnStp_A = 0) AND PickStnDly_A.Q;
IF _w35 THEN PickStnStp_A := 1; END_IF
_w36 := _w34 AND PickStnStp_A = 1;
UD2Work_A := _w36;
_w37 := _w36 AND O_LftC_W_A2;
ReqAuxPick_A := _w37;
IF _w37 AND ModRlsBusy_A THEN PickStnStp_A := 2; END_IF
_w38 := _w34 AND PickStnStp_A = 2;
UD2Org_A := _w38;
_w39 := (_w38 AND O_LftC_R_A2) AND NOT ModRlsBusy_A;
IF _w39 THEN PickStnStp_A := 0; END_IF

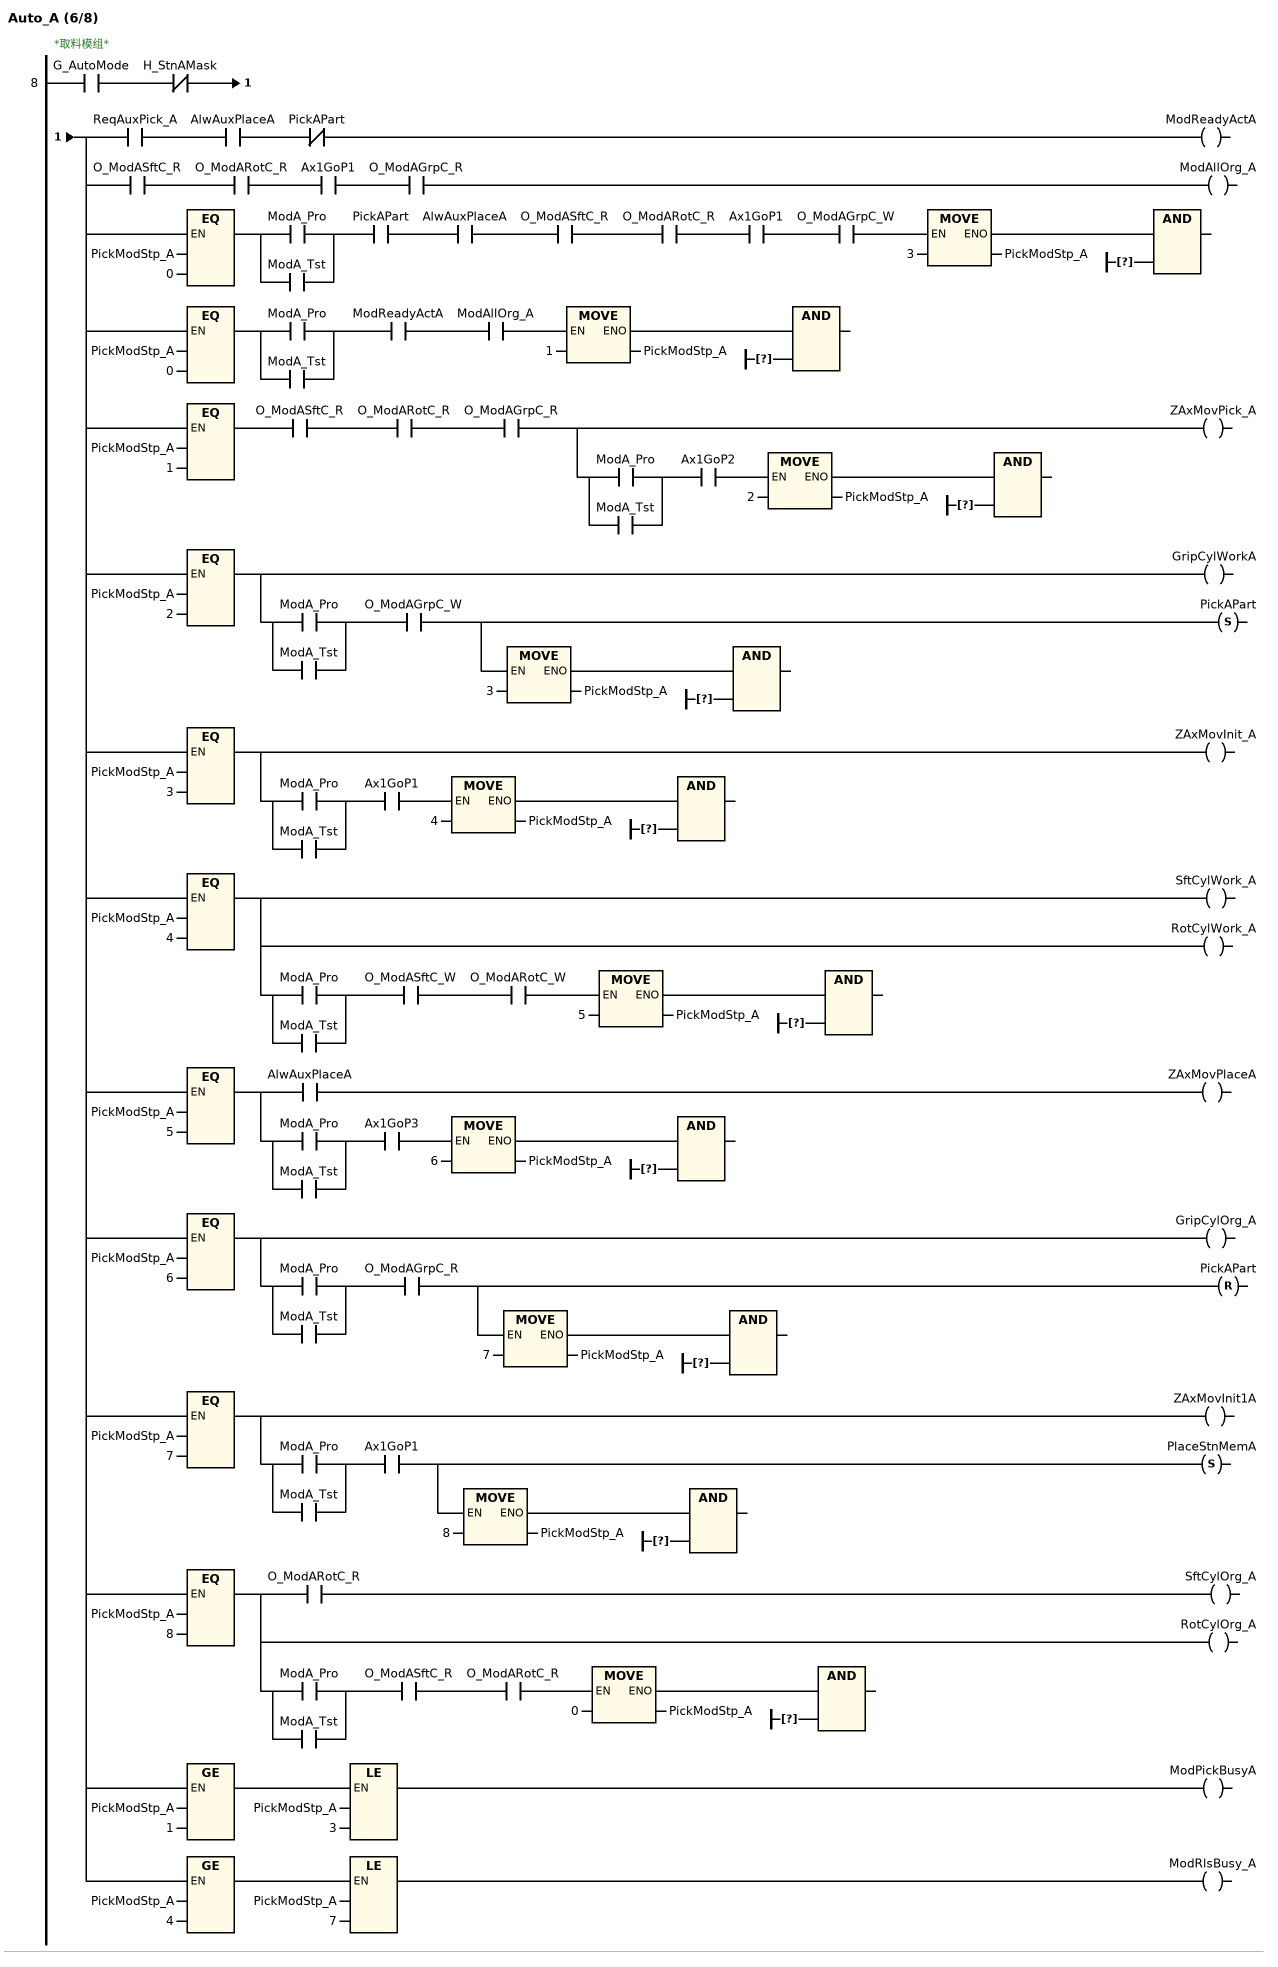
// NETWORK 8
// *取料模组*
_w40 := G_AutoMode AND NOT H_StnAMask;
_w41 := (_w40 AND ReqAuxPick_A) AND AlwAuxPlaceA AND NOT PickAPart;
ModReadyActA := _w41;
_w42 := (_w40 AND O_ModASftC_R) AND O_ModARotC_R AND Ax1GoP1 AND O_ModAGrpC_R;
ModAllOrg_A := _w42;
_w43 := _w40 AND PickModStp_A = 0;
_w44 := (_w43 AND ModA_Pro OR _w43 AND ModA_Tst) AND PickAPart AND AlwAuxPlaceA AND O_ModASftC_R AND O_ModARotC_R AND Ax1GoP1 AND O_ModAGrpC_W;
IF _w44 THEN PickModStp_A := 3; END_IF
_w45 := _w40 AND PickModStp_A = 0;
_w46 := (_w45 AND ModA_Pro OR _w45 AND ModA_Tst) AND ModReadyActA AND ModAllOrg_A;
IF _w46 THEN PickModStp_A := 1; END_IF
_w47 := (_w40 AND PickModStp_A = 1) AND O_ModASftC_R AND O_ModARotC_R AND O_ModAGrpC_R;
ZAxMovPick_A := _w47;
_w48 := (_w47 AND ModA_Pro OR _w47 AND ModA_Tst) AND Ax1GoP2;
IF _w48 THEN PickModStp_A := 2; END_IF
_w49 := _w40 AND PickModStp_A = 2;
GripCylWorkA := _w49;
_w50 := (_w49 AND ModA_Pro OR _w49 AND ModA_Tst) AND O_ModAGrpC_W;
PickAPart S= _w50;
IF _w50 THEN PickModStp_A := 3; END_IF
_w51 := _w40 AND PickModStp_A = 3;
ZAxMovInit_A := _w51;
_w52 := (_w51 AND ModA_Pro OR _w51 AND ModA_Tst) AND Ax1GoP1;
IF _w52 THEN PickModStp_A := 4; END_IF
_w53 := _w40 AND PickModStp_A = 4;
SftCylWork_A := _w53;
RotCylWork_A := _w53;
_w54 := (_w53 AND ModA_Pro OR _w53 AND ModA_Tst) AND O_ModASftC_W AND O_ModARotC_W;
IF _w54 THEN PickModStp_A := 5; END_IF
_w55 := _w40 AND PickModStp_A = 5;
_w56 := _w55 AND AlwAuxPlaceA;
ZAxMovPlaceA := _w56;
_w57 := (_w55 AND ModA_Pro OR _w55 AND ModA_Tst) AND Ax1GoP3;
IF _w57 THEN PickModStp_A := 6; END_IF
_w58 := _w40 AND PickModStp_A = 6;
GripCylOrg_A := _w58;
_w59 := (_w58 AND ModA_Pro OR _w58 AND ModA_Tst) AND O_ModAGrpC_R;
PickAPart R= _w59;
IF _w59 THEN PickModStp_A := 7; END_IF
_w60 := _w40 AND PickModStp_A = 7;
ZAxMovInit1A := _w60;
_w61 := (_w60 AND ModA_Pro OR _w60 AND ModA_Tst) AND Ax1GoP1;
PlaceStnMemA S= _w61;
IF _w61 THEN PickModStp_A := 8; END_IF
_w62 := _w40 AND PickModStp_A = 8;
_w63 := _w62 AND O_ModARotC_R;
SftCylOrg_A := _w63;
RotCylOrg_A := _w62;
_w64 := (_w62 AND ModA_Pro OR _w62 AND ModA_Tst) AND O_ModASftC_R AND O_ModARotC_R;
IF _w64 THEN PickModStp_A := 0; END_IF
_w65 := _w40 AND PickModStp_A >= 1 AND PickModStp_A <= 3;
ModPickBusyA := _w65;
_w66 := _w40 AND PickModStp_A >= 4 AND PickModStp_A <= 7;
ModRlsBusy_A := _w66;

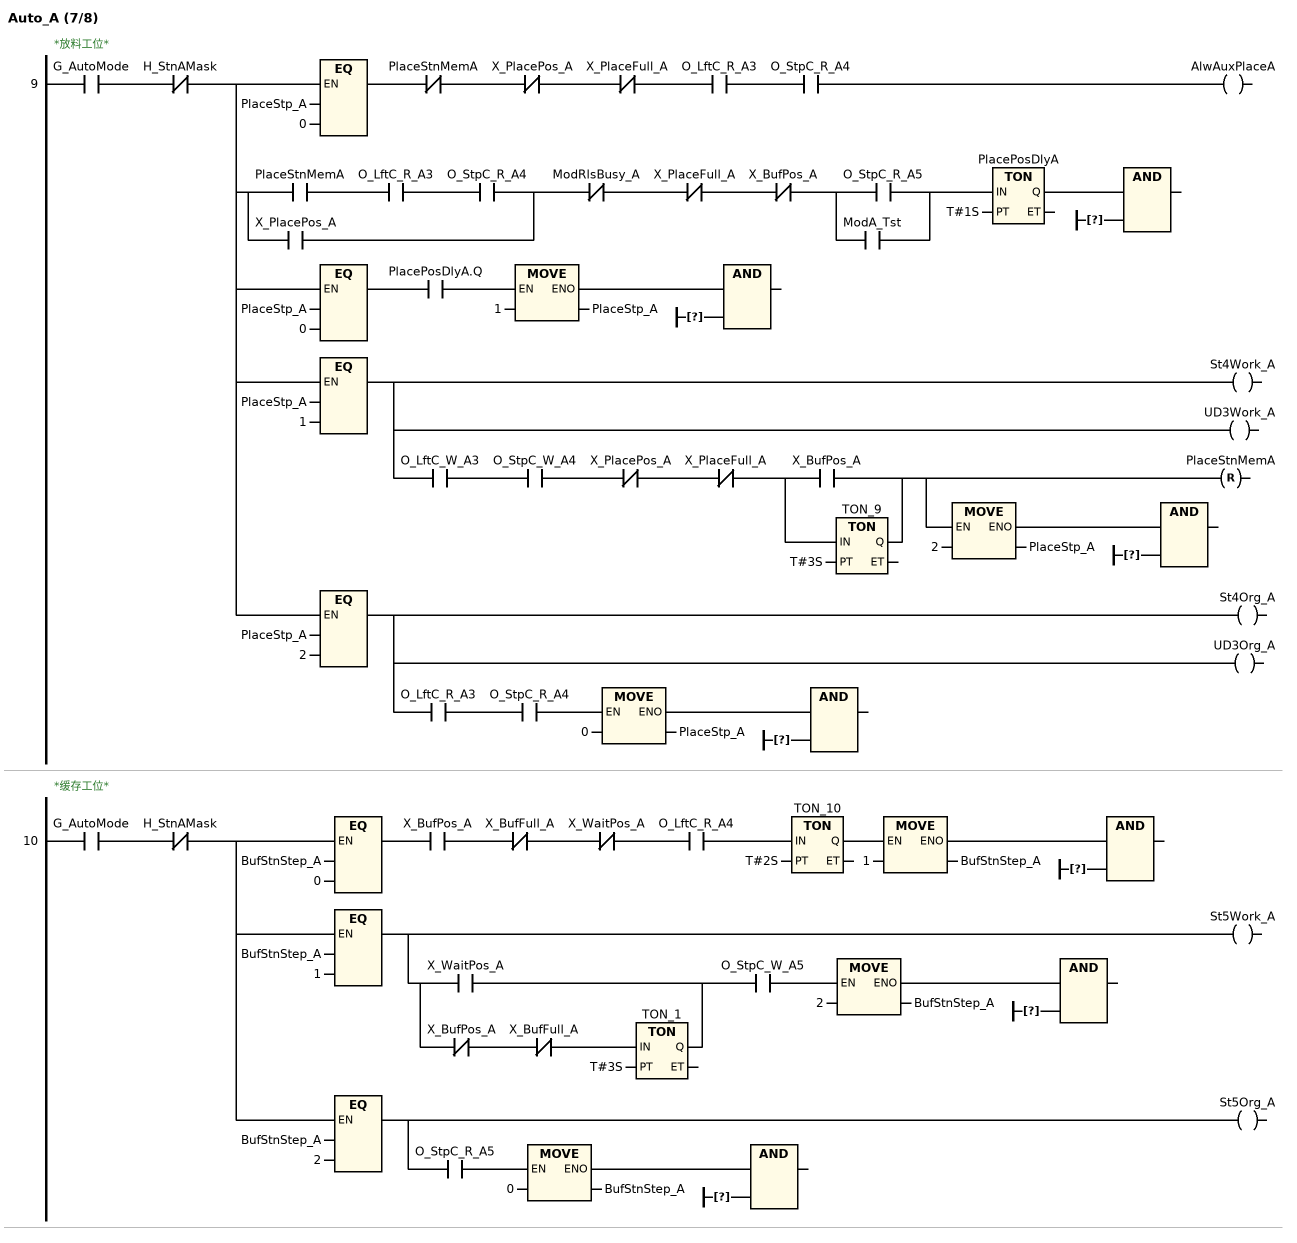
// NETWORK 9
// *放料工位*
_w67 := G_AutoMode AND NOT H_StnAMask;
_w68 := (_w67 AND PlaceStp_A = 0) AND NOT PlaceStnMemA AND NOT X_PlacePos_A AND NOT X_PlaceFull_A AND O_LftC_R_A3 AND O_StpC_R_A4;
AlwAuxPlaceA := _w68;
_w69 := ((_w67 AND PlaceStnMemA) AND O_LftC_R_A3 AND O_StpC_R_A4 OR _w67 AND X_PlacePos_A) AND NOT ModRlsBusy_A AND NOT X_PlaceFull_A AND NOT X_BufPos_A;
PlacePosDlyA(IN := _w69 AND O_StpC_R_A5 OR _w69 AND ModA_Tst, PT := T#1S); // TON
_w70 := (_w67 AND PlaceStp_A = 0) AND PlacePosDlyA.Q;
IF _w70 THEN PlaceStp_A := 1; END_IF
_w71 := _w67 AND PlaceStp_A = 1;
St4Work_A := _w71;
UD3Work_A := _w71;
_w72 := (_w71 AND O_LftC_W_A3) AND O_StpC_W_A4 AND NOT X_PlacePos_A AND NOT X_PlaceFull_A;
TON_9(IN := _w72, PT := T#3S); // TON
_w73 := _w72 AND X_BufPos_A OR TON_9.Q;
PlaceStnMemA R= _w73;
IF _w73 THEN PlaceStp_A := 2; END_IF
_w74 := _w67 AND PlaceStp_A = 2;
St4Org_A := _w74;
UD3Org_A := _w74;
_w75 := (_w74 AND O_LftC_R_A3) AND O_StpC_R_A4;
IF _w75 THEN PlaceStp_A := 0; END_IF

// NETWORK 10
// *缓存工位*
_w76 := G_AutoMode AND NOT H_StnAMask;
TON_10(IN := (_w76 AND BufStnStep_A = 0) AND X_BufPos_A AND NOT X_BufFull_A AND NOT X_WaitPos_A AND O_LftC_R_A4, PT := T#2S); // TON
_w77 := TON_10.Q;
IF _w77 THEN BufStnStep_A := 1; END_IF
_w78 := _w76 AND BufStnStep_A = 1;
St5Work_A := _w78;
TON_1(IN := (_w78 AND NOT X_BufPos_A) AND NOT X_BufFull_A, PT := T#3S); // TON
_w79 := (_w78 AND X_WaitPos_A OR TON_1.Q) AND O_StpC_W_A5;
IF _w79 THEN BufStnStep_A := 2; END_IF
_w80 := _w76 AND BufStnStep_A = 2;
St5Org_A := _w80;
IF _w80 AND O_StpC_R_A5 THEN BufStnStep_A := 0; END_IF

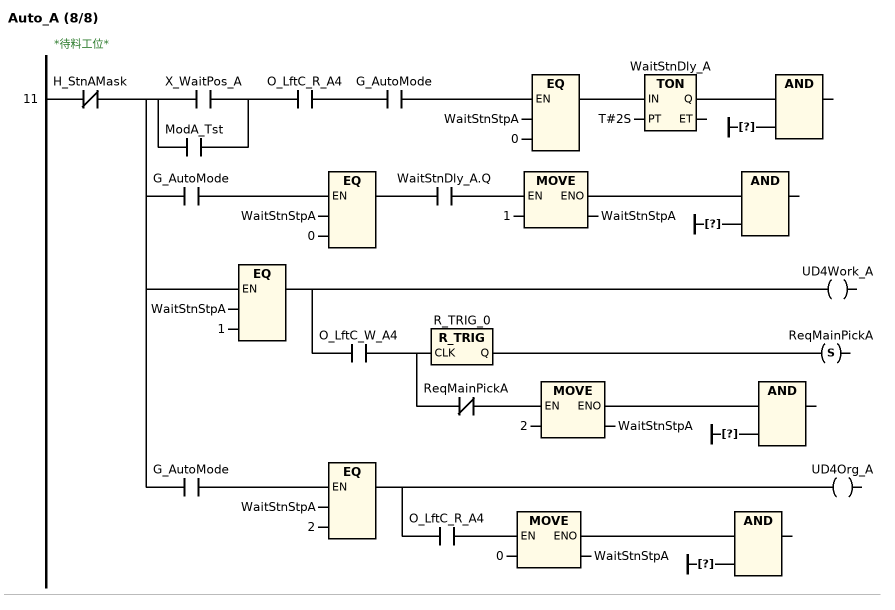
// NETWORK 11
// *待料工位*
_w81 := NOT H_StnAMask;
WaitStnDly_A(IN := (_w81 AND X_WaitPos_A OR _w81 AND ModA_Tst) AND O_LftC_R_A4 AND G_AutoMode AND WaitStnStpA = 0, PT := T#2S); // TON
_w82 := (_w81 AND G_AutoMode AND WaitStnStpA = 0) AND WaitStnDly_A.Q;
IF _w82 THEN WaitStnStpA := 1; END_IF
_w83 := _w81 AND WaitStnStpA = 1;
UD4Work_A := _w83;
_w84 := _w83 AND O_LftC_W_A4;
R_TRIG_0(CLK := _w84); // R_TRIG
ReqMainPickA S= R_TRIG_0.Q;
IF _w84 AND NOT ReqMainPickA THEN WaitStnStpA := 2; END_IF
_w85 := _w81 AND G_AutoMode AND WaitStnStpA = 2;
UD4Org_A := _w85;
IF _w85 AND O_LftC_R_A4 THEN WaitStnStpA := 0; END_IF

END_PROGRAM

// Device/Application/03_程序/自动/Auto_C
PROGRAM Auto_C
VAR

	DockStMemC: BOOL;
	PLSC: R_TRIG;
	ModC_Tst: BOOL;
	ModC_Pro: BOOL;
	TON_0: TON;
	manualS: BOOL;
	TON_1: TON;
	TON_2: TON;
	TON_99: TON;
END_VAR
VAR // added by the converter: edge detectors and wires of the graphical bodies
    _w1, _w2, _w3, _w4, _w5, _w6, _w7, _w8, _w9, _w10, _w11, _w12, _w13, _w14, _w15, _w16, _w17, _w18, _w19, _w20, _w21, _w22, _w23, _w24, _w25, _w26, _w27, _w28, _w29, _w30, _w31, _w32, _w33, _w34, _w35, _w36, _w37, _w38, _w39 : BOOL;
END_VAR

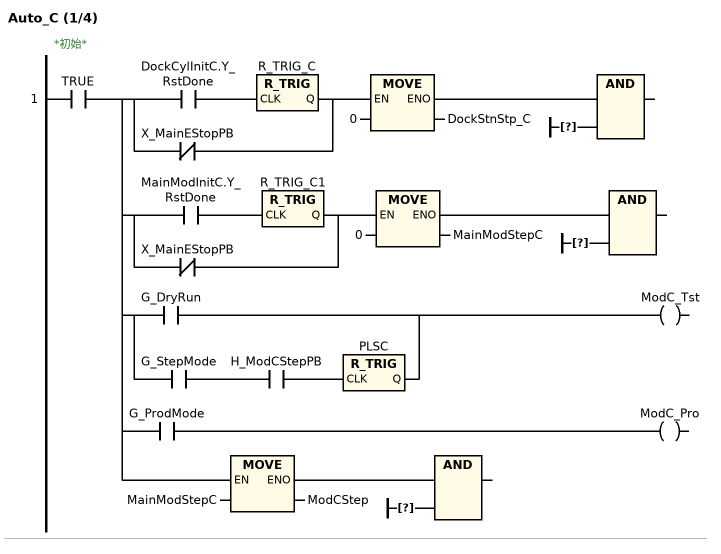
// NETWORK 1
// *初始*
R_TRIG_C(CLK := TRUE AND DockCylInitC.Y_RstDone); // R_TRIG
_w1 := R_TRIG_C.Q OR TRUE AND NOT X_MainEStopPB;
IF _w1 THEN DockStnStp_C := 0; END_IF
R_TRIG_C1(CLK := TRUE AND MainModInitC.Y_RstDone); // R_TRIG
_w2 := R_TRIG_C1.Q OR TRUE AND NOT X_MainEStopPB;
IF _w2 THEN MainModStepC := 0; END_IF
PLSC(CLK := (TRUE AND G_StepMode) AND H_ModCStepPB); // R_TRIG
_w3 := TRUE AND G_DryRun OR PLSC.Q;
ModC_Tst := _w3;
_w4 := TRUE AND G_ProdMode;
ModC_Pro := _w4;
ModCStep := MainModStepC;

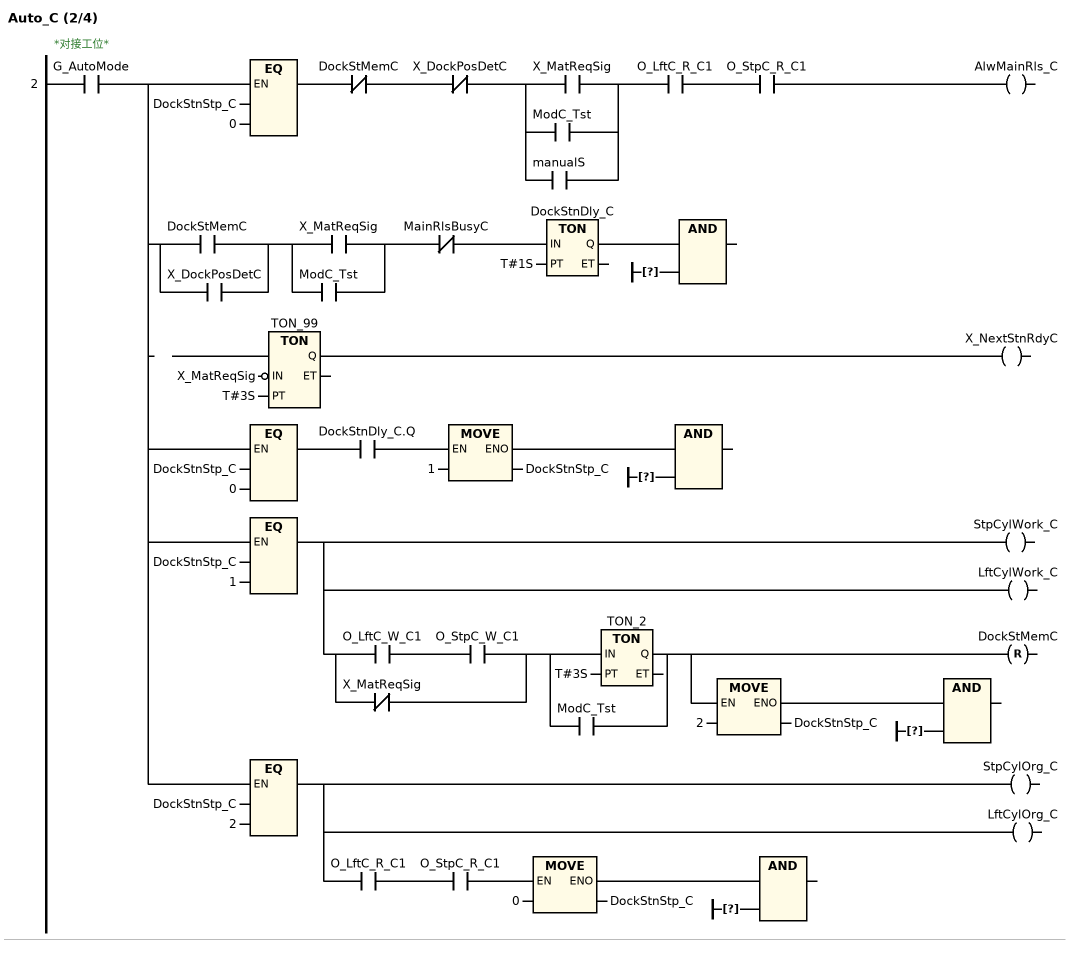
// NETWORK 2
// *对接工位*
_w5 := (G_AutoMode AND DockStnStp_C = 0) AND NOT DockStMemC AND NOT X_DockPosDetC;
_w6 := (_w5 AND X_MatReqSig OR _w5 AND ModC_Tst OR _w5 AND manualS) AND O_LftC_R_C1 AND O_StpC_R_C1;
AlwMainRls_C := _w6;
_w7 := G_AutoMode AND DockStMemC OR G_AutoMode AND X_DockPosDetC;
DockStnDly_C(IN := (_w7 AND X_MatReqSig OR _w7 AND ModC_Tst) AND NOT MainRlsBusyC, PT := T#1S); // TON
TON_99(IN := NOT X_MatReqSig, PT := T#3S); // TON
X_NextStnRdyC := TON_99.Q;
_w8 := (G_AutoMode AND DockStnStp_C = 0) AND DockStnDly_C.Q;
IF _w8 THEN DockStnStp_C := 1; END_IF
_w9 := G_AutoMode AND DockStnStp_C = 1;
StpCylWork_C := _w9;
LftCylWork_C := _w9;
_w10 := (_w9 AND O_LftC_W_C1) AND O_StpC_W_C1 OR _w9 AND NOT X_MatReqSig;
TON_2(IN := _w10, PT := T#3S); // TON
_w11 := TON_2.Q OR _w10 AND ModC_Tst;
DockStMemC R= _w11;
IF _w11 THEN DockStnStp_C := 2; END_IF
_w12 := G_AutoMode AND DockStnStp_C = 2;
StpCylOrg_C := _w12;
LftCylOrg_C := _w12;
_w13 := (_w12 AND O_LftC_R_C1) AND O_StpC_R_C1;
IF _w13 THEN DockStnStp_C := 0; END_IF

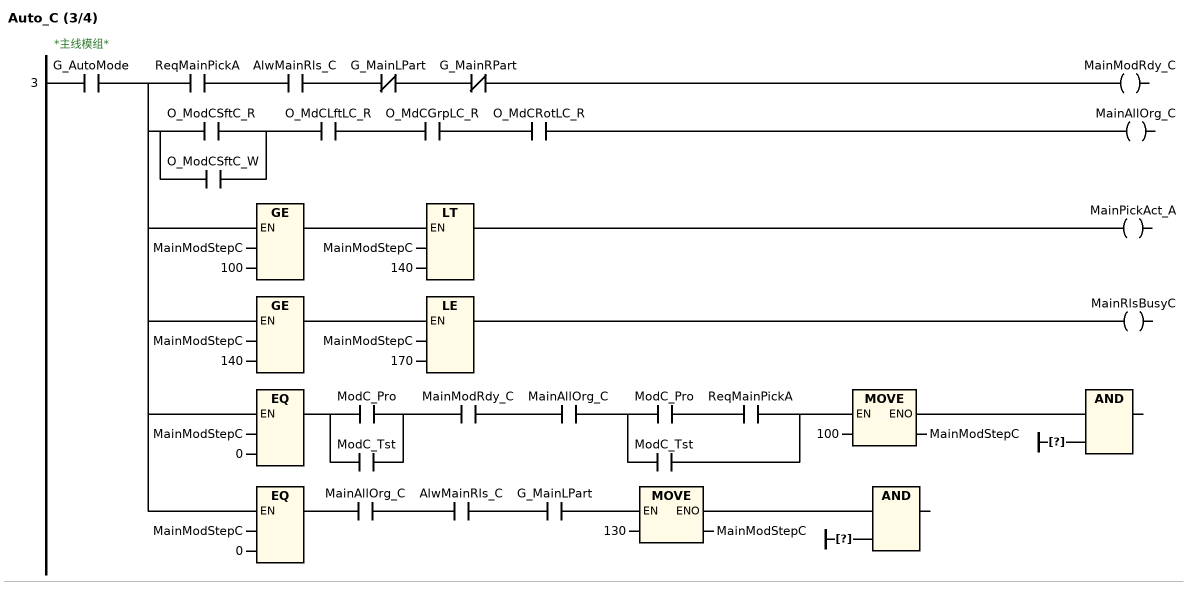
// NETWORK 3
// *主线模组*
_w14 := (G_AutoMode AND ReqMainPickA) AND AlwMainRls_C AND NOT G_MainLPart AND NOT G_MainRPart;
MainModRdy_C := _w14;
_w15 := (G_AutoMode AND O_ModCSftC_R OR G_AutoMode AND O_ModCSftC_W) AND O_MdCLftLC_R AND O_MdCGrpLC_R AND O_MdCRotLC_R;
MainAllOrg_C := _w15;
_w16 := G_AutoMode AND MainModStepC >= 100 AND MainModStepC < 140;
MainPickAct_A := _w16;
_w17 := G_AutoMode AND MainModStepC >= 140 AND MainModStepC <= 170;
MainRlsBusyC := _w17;
_w18 := G_AutoMode AND MainModStepC = 0;
_w19 := (_w18 AND ModC_Pro OR _w18 AND ModC_Tst) AND MainModRdy_C AND MainAllOrg_C;
_w20 := (_w19 AND ModC_Pro) AND ReqMainPickA OR _w19 AND ModC_Tst;
IF _w20 THEN MainModStepC := 100; END_IF
_w21 := (G_AutoMode AND MainModStepC = 0) AND MainAllOrg_C AND AlwMainRls_C AND G_MainLPart;
IF _w21 THEN MainModStepC := 130; END_IF

